REGION Network 20: #T1_ET01. ESTADO REPOSO VACIO.
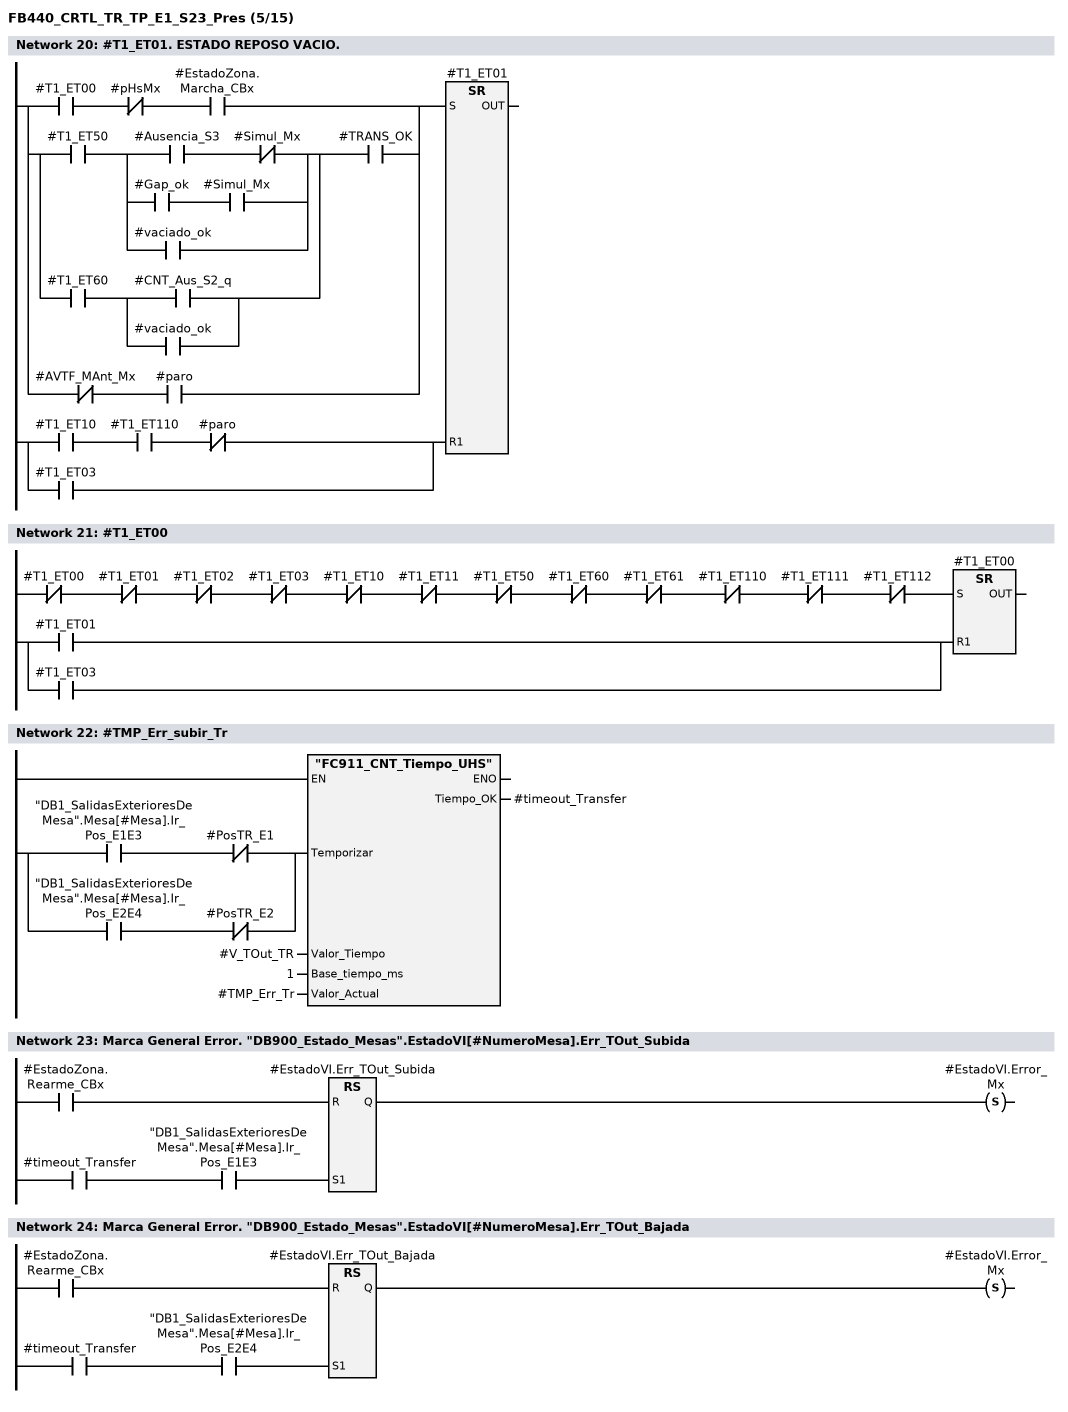
   RUNG wire#powerrail
      Contact( #T1_ET00 )
      I_Contact( #pHsMx )
      Contact( #EstadoZona.Marcha_CBx )
      wire#w1
      S_SR(operand := #T1_ET01, r1 := wire#w5)
   END_RUNG
   RUNG wire#powerrail
      Contact( #T1_ET50 )
      wire#w2
      Contact( #Ausencia_S3 )
      I_Contact( #Simul_Mx )
      wire#w3
      Contact( #TRANS_OK )
   END_RUNG wire#w1
   RUNG wire#w2
      Contact( #Gap_ok )
      Contact( #Simul_Mx )
   END_RUNG wire#w3
   RUNG wire#w2
      Contact( #vaciado_ok )
   END_RUNG wire#w3
   RUNG wire#powerrail
      Contact( #T1_ET60 )
      wire#w4
      Contact( #CNT_Aus_S2_q )
   END_RUNG wire#w3
   RUNG wire#w4
      Contact( #vaciado_ok )
   END_RUNG wire#w3
   RUNG wire#powerrail
      I_Contact( #AVTF_MAnt_Mx )
      Contact( #paro )
   END_RUNG wire#w1
   RUNG wire#powerrail
      Contact( #T1_ET10 )
      Contact( #T1_ET110 )
      I_Contact( #paro )
   END_RUNG wire#w5
   RUNG wire#powerrail
      Contact( #T1_ET03 )
   END_RUNG wire#w5
   // the same network as SCL:
   IF (#T1_ET00 AND NOT #pHsMx AND #EstadoZona.Marcha_CBx) OR (((#T1_ET50 AND ((#Ausencia_S3 AND NOT #Simul_Mx) OR (#Gap_ok AND #Simul_Mx) OR #vaciado_ok)) OR (#T1_ET60 AND (#CNT_Aus_S2_q OR #vaciado_ok))) AND #TRANS_OK) OR (NOT #AVTF_MAnt_Mx AND #paro) THEN
       #T1_ET01 := TRUE;   // SR flip-flop
   END_IF;
   IF (#T1_ET10 AND #T1_ET110 AND NOT #paro) OR #T1_ET03 THEN #T1_ET01 := FALSE; END_IF;
END_REGION

REGION Network 21: #T1_ET00
   RUNG wire#powerrail
      I_Contact( #T1_ET00 )
      I_Contact( #T1_ET01 )
      I_Contact( #T1_ET02 )
      I_Contact( #T1_ET03 )
      I_Contact( #T1_ET10 )
      I_Contact( #T1_ET11 )
      I_Contact( #T1_ET50 )
      I_Contact( #T1_ET60 )
      I_Contact( #T1_ET61 )
      I_Contact( #T1_ET110 )
      I_Contact( #T1_ET111 )
      I_Contact( #T1_ET112 )
      S_SR(operand := #T1_ET00, r1 := wire#w1)
   END_RUNG
   RUNG wire#powerrail
      Contact( #T1_ET01 )
   END_RUNG wire#w1
   RUNG wire#powerrail
      Contact( #T1_ET03 )
   END_RUNG wire#w1
   // the same network as SCL:
   IF NOT #T1_ET00 AND NOT #T1_ET01 AND NOT #T1_ET02 AND NOT #T1_ET03 AND NOT #T1_ET10 AND NOT #T1_ET11 AND NOT #T1_ET50 AND NOT #T1_ET60 AND NOT #T1_ET61 AND NOT #T1_ET110 AND NOT #T1_ET111 AND NOT #T1_ET112 THEN
       #T1_ET00 := TRUE;   // SR flip-flop
   END_IF;
   IF #T1_ET01 OR #T1_ET03 THEN #T1_ET00 := FALSE; END_IF;
END_REGION

REGION Network 22: #TMP_Err_subir_Tr
   RUNG wire#powerrail
      "FC911_CNT_Tiempo_UHS"(Temporizar := wire#w1, Valor_Tiempo := #V_TOut_TR, Base_tiempo_ms := 1, Valor_Actual := #TMP_Err_Tr, Tiempo_OK => #timeout_Transfer)
   END_RUNG
   RUNG wire#powerrail
      Contact( "DB1_SalidasExterioresDeMesa".Mesa[#Mesa].Ir_Pos_E1E3 )
      I_Contact( #PosTR_E1 )
   END_RUNG wire#w1
   RUNG wire#powerrail
      Contact( "DB1_SalidasExterioresDeMesa".Mesa[#Mesa].Ir_Pos_E2E4 )
      I_Contact( #PosTR_E2 )
   END_RUNG wire#w1
   // the same network as SCL:
   "FC911_CNT_Tiempo_UHS"(Temporizar := ("DB1_SalidasExterioresDeMesa".Mesa[#Mesa].Ir_Pos_E1E3 AND NOT #PosTR_E1) OR ("DB1_SalidasExterioresDeMesa".Mesa[#Mesa].Ir_Pos_E2E4 AND NOT #PosTR_E2),
                          Valor_Tiempo := #V_TOut_TR,
                          Base_tiempo_ms := 1,
                          Valor_Actual := #TMP_Err_Tr,
                          Tiempo_OK => #timeout_Transfer);
END_REGION

REGION Network 23: Marca General Error. "DB900_Estado_Mesas".EstadoVI[#NumeroMesa].Err_TOut_Subida
   RUNG wire#powerrail
      Contact( #EstadoZona.Rearme_CBx )
      S_RS(operand := #EstadoVI.Err_TOut_Subida, s1 := wire#w1)
      S_Coil( #EstadoVI.Error_Mx )
   END_RUNG
   RUNG wire#powerrail
      Contact( #timeout_Transfer )
      Contact( "DB1_SalidasExterioresDeMesa".Mesa[#Mesa].Ir_Pos_E1E3 )
   END_RUNG wire#w1
   // the same network as SCL:
   IF #EstadoZona.Rearme_CBx THEN
       #EstadoVI.Err_TOut_Subida := FALSE;   // RS flip-flop
   END_IF;
   IF #timeout_Transfer AND "DB1_SalidasExterioresDeMesa".Mesa[#Mesa].Ir_Pos_E1E3 THEN
       #EstadoVI.Err_TOut_Subida := TRUE;
   END_IF;
   IF #EstadoVI.Err_TOut_Subida THEN #EstadoVI.Error_Mx := TRUE; END_IF;
END_REGION

REGION Network 24: Marca General Error. "DB900_Estado_Mesas".EstadoVI[#NumeroMesa].Err_TOut_Bajada
   RUNG wire#powerrail
      Contact( #EstadoZona.Rearme_CBx )
      S_RS(operand := #EstadoVI.Err_TOut_Bajada, s1 := wire#w1)
      S_Coil( #EstadoVI.Error_Mx )
   END_RUNG
   RUNG wire#powerrail
      Contact( #timeout_Transfer )
      Contact( "DB1_SalidasExterioresDeMesa".Mesa[#Mesa].Ir_Pos_E2E4 )
   END_RUNG wire#w1
   // the same network as SCL:
   IF #EstadoZona.Rearme_CBx THEN
       #EstadoVI.Err_TOut_Bajada := FALSE;   // RS flip-flop
   END_IF;
   IF #timeout_Transfer AND "DB1_SalidasExterioresDeMesa".Mesa[#Mesa].Ir_Pos_E2E4 THEN
       #EstadoVI.Err_TOut_Bajada := TRUE;
   END_IF;
   IF #EstadoVI.Err_TOut_Bajada THEN #EstadoVI.Error_Mx := TRUE; END_IF;
END_REGION

REGION Network 25: Marca General Error. "DB900_Estado_Mesas".EstadoVI[#NumeroMesa].Err_Termico_E1_E3
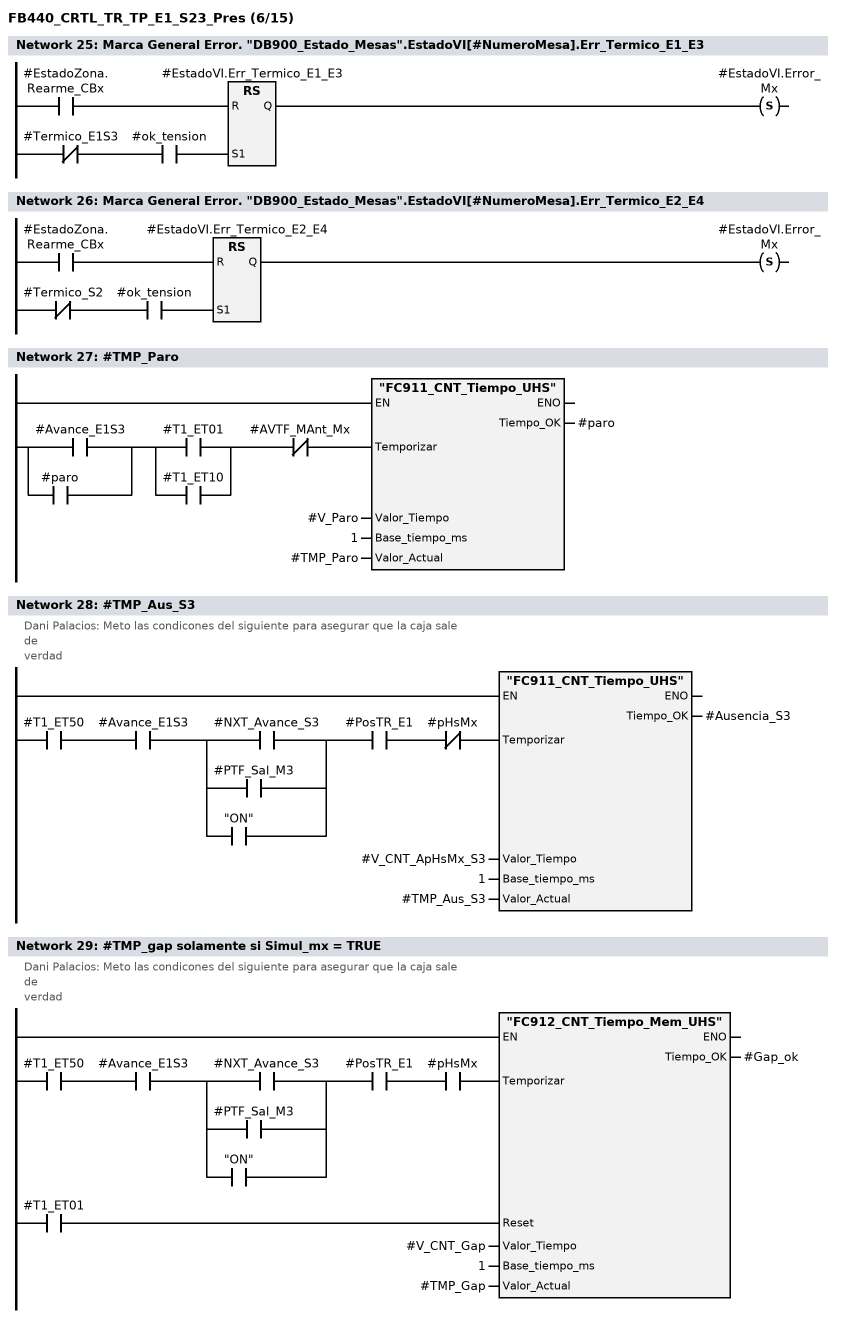
   RUNG wire#powerrail
      Contact( #EstadoZona.Rearme_CBx )
      S_RS(operand := #EstadoVI.Err_Termico_E1_E3, s1 := wire#w1)
      S_Coil( #EstadoVI.Error_Mx )
   END_RUNG
   RUNG wire#powerrail
      I_Contact( #Termico_E1S3 )
      Contact( #ok_tension )
   END_RUNG wire#w1
   // the same network as SCL:
   IF #EstadoZona.Rearme_CBx THEN
       #EstadoVI.Err_Termico_E1_E3 := FALSE;   // RS flip-flop
   END_IF;
   IF NOT #Termico_E1S3 AND #ok_tension THEN #EstadoVI.Err_Termico_E1_E3 := TRUE; END_IF;
   IF #EstadoVI.Err_Termico_E1_E3 THEN #EstadoVI.Error_Mx := TRUE; END_IF;
END_REGION

REGION Network 26: Marca General Error. "DB900_Estado_Mesas".EstadoVI[#NumeroMesa].Err_Termico_E2_E4
   RUNG wire#powerrail
      Contact( #EstadoZona.Rearme_CBx )
      S_RS(operand := #EstadoVI.Err_Termico_E2_E4, s1 := wire#w1)
      S_Coil( #EstadoVI.Error_Mx )
   END_RUNG
   RUNG wire#powerrail
      I_Contact( #Termico_S2 )
      Contact( #ok_tension )
   END_RUNG wire#w1
   // the same network as SCL:
   IF #EstadoZona.Rearme_CBx THEN
       #EstadoVI.Err_Termico_E2_E4 := FALSE;   // RS flip-flop
   END_IF;
   IF NOT #Termico_S2 AND #ok_tension THEN #EstadoVI.Err_Termico_E2_E4 := TRUE; END_IF;
   IF #EstadoVI.Err_Termico_E2_E4 THEN #EstadoVI.Error_Mx := TRUE; END_IF;
END_REGION

REGION Network 27: #TMP_Paro
   RUNG wire#powerrail
      "FC911_CNT_Tiempo_UHS"(Temporizar := wire#w3, Valor_Tiempo := #V_Paro, Base_tiempo_ms := 1, Valor_Actual := #TMP_Paro, Tiempo_OK => #paro)
   END_RUNG
   RUNG wire#powerrail
      Contact( #Avance_E1S3 )
      wire#w1
      Contact( #T1_ET01 )
      wire#w2
      I_Contact( #AVTF_MAnt_Mx )
   END_RUNG wire#w3
   RUNG wire#powerrail
      Contact( #paro )
   END_RUNG wire#w1
   RUNG wire#w1
      Contact( #T1_ET10 )
   END_RUNG wire#w2
   // the same network as SCL:
   "FC911_CNT_Tiempo_UHS"(Temporizar := (#Avance_E1S3 OR #paro) AND (#T1_ET01 OR #T1_ET10) AND NOT #AVTF_MAnt_Mx,
                          Valor_Tiempo := #V_Paro,
                          Base_tiempo_ms := 1,
                          Valor_Actual := #TMP_Paro,
                          Tiempo_OK => #paro);
END_REGION

REGION Network 28: #TMP_Aus_S3
   // Dani Palacios: Meto las condicones del siguiente para asegurar que la caja sale 
   // de 
   // verdad
   RUNG wire#powerrail
      "FC911_CNT_Tiempo_UHS"(Temporizar := wire#w3, Valor_Tiempo := #V_CNT_ApHsMx_S3, Base_tiempo_ms := 1, Valor_Actual := #TMP_Aus_S3, Tiempo_OK => #Ausencia_S3)
   END_RUNG
   RUNG wire#powerrail
      Contact( #T1_ET50 )
      Contact( #Avance_E1S3 )
      wire#w1
      Contact( #NXT_Avance_S3 )
      wire#w2
      Contact( #PosTR_E1 )
      I_Contact( #pHsMx )
   END_RUNG wire#w3
   RUNG wire#w1
      Contact( #PTF_Sal_M3 )
   END_RUNG wire#w2
   RUNG wire#w1
      Contact( "ON" )
   END_RUNG wire#w2
   // the same network as SCL:
   "FC911_CNT_Tiempo_UHS"(Temporizar := #T1_ET50 AND #Avance_E1S3 AND (#NXT_Avance_S3 OR #PTF_Sal_M3 OR "ON") AND #PosTR_E1 AND NOT #pHsMx,
                          Valor_Tiempo := #V_CNT_ApHsMx_S3,
                          Base_tiempo_ms := 1,
                          Valor_Actual := #TMP_Aus_S3,
                          Tiempo_OK => #Ausencia_S3);
END_REGION

REGION Network 29: #TMP_gap solamente si Simul_mx = TRUE
   // Dani Palacios: Meto las condicones del siguiente para asegurar que la caja sale 
   // de 
   // verdad
   RUNG wire#powerrail
      "FC912_CNT_Tiempo_Mem_UHS"(Temporizar := wire#w3, Reset := wire#w4, Valor_Tiempo := #V_CNT_Gap, Base_tiempo_ms := 1, Valor_Actual := #TMP_Gap, Tiempo_OK => #Gap_ok)
   END_RUNG
   RUNG wire#powerrail
      Contact( #T1_ET50 )
      Contact( #Avance_E1S3 )
      wire#w1
      Contact( #NXT_Avance_S3 )
      wire#w2
      Contact( #PosTR_E1 )
      Contact( #pHsMx )
   END_RUNG wire#w3
   RUNG wire#w1
      Contact( #PTF_Sal_M3 )
   END_RUNG wire#w2
   RUNG wire#w1
      Contact( "ON" )
   END_RUNG wire#w2
   RUNG wire#powerrail
      Contact( #T1_ET01 )
   END_RUNG wire#w4
   // the same network as SCL:
   "FC912_CNT_Tiempo_Mem_UHS"(Temporizar := #T1_ET50 AND #Avance_E1S3 AND (#NXT_Avance_S3 OR #PTF_Sal_M3 OR "ON") AND #PosTR_E1 AND #pHsMx,
                           Reset := #T1_ET01,
                           Valor_Tiempo := #V_CNT_Gap,
                           Base_tiempo_ms := 1,
                           Valor_Actual := #TMP_Gap,
                           Tiempo_OK => #Gap_ok);
END_REGION

REGION Network 30: tout avance
   // Nieves 16/12/17. incluyo porque no existe el error
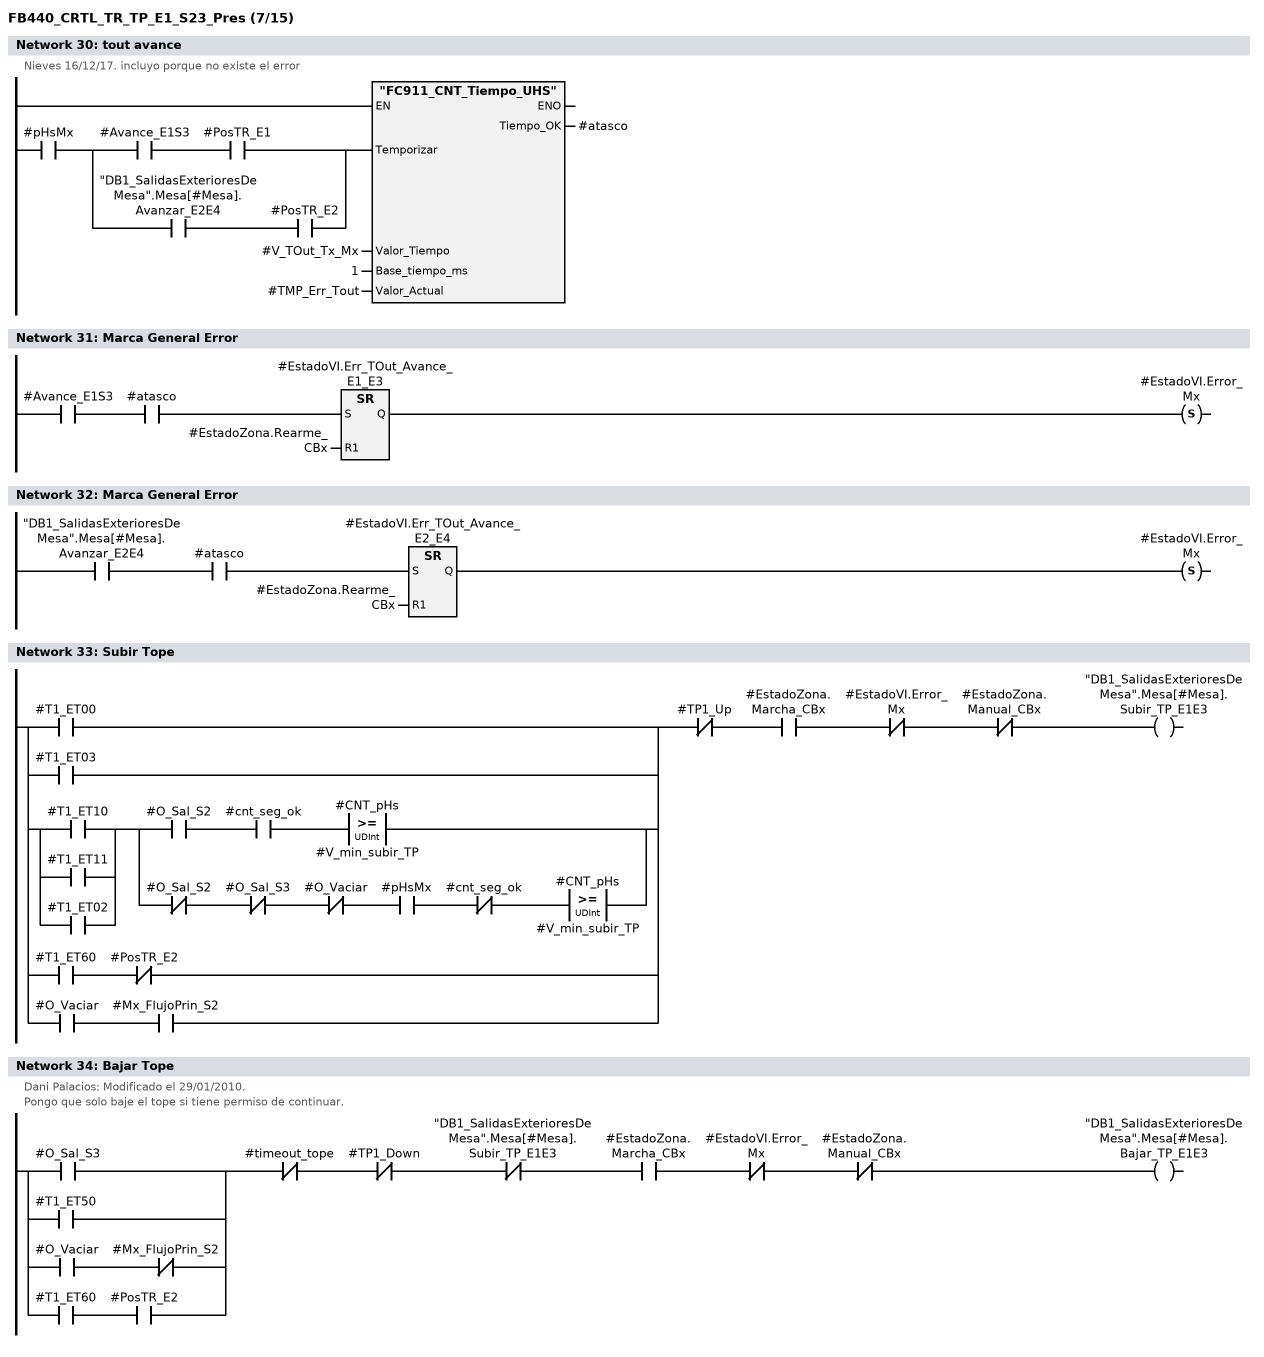
   RUNG wire#powerrail
      "FC911_CNT_Tiempo_UHS"(Temporizar := wire#w2, Valor_Tiempo := #V_TOut_Tx_Mx, Base_tiempo_ms := 1, Valor_Actual := #TMP_Err_Tout, Tiempo_OK => #atasco)
   END_RUNG
   RUNG wire#powerrail
      Contact( #pHsMx )
      wire#w1
      Contact( #Avance_E1S3 )
      Contact( #PosTR_E1 )
   END_RUNG wire#w2
   RUNG wire#w1
      Contact( "DB1_SalidasExterioresDeMesa".Mesa[#Mesa].Avanzar_E2E4 )
      Contact( #PosTR_E2 )
   END_RUNG wire#w2
   // the same network as SCL:
   "FC911_CNT_Tiempo_UHS"(Temporizar := #pHsMx AND ((#Avance_E1S3 AND #PosTR_E1) OR ("DB1_SalidasExterioresDeMesa".Mesa[#Mesa].Avanzar_E2E4 AND #PosTR_E2)),
                          Valor_Tiempo := #V_TOut_Tx_Mx,
                          Base_tiempo_ms := 1,
                          Valor_Actual := #TMP_Err_Tout,
                          Tiempo_OK => #atasco);
END_REGION

REGION Network 31: Marca General Error
   RUNG wire#powerrail
      Contact( #Avance_E1S3 )
      Contact( #atasco )
      S_SR(operand := #EstadoVI.Err_TOut_Avance_E1_E3, r1 := #EstadoZona.Rearme_CBx)
      S_Coil( #EstadoVI.Error_Mx )
   END_RUNG
   // the same network as SCL:
   IF #Avance_E1S3 AND #atasco THEN
       #EstadoVI.Err_TOut_Avance_E1_E3 := TRUE;   // SR flip-flop
   END_IF;
   IF #EstadoZona.Rearme_CBx THEN #EstadoVI.Err_TOut_Avance_E1_E3 := FALSE; END_IF;
   IF #EstadoVI.Err_TOut_Avance_E1_E3 THEN #EstadoVI.Error_Mx := TRUE; END_IF;
END_REGION

REGION Network 32: Marca General Error
   RUNG wire#powerrail
      Contact( "DB1_SalidasExterioresDeMesa".Mesa[#Mesa].Avanzar_E2E4 )
      Contact( #atasco )
      S_SR(operand := #EstadoVI.Err_TOut_Avance_E2_E4, r1 := #EstadoZona.Rearme_CBx)
      S_Coil( #EstadoVI.Error_Mx )
   END_RUNG
   // the same network as SCL:
   IF "DB1_SalidasExterioresDeMesa".Mesa[#Mesa].Avanzar_E2E4 AND #atasco THEN
       #EstadoVI.Err_TOut_Avance_E2_E4 := TRUE;   // SR flip-flop
   END_IF;
   IF #EstadoZona.Rearme_CBx THEN #EstadoVI.Err_TOut_Avance_E2_E4 := FALSE; END_IF;
   IF #EstadoVI.Err_TOut_Avance_E2_E4 THEN #EstadoVI.Error_Mx := TRUE; END_IF;
END_REGION

REGION Network 33: Subir Tope
   RUNG wire#powerrail
      Contact( #T1_ET00 )
      wire#w1
      I_Contact( #TP1_Up )
      Contact( #EstadoZona.Marcha_CBx )
      I_Contact( #EstadoVI.Error_Mx )
      I_Contact( #EstadoZona.Manual_CBx )
      Coil( "DB1_SalidasExterioresDeMesa".Mesa[#Mesa].Subir_TP_E1E3 )
   END_RUNG
   RUNG wire#powerrail
      Contact( #T1_ET03 )
   END_RUNG wire#w1
   RUNG wire#powerrail
      Contact( #T1_ET10 )
      wire#w2
      Contact( #O_Sal_S2 )
      Contact( #cnt_seg_ok )
      { S7_Templates := "SrcType := UDInt" } GE_Contact(in1 := #CNT_pHs, in2 := #V_min_subir_TP)
   END_RUNG wire#w1
   RUNG wire#powerrail
      Contact( #T1_ET11 )
   END_RUNG wire#w2
   RUNG wire#powerrail
      Contact( #T1_ET02 )
   END_RUNG wire#w2
   RUNG wire#w2
      I_Contact( #O_Sal_S2 )
      I_Contact( #O_Sal_S3 )
      I_Contact( #O_Vaciar )
      Contact( #pHsMx )
      I_Contact( #cnt_seg_ok )
      { S7_Templates := "SrcType := UDInt" } GE_Contact(in1 := #CNT_pHs, in2 := #V_min_subir_TP)
   END_RUNG wire#w1
   RUNG wire#powerrail
      Contact( #T1_ET60 )
      I_Contact( #PosTR_E2 )
   END_RUNG wire#w1
   RUNG wire#powerrail
      Contact( #O_Vaciar )
      Contact( #Mx_FlujoPrin_S2 )
   END_RUNG wire#w1
   // the same network as SCL:
   "DB1_SalidasExterioresDeMesa".Mesa[#Mesa].Subir_TP_E1E3 := (#T1_ET00 OR #T1_ET03 OR ((#T1_ET10 OR #T1_ET11 OR #T1_ET02) AND ((#O_Sal_S2 AND #cnt_seg_ok AND (#CNT_pHs >= #V_min_subir_TP)) OR (NOT #O_Sal_S2 AND NOT #O_Sal_S3 AND NOT #O_Vaciar AND #pHsMx AND NOT #cnt_seg_ok AND (#CNT_pHs >= #V_min_subir_TP)))) OR (#T1_ET60 AND NOT #PosTR_E2) OR (#O_Vaciar AND #Mx_FlujoPrin_S2)) AND NOT #TP1_Up AND #EstadoZona.Marcha_CBx AND NOT #EstadoVI.Error_Mx AND NOT #EstadoZona.Manual_CBx;
END_REGION

REGION Network 34: Bajar Tope
   // Dani Palacios: Modificado el 29/01/2010.
   // Pongo que solo baje el tope si tiene permiso de continuar.
   RUNG wire#powerrail
      Contact( #O_Sal_S3 )
      wire#w1
      I_Contact( #timeout_tope )
      I_Contact( #TP1_Down )
      I_Contact( "DB1_SalidasExterioresDeMesa".Mesa[#Mesa].Subir_TP_E1E3 )
      Contact( #EstadoZona.Marcha_CBx )
      I_Contact( #EstadoVI.Error_Mx )
      I_Contact( #EstadoZona.Manual_CBx )
      Coil( "DB1_SalidasExterioresDeMesa".Mesa[#Mesa].Bajar_TP_E1E3 )
   END_RUNG
   RUNG wire#powerrail
      Contact( #T1_ET50 )
   END_RUNG wire#w1
   RUNG wire#powerrail
      Contact( #O_Vaciar )
      I_Contact( #Mx_FlujoPrin_S2 )
   END_RUNG wire#w1
   RUNG wire#powerrail
      Contact( #T1_ET60 )
      Contact( #PosTR_E2 )
   END_RUNG wire#w1
   // the same network as SCL:
   "DB1_SalidasExterioresDeMesa".Mesa[#Mesa].Bajar_TP_E1E3 := (#O_Sal_S3 OR #T1_ET50 OR (#O_Vaciar AND NOT #Mx_FlujoPrin_S2) OR (#T1_ET60 AND #PosTR_E2)) AND NOT #timeout_tope AND NOT #TP1_Down AND NOT "DB1_SalidasExterioresDeMesa".Mesa[#Mesa].Subir_TP_E1E3 AND #EstadoZona.Marcha_CBx AND NOT #EstadoVI.Error_Mx AND NOT #EstadoZona.Manual_CBx;
END_REGION

REGION Network 35: #TIM_TP_DW
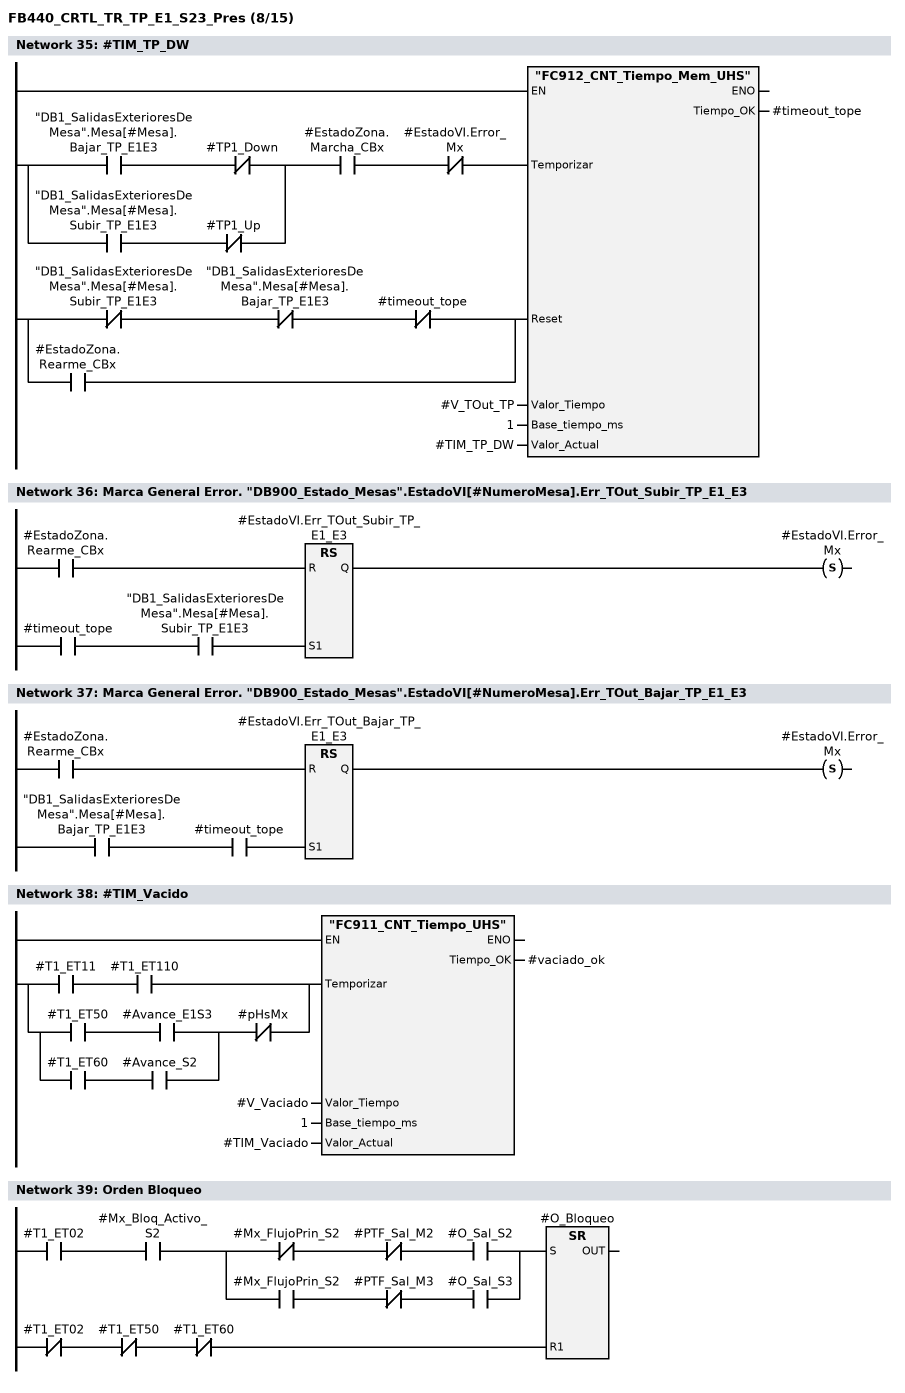
   RUNG wire#powerrail
      "FC912_CNT_Tiempo_Mem_UHS"(Temporizar := wire#w2, Reset := wire#w3, Valor_Tiempo := #V_TOut_TP, Base_tiempo_ms := 1, Valor_Actual := #TIM_TP_DW, Tiempo_OK => #timeout_tope)
   END_RUNG
   RUNG wire#powerrail
      Contact( "DB1_SalidasExterioresDeMesa".Mesa[#Mesa].Bajar_TP_E1E3 )
      I_Contact( #TP1_Down )
      wire#w1
      Contact( #EstadoZona.Marcha_CBx )
      I_Contact( #EstadoVI.Error_Mx )
   END_RUNG wire#w2
   RUNG wire#powerrail
      Contact( "DB1_SalidasExterioresDeMesa".Mesa[#Mesa].Subir_TP_E1E3 )
      I_Contact( #TP1_Up )
   END_RUNG wire#w1
   RUNG wire#powerrail
      I_Contact( "DB1_SalidasExterioresDeMesa".Mesa[#Mesa].Subir_TP_E1E3 )
      I_Contact( "DB1_SalidasExterioresDeMesa".Mesa[#Mesa].Bajar_TP_E1E3 )
      I_Contact( #timeout_tope )
   END_RUNG wire#w3
   RUNG wire#powerrail
      Contact( #EstadoZona.Rearme_CBx )
   END_RUNG wire#w3
   // the same network as SCL:
   "FC912_CNT_Tiempo_Mem_UHS"(Temporizar := (("DB1_SalidasExterioresDeMesa".Mesa[#Mesa].Bajar_TP_E1E3 AND NOT #TP1_Down) OR ("DB1_SalidasExterioresDeMesa".Mesa[#Mesa].Subir_TP_E1E3 AND NOT #TP1_Up)) AND #EstadoZona.Marcha_CBx AND NOT #EstadoVI.Error_Mx,
                           Reset := (NOT "DB1_SalidasExterioresDeMesa".Mesa[#Mesa].Subir_TP_E1E3 AND NOT "DB1_SalidasExterioresDeMesa".Mesa[#Mesa].Bajar_TP_E1E3 AND NOT #timeout_tope) OR #EstadoZona.Rearme_CBx,
                           Valor_Tiempo := #V_TOut_TP,
                           Base_tiempo_ms := 1,
                           Valor_Actual := #TIM_TP_DW,
                           Tiempo_OK => #timeout_tope);
END_REGION

REGION Network 36: Marca General Error. "DB900_Estado_Mesas".EstadoVI[#NumeroMesa].Err_TOut_Subir_TP_E1_E3
   RUNG wire#powerrail
      Contact( #EstadoZona.Rearme_CBx )
      S_RS(operand := #EstadoVI.Err_TOut_Subir_TP_E1_E3, s1 := wire#w1)
      S_Coil( #EstadoVI.Error_Mx )
   END_RUNG
   RUNG wire#powerrail
      Contact( #timeout_tope )
      Contact( "DB1_SalidasExterioresDeMesa".Mesa[#Mesa].Subir_TP_E1E3 )
   END_RUNG wire#w1
   // the same network as SCL:
   IF #EstadoZona.Rearme_CBx THEN
       #EstadoVI.Err_TOut_Subir_TP_E1_E3 := FALSE;   // RS flip-flop
   END_IF;
   IF #timeout_tope AND "DB1_SalidasExterioresDeMesa".Mesa[#Mesa].Subir_TP_E1E3 THEN
       #EstadoVI.Err_TOut_Subir_TP_E1_E3 := TRUE;
   END_IF;
   IF #EstadoVI.Err_TOut_Subir_TP_E1_E3 THEN #EstadoVI.Error_Mx := TRUE; END_IF;
END_REGION

REGION Network 37: Marca General Error. "DB900_Estado_Mesas".EstadoVI[#NumeroMesa].Err_TOut_Bajar_TP_E1_E3
   RUNG wire#powerrail
      Contact( #EstadoZona.Rearme_CBx )
      S_RS(operand := #EstadoVI.Err_TOut_Bajar_TP_E1_E3, s1 := wire#w1)
      S_Coil( #EstadoVI.Error_Mx )
   END_RUNG
   RUNG wire#powerrail
      Contact( "DB1_SalidasExterioresDeMesa".Mesa[#Mesa].Bajar_TP_E1E3 )
      Contact( #timeout_tope )
   END_RUNG wire#w1
   // the same network as SCL:
   IF #EstadoZona.Rearme_CBx THEN
       #EstadoVI.Err_TOut_Bajar_TP_E1_E3 := FALSE;   // RS flip-flop
   END_IF;
   IF "DB1_SalidasExterioresDeMesa".Mesa[#Mesa].Bajar_TP_E1E3 AND #timeout_tope THEN
       #EstadoVI.Err_TOut_Bajar_TP_E1_E3 := TRUE;
   END_IF;
   IF #EstadoVI.Err_TOut_Bajar_TP_E1_E3 THEN #EstadoVI.Error_Mx := TRUE; END_IF;
END_REGION

REGION Network 38: #TIM_Vacido
   RUNG wire#powerrail
      "FC911_CNT_Tiempo_UHS"(Temporizar := wire#w2, Valor_Tiempo := #V_Vaciado, Base_tiempo_ms := 1, Valor_Actual := #TIM_Vaciado, Tiempo_OK => #vaciado_ok)
   END_RUNG
   RUNG wire#powerrail
      Contact( #T1_ET11 )
      Contact( #T1_ET110 )
   END_RUNG wire#w2
   RUNG wire#powerrail
      Contact( #T1_ET50 )
      Contact( #Avance_E1S3 )
      wire#w1
      I_Contact( #pHsMx )
   END_RUNG wire#w2
   RUNG wire#powerrail
      Contact( #T1_ET60 )
      Contact( #Avance_S2 )
   END_RUNG wire#w1
   // the same network as SCL:
   "FC911_CNT_Tiempo_UHS"(Temporizar := (#T1_ET11 AND #T1_ET110) OR (((#T1_ET50 AND #Avance_E1S3) OR (#T1_ET60 AND #Avance_S2)) AND NOT #pHsMx),
                          Valor_Tiempo := #V_Vaciado,
                          Base_tiempo_ms := 1,
                          Valor_Actual := #TIM_Vaciado,
                          Tiempo_OK => #vaciado_ok);
END_REGION

REGION Network 39: Orden Bloqueo
   RUNG wire#powerrail
      Contact( #T1_ET02 )
      Contact( #Mx_Bloq_Activo_S2 )
      wire#w1
      I_Contact( #Mx_FlujoPrin_S2 )
      I_Contact( #PTF_Sal_M2 )
      Contact( #O_Sal_S2 )
      wire#w2
      S_SR(operand := #O_Bloqueo, r1 := wire#w3)
   END_RUNG
   RUNG wire#w1
      Contact( #Mx_FlujoPrin_S2 )
      I_Contact( #PTF_Sal_M3 )
      Contact( #O_Sal_S3 )
   END_RUNG wire#w2
   RUNG wire#powerrail
      I_Contact( #T1_ET02 )
      I_Contact( #T1_ET50 )
      I_Contact( #T1_ET60 )
   END_RUNG wire#w3
   // the same network as SCL:
   IF #T1_ET02 AND #Mx_Bloq_Activo_S2 AND ((NOT #Mx_FlujoPrin_S2 AND NOT #PTF_Sal_M2 AND #O_Sal_S2) OR (#Mx_FlujoPrin_S2 AND NOT #PTF_Sal_M3 AND #O_Sal_S3)) THEN
       #O_Bloqueo := TRUE;   // SR flip-flop
   END_IF;
   IF NOT #T1_ET02 AND NOT #T1_ET50 AND NOT #T1_ET60 THEN #O_Bloqueo := FALSE; END_IF;
END_REGION

REGION Network 40: GESTION ORDENES BORRADO
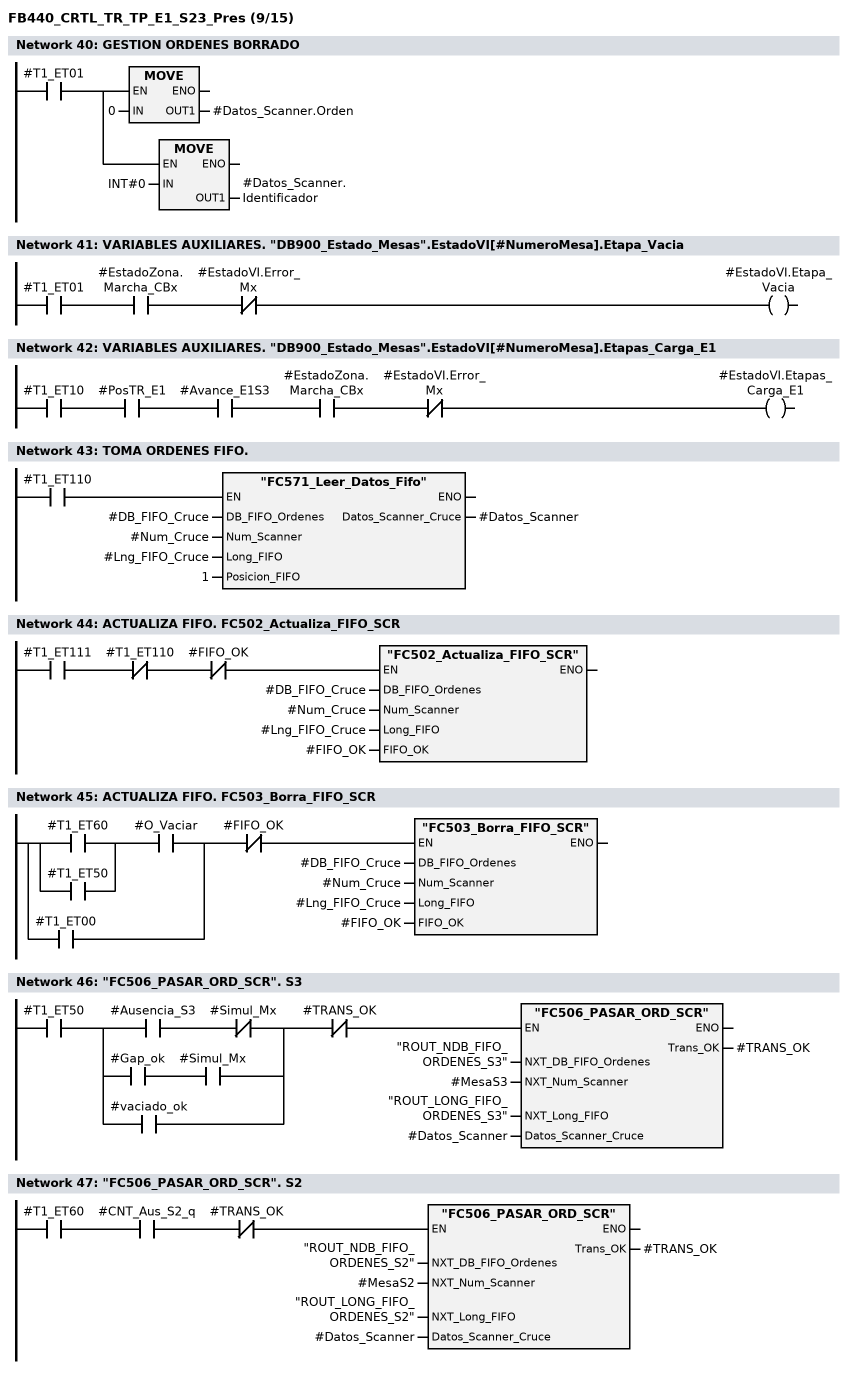
   RUNG wire#powerrail
      Contact( #T1_ET01 )
      wire#w1
      { S7_GenerateENO := "TRUE" } Move(in := 0, out1 => #Datos_Scanner.Orden)
   END_RUNG
   RUNG wire#w1
      { S7_GenerateENO := "TRUE" } Move(in := INT#0, out1 => #Datos_Scanner.Identificador)
   END_RUNG
   // the same network as SCL:
   IF #T1_ET01 THEN
       #Datos_Scanner.Orden := 0;
       #Datos_Scanner.Identificador := INT#0;
   END_IF;
END_REGION

REGION Network 41: VARIABLES AUXILIARES. "DB900_Estado_Mesas".EstadoVI[#NumeroMesa].Etapa_Vacia
   RUNG wire#powerrail
      Contact( #T1_ET01 )
      Contact( #EstadoZona.Marcha_CBx )
      I_Contact( #EstadoVI.Error_Mx )
      Coil( #EstadoVI.Etapa_Vacia )
   END_RUNG
   // the same network as SCL:
   #EstadoVI.Etapa_Vacia := #T1_ET01 AND #EstadoZona.Marcha_CBx AND NOT #EstadoVI.Error_Mx;
END_REGION

REGION Network 42: VARIABLES AUXILIARES. "DB900_Estado_Mesas".EstadoVI[#NumeroMesa].Etapas_Carga_E1
   RUNG wire#powerrail
      Contact( #T1_ET10 )
      Contact( #PosTR_E1 )
      Contact( #Avance_E1S3 )
      Contact( #EstadoZona.Marcha_CBx )
      I_Contact( #EstadoVI.Error_Mx )
      Coil( #EstadoVI.Etapas_Carga_E1 )
   END_RUNG
   // the same network as SCL:
   #EstadoVI.Etapas_Carga_E1 := #T1_ET10 AND #PosTR_E1 AND #Avance_E1S3 AND #EstadoZona.Marcha_CBx AND NOT #EstadoVI.Error_Mx;
END_REGION

REGION Network 43: TOMA ORDENES FIFO.
   RUNG wire#powerrail
      Contact( #T1_ET110 )
      "FC571_Leer_Datos_Fifo"(DB_FIFO_Ordenes := #DB_FIFO_Cruce, Num_Scanner := #Num_Cruce, Long_FIFO := #Lng_FIFO_Cruce, Posicion_FIFO := 1, Datos_Scanner_Cruce => #Datos_Scanner)
   END_RUNG
   // the same network as SCL:
   IF #T1_ET110 THEN
       "FC571_Leer_Datos_Fifo"(DB_FIFO_Ordenes := #DB_FIFO_Cruce,
                               Num_Scanner := #Num_Cruce,
                               Long_FIFO := #Lng_FIFO_Cruce,
                               Posicion_FIFO := 1,
                               Datos_Scanner_Cruce => #Datos_Scanner);
   END_IF;
END_REGION

REGION Network 44: ACTUALIZA FIFO. FC502_Actualiza_FIFO_SCR
   RUNG wire#powerrail
      Contact( #T1_ET111 )
      I_Contact( #T1_ET110 )
      I_Contact( #FIFO_OK )
      "FC502_Actualiza_FIFO_SCR"(DB_FIFO_Ordenes := #DB_FIFO_Cruce, Num_Scanner := #Num_Cruce, Long_FIFO := #Lng_FIFO_Cruce, FIFO_OK := #FIFO_OK)
   END_RUNG
   // the same network as SCL:
   IF #T1_ET111 AND NOT #T1_ET110 AND NOT #FIFO_OK THEN
       "FC502_Actualiza_FIFO_SCR"(DB_FIFO_Ordenes := #DB_FIFO_Cruce,
                               Num_Scanner := #Num_Cruce,
                               Long_FIFO := #Lng_FIFO_Cruce,
                               FIFO_OK := #FIFO_OK);
   END_IF;
END_REGION

REGION Network 45: ACTUALIZA FIFO. FC503_Borra_FIFO_SCR
   RUNG wire#powerrail
      Contact( #T1_ET60 )
      wire#w1
      Contact( #O_Vaciar )
      wire#w2
      I_Contact( #FIFO_OK )
      "FC503_Borra_FIFO_SCR"(DB_FIFO_Ordenes := #DB_FIFO_Cruce, Num_Scanner := #Num_Cruce, Long_FIFO := #Lng_FIFO_Cruce, FIFO_OK := #FIFO_OK)
   END_RUNG
   RUNG wire#powerrail
      Contact( #T1_ET50 )
   END_RUNG wire#w1
   RUNG wire#powerrail
      Contact( #T1_ET00 )
   END_RUNG wire#w2
   // the same network as SCL:
   IF (((#T1_ET60 OR #T1_ET50) AND #O_Vaciar) OR #T1_ET00) AND NOT #FIFO_OK THEN
       "FC503_Borra_FIFO_SCR"(DB_FIFO_Ordenes := #DB_FIFO_Cruce,
                              Num_Scanner := #Num_Cruce,
                              Long_FIFO := #Lng_FIFO_Cruce,
                              FIFO_OK := #FIFO_OK);
   END_IF;
END_REGION

REGION Network 46: "FC506_PASAR_ORD_SCR". S3
   RUNG wire#powerrail
      Contact( #T1_ET50 )
      wire#w1
      Contact( #Ausencia_S3 )
      I_Contact( #Simul_Mx )
      wire#w2
      I_Contact( #TRANS_OK )
      "FC506_PASAR_ORD_SCR"(NXT_DB_FIFO_Ordenes := "ROUT_NDB_FIFO_ORDENES_S3", NXT_Num_Scanner := #MesaS3, NXT_Long_FIFO := "ROUT_LONG_FIFO_ORDENES_S3", Datos_Scanner_Cruce := #Datos_Scanner, Trans_OK => #TRANS_OK)
   END_RUNG
   RUNG wire#w1
      Contact( #Gap_ok )
      Contact( #Simul_Mx )
   END_RUNG wire#w2
   RUNG wire#w1
      Contact( #vaciado_ok )
   END_RUNG wire#w2
   // the same network as SCL:
   IF #T1_ET50 AND ((#Ausencia_S3 AND NOT #Simul_Mx) OR (#Gap_ok AND #Simul_Mx) OR #vaciado_ok) AND NOT #TRANS_OK THEN
       "FC506_PASAR_ORD_SCR"(NXT_DB_FIFO_Ordenes := "ROUT_NDB_FIFO_ORDENES_S3",
                             NXT_Num_Scanner := #MesaS3,
                             NXT_Long_FIFO := "ROUT_LONG_FIFO_ORDENES_S3",
                             Datos_Scanner_Cruce := #Datos_Scanner,
                             Trans_OK => #TRANS_OK);
   END_IF;
END_REGION

REGION Network 47: "FC506_PASAR_ORD_SCR". S2
   RUNG wire#powerrail
      Contact( #T1_ET60 )
      Contact( #CNT_Aus_S2_q )
      I_Contact( #TRANS_OK )
      "FC506_PASAR_ORD_SCR"(NXT_DB_FIFO_Ordenes := "ROUT_NDB_FIFO_ORDENES_S2", NXT_Num_Scanner := #MesaS2, NXT_Long_FIFO := "ROUT_LONG_FIFO_ORDENES_S2", Datos_Scanner_Cruce := #Datos_Scanner, Trans_OK => #TRANS_OK)
   END_RUNG
   // the same network as SCL:
   IF #T1_ET60 AND #CNT_Aus_S2_q AND NOT #TRANS_OK THEN
       "FC506_PASAR_ORD_SCR"(NXT_DB_FIFO_Ordenes := "ROUT_NDB_FIFO_ORDENES_S2",
                             NXT_Num_Scanner := #MesaS2,
                             NXT_Long_FIFO := "ROUT_LONG_FIFO_ORDENES_S2",
                             Datos_Scanner_Cruce := #Datos_Scanner,
                             Trans_OK => #TRANS_OK);
   END_IF;
END_REGION

REGION Network 48: #FIFO_OK
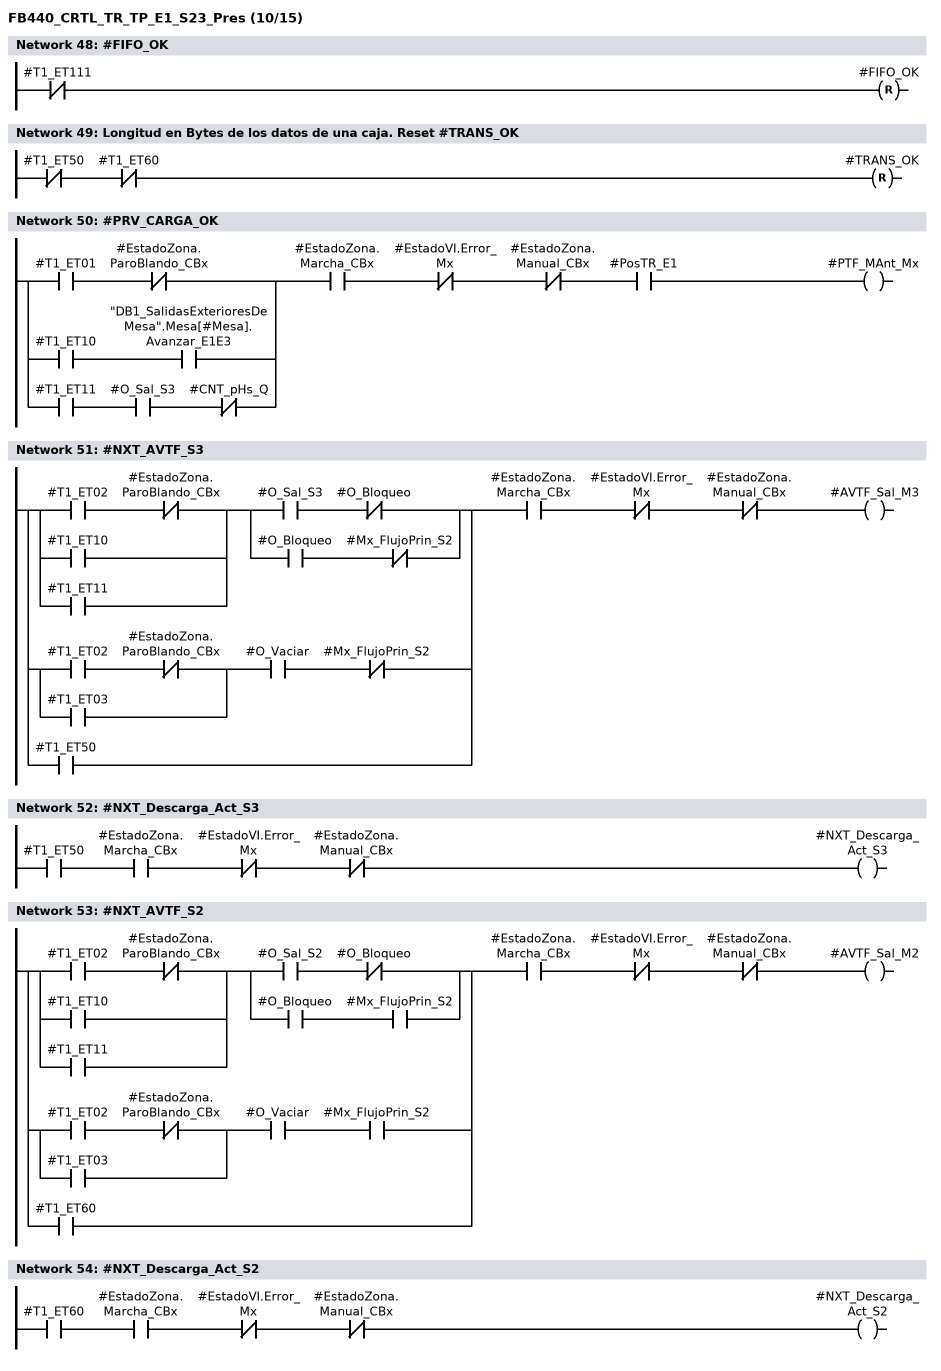
   RUNG wire#powerrail
      I_Contact( #T1_ET111 )
      R_Coil( #FIFO_OK )
   END_RUNG
   // the same network as SCL:
   IF NOT #T1_ET111 THEN #FIFO_OK := FALSE; END_IF;
END_REGION

REGION Network 49: Longitud en Bytes de los datos de una caja. Reset #TRANS_OK
   RUNG wire#powerrail
      I_Contact( #T1_ET50 )
      I_Contact( #T1_ET60 )
      R_Coil( #TRANS_OK )
   END_RUNG
   // the same network as SCL:
   IF NOT #T1_ET50 AND NOT #T1_ET60 THEN #TRANS_OK := FALSE; END_IF;
END_REGION

REGION Network 50: #PRV_CARGA_OK
   RUNG wire#powerrail
      Contact( #T1_ET01 )
      I_Contact( #EstadoZona.ParoBlando_CBx )
      wire#w1
      Contact( #EstadoZona.Marcha_CBx )
      I_Contact( #EstadoVI.Error_Mx )
      I_Contact( #EstadoZona.Manual_CBx )
      Contact( #PosTR_E1 )
      Coil( #PTF_MAnt_Mx )
   END_RUNG
   RUNG wire#powerrail
      Contact( #T1_ET10 )
      Contact( "DB1_SalidasExterioresDeMesa".Mesa[#Mesa].Avanzar_E1E3 )
   END_RUNG wire#w1
   RUNG wire#powerrail
      Contact( #T1_ET11 )
      Contact( #O_Sal_S3 )
      I_Contact( #CNT_pHs_Q )
   END_RUNG wire#w1
   // the same network as SCL:
   #PTF_MAnt_Mx := ((#T1_ET01 AND NOT #EstadoZona.ParoBlando_CBx) OR (#T1_ET10 AND "DB1_SalidasExterioresDeMesa".Mesa[#Mesa].Avanzar_E1E3) OR (#T1_ET11 AND #O_Sal_S3 AND NOT #CNT_pHs_Q)) AND #EstadoZona.Marcha_CBx AND NOT #EstadoVI.Error_Mx AND NOT #EstadoZona.Manual_CBx AND #PosTR_E1;
END_REGION

REGION Network 51: #NXT_AVTF_S3
   RUNG wire#powerrail
      Contact( #T1_ET02 )
      I_Contact( #EstadoZona.ParoBlando_CBx )
      wire#w1
      Contact( #O_Sal_S3 )
      I_Contact( #O_Bloqueo )
      wire#w2
      Contact( #EstadoZona.Marcha_CBx )
      I_Contact( #EstadoVI.Error_Mx )
      I_Contact( #EstadoZona.Manual_CBx )
      Coil( #AVTF_Sal_M3 )
   END_RUNG
   RUNG wire#powerrail
      Contact( #T1_ET10 )
   END_RUNG wire#w1
   RUNG wire#powerrail
      Contact( #T1_ET11 )
   END_RUNG wire#w1
   RUNG wire#w1
      Contact( #O_Bloqueo )
      I_Contact( #Mx_FlujoPrin_S2 )
   END_RUNG wire#w2
   RUNG wire#powerrail
      Contact( #T1_ET02 )
      I_Contact( #EstadoZona.ParoBlando_CBx )
      wire#w3
      Contact( #O_Vaciar )
      I_Contact( #Mx_FlujoPrin_S2 )
   END_RUNG wire#w2
   RUNG wire#powerrail
      Contact( #T1_ET03 )
   END_RUNG wire#w3
   RUNG wire#powerrail
      Contact( #T1_ET50 )
   END_RUNG wire#w2
   // the same network as SCL:
   #AVTF_Sal_M3 := ((((#T1_ET02 AND NOT #EstadoZona.ParoBlando_CBx) OR #T1_ET10 OR #T1_ET11) AND ((#O_Sal_S3 AND NOT #O_Bloqueo) OR (#O_Bloqueo AND NOT #Mx_FlujoPrin_S2))) OR (((#T1_ET02 AND NOT #EstadoZona.ParoBlando_CBx) OR #T1_ET03) AND #O_Vaciar AND NOT #Mx_FlujoPrin_S2) OR #T1_ET50) AND #EstadoZona.Marcha_CBx AND NOT #EstadoVI.Error_Mx AND NOT #EstadoZona.Manual_CBx;
END_REGION

REGION Network 52: #NXT_Descarga_Act_S3
   RUNG wire#powerrail
      Contact( #T1_ET50 )
      Contact( #EstadoZona.Marcha_CBx )
      I_Contact( #EstadoVI.Error_Mx )
      I_Contact( #EstadoZona.Manual_CBx )
      Coil( #NXT_Descarga_Act_S3 )
   END_RUNG
   // the same network as SCL:
   #NXT_Descarga_Act_S3 := #T1_ET50 AND #EstadoZona.Marcha_CBx AND NOT #EstadoVI.Error_Mx AND NOT #EstadoZona.Manual_CBx;
END_REGION

REGION Network 53: #NXT_AVTF_S2
   RUNG wire#powerrail
      Contact( #T1_ET02 )
      I_Contact( #EstadoZona.ParoBlando_CBx )
      wire#w1
      Contact( #O_Sal_S2 )
      I_Contact( #O_Bloqueo )
      wire#w2
      Contact( #EstadoZona.Marcha_CBx )
      I_Contact( #EstadoVI.Error_Mx )
      I_Contact( #EstadoZona.Manual_CBx )
      Coil( #AVTF_Sal_M2 )
   END_RUNG
   RUNG wire#powerrail
      Contact( #T1_ET10 )
   END_RUNG wire#w1
   RUNG wire#powerrail
      Contact( #T1_ET11 )
   END_RUNG wire#w1
   RUNG wire#w1
      Contact( #O_Bloqueo )
      Contact( #Mx_FlujoPrin_S2 )
   END_RUNG wire#w2
   RUNG wire#powerrail
      Contact( #T1_ET02 )
      I_Contact( #EstadoZona.ParoBlando_CBx )
      wire#w3
      Contact( #O_Vaciar )
      Contact( #Mx_FlujoPrin_S2 )
   END_RUNG wire#w2
   RUNG wire#powerrail
      Contact( #T1_ET03 )
   END_RUNG wire#w3
   RUNG wire#powerrail
      Contact( #T1_ET60 )
   END_RUNG wire#w2
   // the same network as SCL:
   #AVTF_Sal_M2 := ((((#T1_ET02 AND NOT #EstadoZona.ParoBlando_CBx) OR #T1_ET10 OR #T1_ET11) AND ((#O_Sal_S2 AND NOT #O_Bloqueo) OR (#O_Bloqueo AND #Mx_FlujoPrin_S2))) OR (((#T1_ET02 AND NOT #EstadoZona.ParoBlando_CBx) OR #T1_ET03) AND #O_Vaciar AND #Mx_FlujoPrin_S2) OR #T1_ET60) AND #EstadoZona.Marcha_CBx AND NOT #EstadoVI.Error_Mx AND NOT #EstadoZona.Manual_CBx;
END_REGION

REGION Network 54: #NXT_Descarga_Act_S2
   RUNG wire#powerrail
      Contact( #T1_ET60 )
      Contact( #EstadoZona.Marcha_CBx )
      I_Contact( #EstadoVI.Error_Mx )
      I_Contact( #EstadoZona.Manual_CBx )
      Coil( #NXT_Descarga_Act_S2 )
   END_RUNG
   // the same network as SCL:
   #NXT_Descarga_Act_S2 := #T1_ET60 AND #EstadoZona.Marcha_CBx AND NOT #EstadoVI.Error_Mx AND NOT #EstadoZona.Manual_CBx;
END_REGION

REGION Network 55: #MA_IR_POS_24_TR
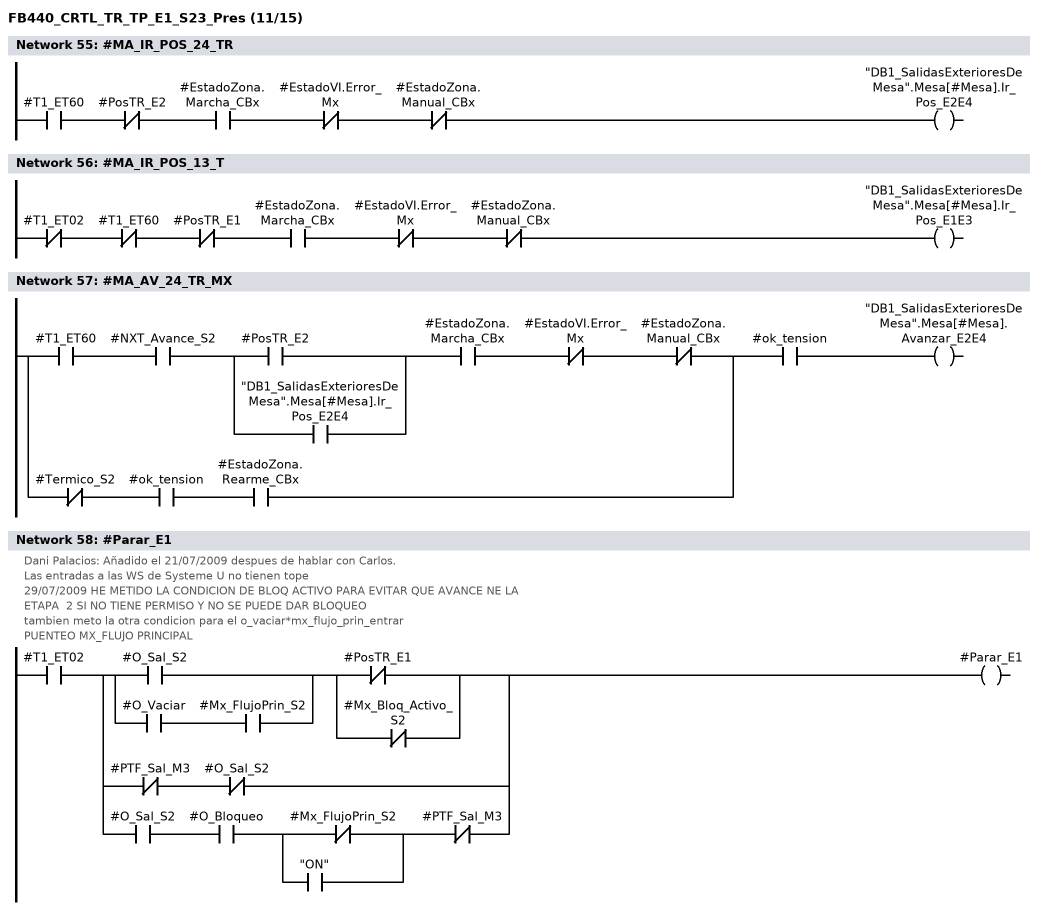
   RUNG wire#powerrail
      Contact( #T1_ET60 )
      I_Contact( #PosTR_E2 )
      Contact( #EstadoZona.Marcha_CBx )
      I_Contact( #EstadoVI.Error_Mx )
      I_Contact( #EstadoZona.Manual_CBx )
      Coil( "DB1_SalidasExterioresDeMesa".Mesa[#Mesa].Ir_Pos_E2E4 )
   END_RUNG
   // the same network as SCL:
   "DB1_SalidasExterioresDeMesa".Mesa[#Mesa].Ir_Pos_E2E4 := #T1_ET60 AND NOT #PosTR_E2 AND #EstadoZona.Marcha_CBx AND NOT #EstadoVI.Error_Mx AND NOT #EstadoZona.Manual_CBx;
END_REGION

REGION Network 56: #MA_IR_POS_13_T
   RUNG wire#powerrail
      I_Contact( #T1_ET02 )
      I_Contact( #T1_ET60 )
      I_Contact( #PosTR_E1 )
      Contact( #EstadoZona.Marcha_CBx )
      I_Contact( #EstadoVI.Error_Mx )
      I_Contact( #EstadoZona.Manual_CBx )
      Coil( "DB1_SalidasExterioresDeMesa".Mesa[#Mesa].Ir_Pos_E1E3 )
   END_RUNG
   // the same network as SCL:
   "DB1_SalidasExterioresDeMesa".Mesa[#Mesa].Ir_Pos_E1E3 := NOT #T1_ET02 AND NOT #T1_ET60 AND NOT #PosTR_E1 AND #EstadoZona.Marcha_CBx AND NOT #EstadoVI.Error_Mx AND NOT #EstadoZona.Manual_CBx;
END_REGION

REGION Network 57: #MA_AV_24_TR_MX
   RUNG wire#powerrail
      Contact( #T1_ET60 )
      Contact( #NXT_Avance_S2 )
      wire#w1
      Contact( #PosTR_E2 )
      wire#w2
      Contact( #EstadoZona.Marcha_CBx )
      I_Contact( #EstadoVI.Error_Mx )
      I_Contact( #EstadoZona.Manual_CBx )
      wire#w3
      Contact( #ok_tension )
      Coil( "DB1_SalidasExterioresDeMesa".Mesa[#Mesa].Avanzar_E2E4 )
   END_RUNG
   RUNG wire#w1
      Contact( "DB1_SalidasExterioresDeMesa".Mesa[#Mesa].Ir_Pos_E2E4 )
   END_RUNG wire#w2
   RUNG wire#powerrail
      I_Contact( #Termico_S2 )
      Contact( #ok_tension )
      Contact( #EstadoZona.Rearme_CBx )
   END_RUNG wire#w3
   // the same network as SCL:
   "DB1_SalidasExterioresDeMesa".Mesa[#Mesa].Avanzar_E2E4 := ((#T1_ET60 AND #NXT_Avance_S2 AND (#PosTR_E2 OR "DB1_SalidasExterioresDeMesa".Mesa[#Mesa].Ir_Pos_E2E4) AND #EstadoZona.Marcha_CBx AND NOT #EstadoVI.Error_Mx AND NOT #EstadoZona.Manual_CBx) OR (NOT #Termico_S2 AND #ok_tension AND #EstadoZona.Rearme_CBx)) AND #ok_tension;
END_REGION

REGION Network 58: #Parar_E1
   // Dani Palacios: Añadido el 21/07/2009 despues de hablar con Carlos.
   // Las entradas a las WS de Systeme U no tienen tope
   // 29/07/2009 HE METIDO LA CONDICION DE BLOQ ACTIVO PARA EVITAR QUE AVANCE NE LA 
   // ETAPA  2 SI NO TIENE PERMISO Y NO SE PUEDE DAR BLOQUEO
   // tambien meto la otra condicion para el o_vaciar*mx_flujo_prin_entrar
   // PUENTEO MX_FLUJO PRINCIPAL
   RUNG wire#powerrail
      Contact( #T1_ET02 )
      wire#w1
      Contact( #O_Sal_S2 )
      wire#w2
      I_Contact( #PosTR_E1 )
      wire#w3
      Coil( #Parar_E1 )
   END_RUNG
   RUNG wire#w1
      Contact( #O_Vaciar )
      Contact( #Mx_FlujoPrin_S2 )
   END_RUNG wire#w2
   RUNG wire#w2
      I_Contact( #Mx_Bloq_Activo_S2 )
   END_RUNG wire#w3
   RUNG wire#w1
      I_Contact( #PTF_Sal_M3 )
      I_Contact( #O_Sal_S2 )
   END_RUNG wire#w3
   RUNG wire#w1
      Contact( #O_Sal_S2 )
      Contact( #O_Bloqueo )
      wire#w4
      I_Contact( #Mx_FlujoPrin_S2 )
      wire#w5
      I_Contact( #PTF_Sal_M3 )
   END_RUNG wire#w3
   RUNG wire#w4
      Contact( "ON" )
   END_RUNG wire#w5
   // the same network as SCL:
   #Parar_E1 := #T1_ET02 AND (((#O_Sal_S2 OR (#O_Vaciar AND #Mx_FlujoPrin_S2)) AND (NOT #PosTR_E1 OR NOT #Mx_Bloq_Activo_S2)) OR (NOT #PTF_Sal_M3 AND NOT #O_Sal_S2) OR (#O_Sal_S2 AND #O_Bloqueo AND (NOT #Mx_FlujoPrin_S2 OR "ON") AND NOT #PTF_Sal_M3));
END_REGION

REGION Network 59: #MA_AV_13_T_MX
   // Dani Palacios: en etapa 50 se deja que avance si no fotocelula. Es para 
   // asegurar 
   // que escribe la orden en el fifo y la puede leer el siguiente
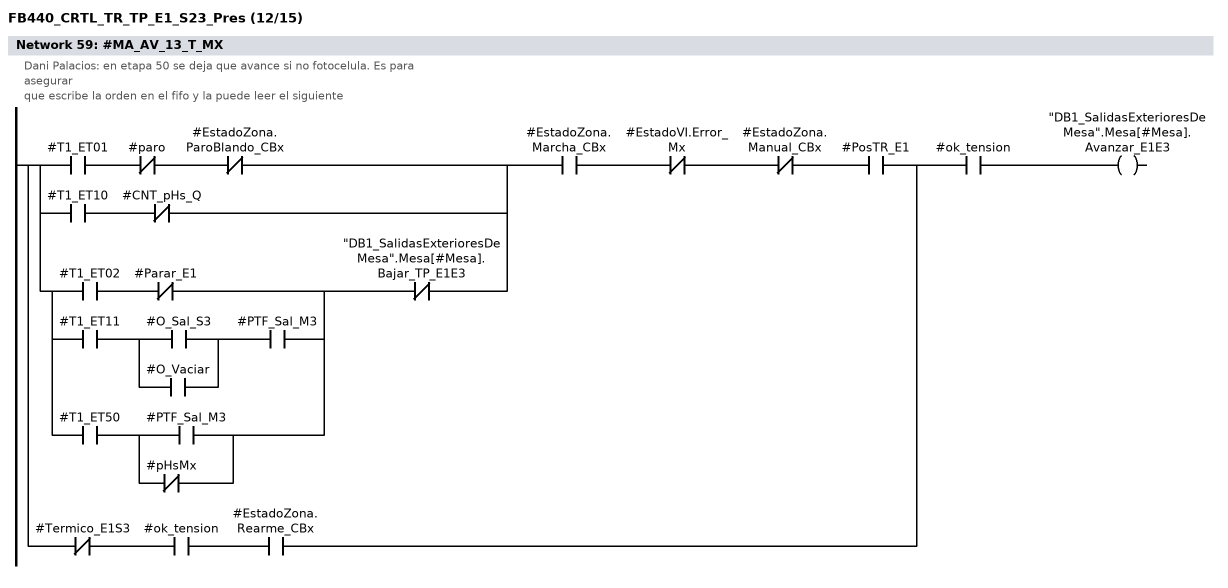
   RUNG wire#powerrail
      Contact( #T1_ET01 )
      I_Contact( #paro )
      I_Contact( #EstadoZona.ParoBlando_CBx )
      wire#w1
      Contact( #EstadoZona.Marcha_CBx )
      I_Contact( #EstadoVI.Error_Mx )
      I_Contact( #EstadoZona.Manual_CBx )
      Contact( #PosTR_E1 )
      wire#w6
      Contact( #ok_tension )
      Coil( "DB1_SalidasExterioresDeMesa".Mesa[#Mesa].Avanzar_E1E3 )
   END_RUNG
   RUNG wire#powerrail
      Contact( #T1_ET10 )
      I_Contact( #CNT_pHs_Q )
   END_RUNG wire#w1
   RUNG wire#powerrail
      Contact( #T1_ET02 )
      I_Contact( #Parar_E1 )
      wire#w2
      I_Contact( "DB1_SalidasExterioresDeMesa".Mesa[#Mesa].Bajar_TP_E1E3 )
   END_RUNG wire#w1
   RUNG wire#powerrail
      Contact( #T1_ET11 )
      wire#w3
      Contact( #O_Sal_S3 )
      wire#w4
      Contact( #PTF_Sal_M3 )
   END_RUNG wire#w2
   RUNG wire#w3
      Contact( #O_Vaciar )
   END_RUNG wire#w4
   RUNG wire#powerrail
      Contact( #T1_ET50 )
      wire#w5
      Contact( #PTF_Sal_M3 )
   END_RUNG wire#w2
   RUNG wire#w5
      I_Contact( #pHsMx )
   END_RUNG wire#w2
   RUNG wire#powerrail
      I_Contact( #Termico_E1S3 )
      Contact( #ok_tension )
      Contact( #EstadoZona.Rearme_CBx )
   END_RUNG wire#w6
   // the same network as SCL:
   "DB1_SalidasExterioresDeMesa".Mesa[#Mesa].Avanzar_E1E3 := ((((#T1_ET01 AND NOT #paro AND NOT #EstadoZona.ParoBlando_CBx) OR (#T1_ET10 AND NOT #CNT_pHs_Q) OR (((#T1_ET02 AND NOT #Parar_E1) OR (#T1_ET11 AND (#O_Sal_S3 OR #O_Vaciar) AND #PTF_Sal_M3) OR (#T1_ET50 AND (#PTF_Sal_M3 OR NOT #pHsMx))) AND NOT "DB1_SalidasExterioresDeMesa".Mesa[#Mesa].Bajar_TP_E1E3)) AND #EstadoZona.Marcha_CBx AND NOT #EstadoVI.Error_Mx AND NOT #EstadoZona.Manual_CBx AND #PosTR_E1) OR (NOT #Termico_E1S3 AND #ok_tension AND #EstadoZona.Rearme_CBx)) AND #ok_tension;
END_REGION

REGION Network 60: PASAR ETIQUETA JDT
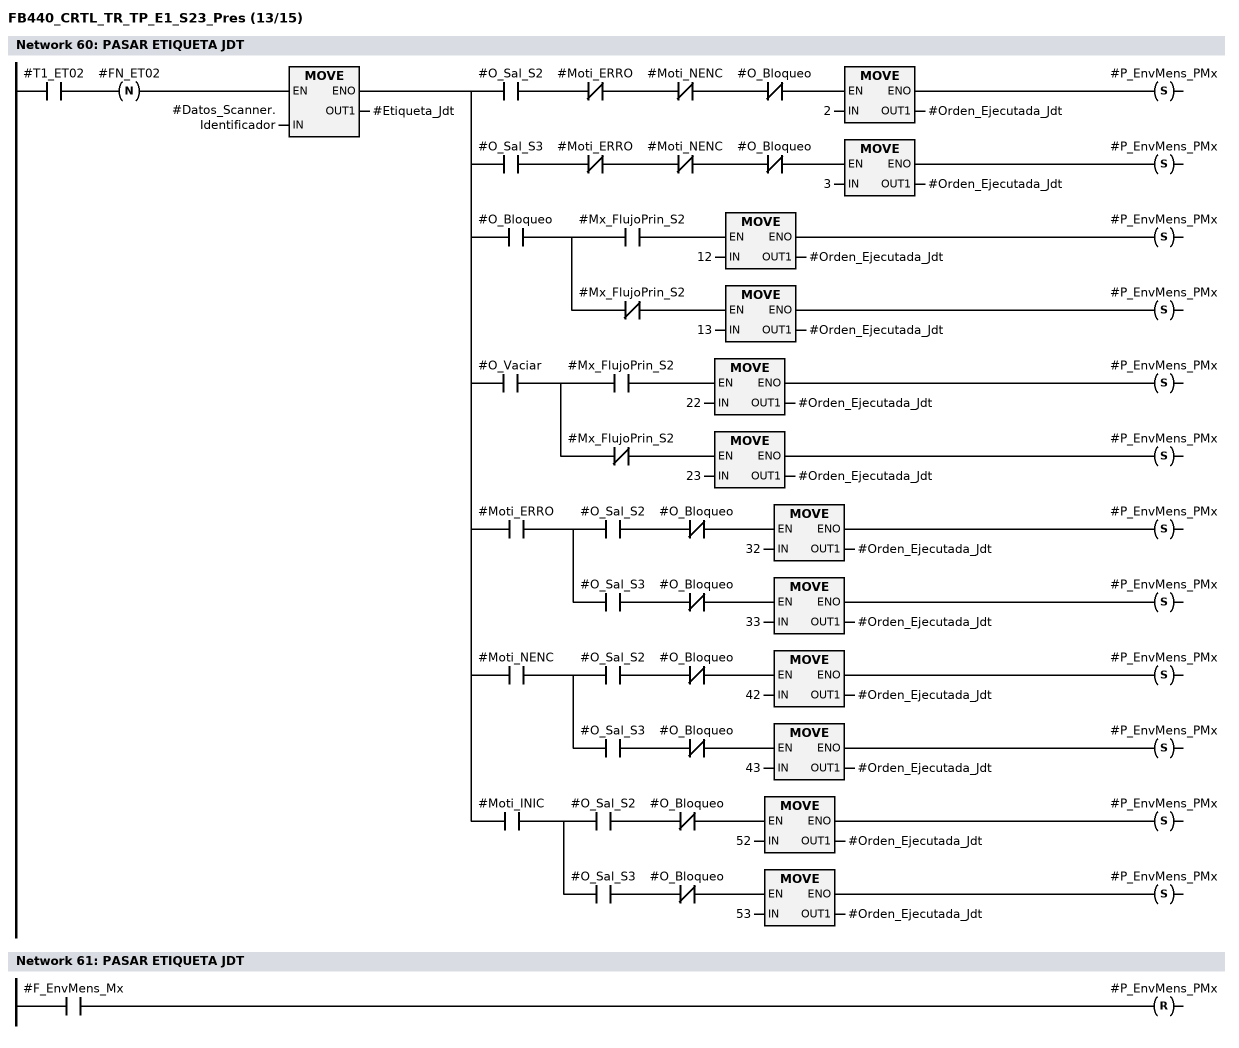
   RUNG wire#powerrail
      Contact( #T1_ET02 )
      N_Trig( #FN_ET02 )
      { S7_GenerateENO := "TRUE" } Move(in := #Datos_Scanner.Identificador, out1 => #Etiqueta_Jdt)
      wire#w1
      Contact( #O_Sal_S2 )
      I_Contact( #Moti_ERRO )
      I_Contact( #Moti_NENC )
      I_Contact( #O_Bloqueo )
      { S7_GenerateENO := "TRUE" } Move(in := 2, out1 => #Orden_Ejecutada_Jdt)
      S_Coil( #P_EnvMens_PMx )
   END_RUNG
   RUNG wire#w1
      Contact( #O_Sal_S3 )
      I_Contact( #Moti_ERRO )
      I_Contact( #Moti_NENC )
      I_Contact( #O_Bloqueo )
      { S7_GenerateENO := "TRUE" } Move(in := 3, out1 => #Orden_Ejecutada_Jdt)
      S_Coil( #P_EnvMens_PMx )
   END_RUNG
   RUNG wire#w1
      Contact( #O_Bloqueo )
      wire#w2
      Contact( #Mx_FlujoPrin_S2 )
      { S7_GenerateENO := "TRUE" } Move(in := 12, out1 => #Orden_Ejecutada_Jdt)
      S_Coil( #P_EnvMens_PMx )
   END_RUNG
   RUNG wire#w2
      I_Contact( #Mx_FlujoPrin_S2 )
      { S7_GenerateENO := "TRUE" } Move(in := 13, out1 => #Orden_Ejecutada_Jdt)
      S_Coil( #P_EnvMens_PMx )
   END_RUNG
   RUNG wire#w1
      Contact( #O_Vaciar )
      wire#w3
      Contact( #Mx_FlujoPrin_S2 )
      { S7_GenerateENO := "TRUE" } Move(in := 22, out1 => #Orden_Ejecutada_Jdt)
      S_Coil( #P_EnvMens_PMx )
   END_RUNG
   RUNG wire#w3
      I_Contact( #Mx_FlujoPrin_S2 )
      { S7_GenerateENO := "TRUE" } Move(in := 23, out1 => #Orden_Ejecutada_Jdt)
      S_Coil( #P_EnvMens_PMx )
   END_RUNG
   RUNG wire#w1
      Contact( #Moti_ERRO )
      wire#w4
      Contact( #O_Sal_S2 )
      I_Contact( #O_Bloqueo )
      { S7_GenerateENO := "TRUE" } Move(in := 32, out1 => #Orden_Ejecutada_Jdt)
      S_Coil( #P_EnvMens_PMx )
   END_RUNG
   RUNG wire#w4
      Contact( #O_Sal_S3 )
      I_Contact( #O_Bloqueo )
      { S7_GenerateENO := "TRUE" } Move(in := 33, out1 => #Orden_Ejecutada_Jdt)
      S_Coil( #P_EnvMens_PMx )
   END_RUNG
   RUNG wire#w1
      Contact( #Moti_NENC )
      wire#w5
      Contact( #O_Sal_S2 )
      I_Contact( #O_Bloqueo )
      { S7_GenerateENO := "TRUE" } Move(in := 42, out1 => #Orden_Ejecutada_Jdt)
      S_Coil( #P_EnvMens_PMx )
   END_RUNG
   RUNG wire#w5
      Contact( #O_Sal_S3 )
      I_Contact( #O_Bloqueo )
      { S7_GenerateENO := "TRUE" } Move(in := 43, out1 => #Orden_Ejecutada_Jdt)
      S_Coil( #P_EnvMens_PMx )
   END_RUNG
   RUNG wire#w1
      Contact( #Moti_INIC )
      wire#w6
      Contact( #O_Sal_S2 )
      I_Contact( #O_Bloqueo )
      { S7_GenerateENO := "TRUE" } Move(in := 52, out1 => #Orden_Ejecutada_Jdt)
      S_Coil( #P_EnvMens_PMx )
   END_RUNG
   RUNG wire#w6
      Contact( #O_Sal_S3 )
      I_Contact( #O_Bloqueo )
      { S7_GenerateENO := "TRUE" } Move(in := 53, out1 => #Orden_Ejecutada_Jdt)
      S_Coil( #P_EnvMens_PMx )
   END_RUNG
   // the same network as SCL:
   // ENO of a box is taken as its EN; it also drops when the box reports an error
   #_w1 := NOT #T1_ET02 AND #FN_ET02;   // falling edge
   #FN_ET02 := #T1_ET02;
   IF #_w1 THEN #Etiqueta_Jdt := #Datos_Scanner.Identificador; END_IF;
   IF #_w1 AND #O_Sal_S2 AND NOT #Moti_ERRO AND NOT #Moti_NENC AND NOT #O_Bloqueo THEN
       #Orden_Ejecutada_Jdt := 2;
       #P_EnvMens_PMx := TRUE;
   END_IF;
   IF #_w1 AND #O_Sal_S3 AND NOT #Moti_ERRO AND NOT #Moti_NENC AND NOT #O_Bloqueo THEN
       #Orden_Ejecutada_Jdt := 3;
       #P_EnvMens_PMx := TRUE;
   END_IF;
   #_w2 := #_w1 AND #O_Bloqueo;
   IF #_w2 AND #Mx_FlujoPrin_S2 THEN
       #Orden_Ejecutada_Jdt := 12;
       #P_EnvMens_PMx := TRUE;
   END_IF;
   IF #_w2 AND NOT #Mx_FlujoPrin_S2 THEN
       #Orden_Ejecutada_Jdt := 13;
       #P_EnvMens_PMx := TRUE;
   END_IF;
   #_w3 := #_w1 AND #O_Vaciar;
   IF #_w3 AND #Mx_FlujoPrin_S2 THEN
       #Orden_Ejecutada_Jdt := 22;
       #P_EnvMens_PMx := TRUE;
   END_IF;
   IF #_w3 AND NOT #Mx_FlujoPrin_S2 THEN
       #Orden_Ejecutada_Jdt := 23;
       #P_EnvMens_PMx := TRUE;
   END_IF;
   #_w4 := #_w1 AND #Moti_ERRO;
   IF #_w4 AND #O_Sal_S2 AND NOT #O_Bloqueo THEN
       #Orden_Ejecutada_Jdt := 32;
       #P_EnvMens_PMx := TRUE;
   END_IF;
   IF #_w4 AND #O_Sal_S3 AND NOT #O_Bloqueo THEN
       #Orden_Ejecutada_Jdt := 33;
       #P_EnvMens_PMx := TRUE;
   END_IF;
   #_w5 := #_w1 AND #Moti_NENC;
   IF #_w5 AND #O_Sal_S2 AND NOT #O_Bloqueo THEN
       #Orden_Ejecutada_Jdt := 42;
       #P_EnvMens_PMx := TRUE;
   END_IF;
   IF #_w5 AND #O_Sal_S3 AND NOT #O_Bloqueo THEN
       #Orden_Ejecutada_Jdt := 43;
       #P_EnvMens_PMx := TRUE;
   END_IF;
   #_w6 := #_w1 AND #Moti_INIC;
   IF #_w6 AND #O_Sal_S2 AND NOT #O_Bloqueo THEN
       #Orden_Ejecutada_Jdt := 52;
       #P_EnvMens_PMx := TRUE;
   END_IF;
   IF #_w6 AND #O_Sal_S3 AND NOT #O_Bloqueo THEN
       #Orden_Ejecutada_Jdt := 53;
       #P_EnvMens_PMx := TRUE;
   END_IF;
END_REGION

REGION Network 61: PASAR ETIQUETA JDT
   RUNG wire#powerrail
      Contact( #F_EnvMens_Mx )
      R_Coil( #P_EnvMens_PMx )
   END_RUNG
   // the same network as SCL:
   IF #F_EnvMens_Mx THEN #P_EnvMens_PMx := FALSE; END_IF;
END_REGION

REGION Network 62: ESTADOS MESA
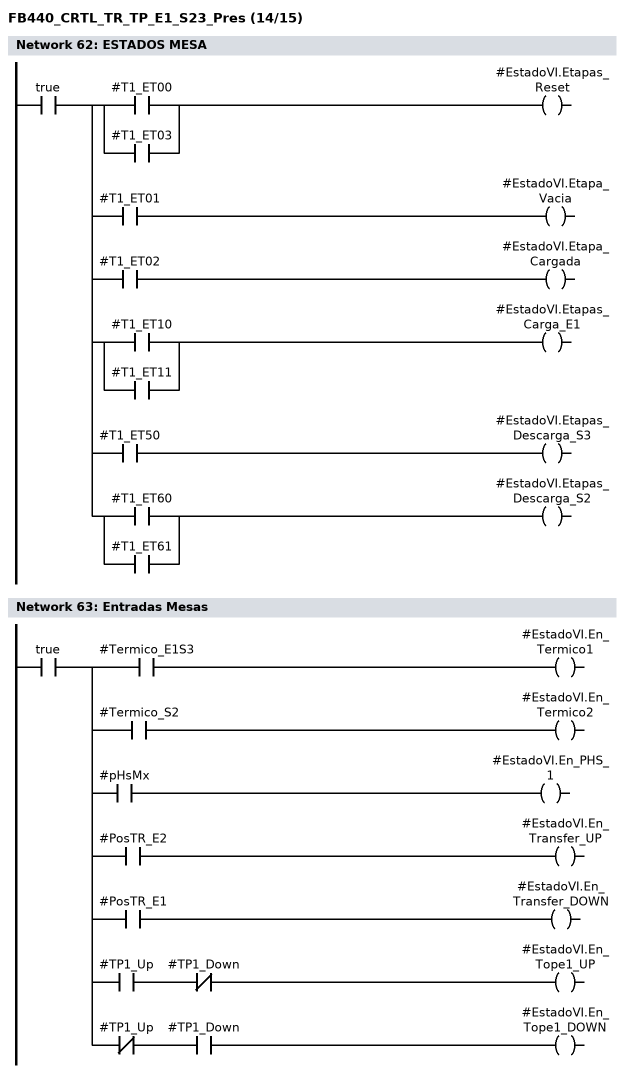
   RUNG wire#powerrail
      Contact( true )
      wire#w1
      Contact( #T1_ET00 )
      wire#w2
      Coil( #EstadoVI.Etapas_Reset )
   END_RUNG
   RUNG wire#w1
      Contact( #T1_ET03 )
   END_RUNG wire#w2
   RUNG wire#w1
      Contact( #T1_ET01 )
      Coil( #EstadoVI.Etapa_Vacia )
   END_RUNG
   RUNG wire#w1
      Contact( #T1_ET02 )
      Coil( #EstadoVI.Etapa_Cargada )
   END_RUNG
   RUNG wire#w1
      Contact( #T1_ET10 )
      wire#w3
      Coil( #EstadoVI.Etapas_Carga_E1 )
   END_RUNG
   RUNG wire#w1
      Contact( #T1_ET11 )
   END_RUNG wire#w3
   RUNG wire#w1
      Contact( #T1_ET50 )
      Coil( #EstadoVI.Etapas_Descarga_S3 )
   END_RUNG
   RUNG wire#w1
      Contact( #T1_ET60 )
      wire#w4
      Coil( #EstadoVI.Etapas_Descarga_S2 )
   END_RUNG
   RUNG wire#w1
      Contact( #T1_ET61 )
   END_RUNG wire#w4
   // the same network as SCL:
   #EstadoVI.Etapas_Reset := true AND (#T1_ET00 OR #T1_ET03);
   #EstadoVI.Etapa_Vacia := true AND #T1_ET01;
   #EstadoVI.Etapa_Cargada := true AND #T1_ET02;
   #EstadoVI.Etapas_Carga_E1 := true AND (#T1_ET10 OR #T1_ET11);
   #EstadoVI.Etapas_Descarga_S3 := true AND #T1_ET50;
   #EstadoVI.Etapas_Descarga_S2 := true AND (#T1_ET60 OR #T1_ET61);
END_REGION

REGION Network 63: Entradas Mesas
   RUNG wire#powerrail
      Contact( true )
      wire#w1
      Contact( #Termico_E1S3 )
      Coil( #EstadoVI.En_Termico1 )
   END_RUNG
   RUNG wire#w1
      Contact( #Termico_S2 )
      Coil( #EstadoVI.En_Termico2 )
   END_RUNG
   RUNG wire#w1
      Contact( #pHsMx )
      Coil( #EstadoVI.En_PHS_1 )
   END_RUNG
   RUNG wire#w1
      Contact( #PosTR_E2 )
      Coil( #EstadoVI.En_Transfer_UP )
   END_RUNG
   RUNG wire#w1
      Contact( #PosTR_E1 )
      Coil( #EstadoVI.En_Transfer_DOWN )
   END_RUNG
   RUNG wire#w1
      Contact( #TP1_Up )
      I_Contact( #TP1_Down )
      Coil( #EstadoVI.En_Tope1_UP )
   END_RUNG
   RUNG wire#w1
      I_Contact( #TP1_Up )
      Contact( #TP1_Down )
      Coil( #EstadoVI.En_Tope1_DOWN )
   END_RUNG
   // the same network as SCL:
   #EstadoVI.En_Termico1 := true AND #Termico_E1S3;
   #EstadoVI.En_Termico2 := true AND #Termico_S2;
   #EstadoVI.En_PHS_1 := true AND #pHsMx;
   #EstadoVI.En_Transfer_UP := true AND #PosTR_E2;
   #EstadoVI.En_Transfer_DOWN := true AND #PosTR_E1;
   #EstadoVI.En_Tope1_UP := true AND #TP1_Up AND NOT #TP1_Down;
   #EstadoVI.En_Tope1_DOWN := true AND NOT #TP1_Up AND #TP1_Down;
END_REGION

REGION Network 64: Salidas Mesas
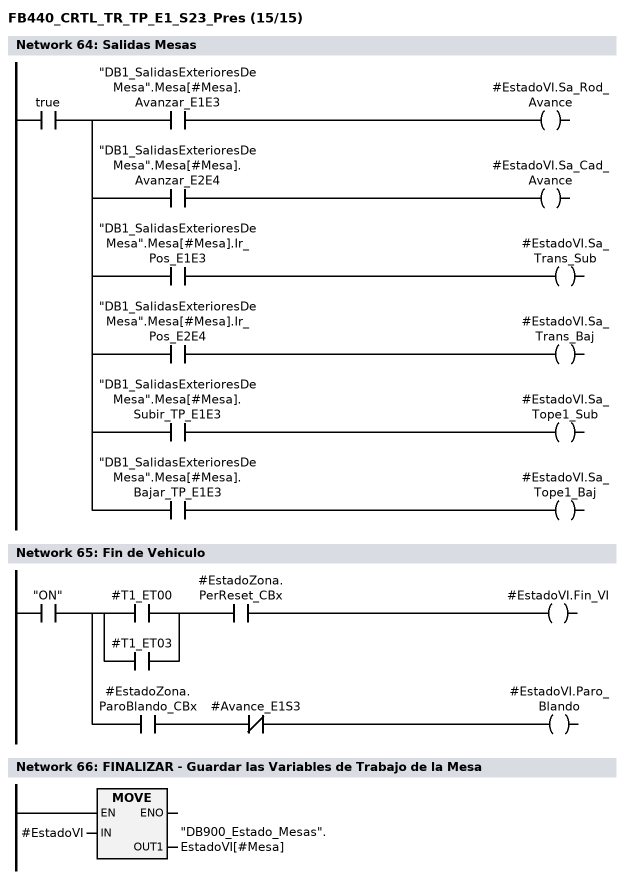
   RUNG wire#powerrail
      Contact( true )
      wire#w1
      Contact( "DB1_SalidasExterioresDeMesa".Mesa[#Mesa].Avanzar_E1E3 )
      Coil( #EstadoVI.Sa_Rod_Avance )
   END_RUNG
   RUNG wire#w1
      Contact( "DB1_SalidasExterioresDeMesa".Mesa[#Mesa].Avanzar_E2E4 )
      Coil( #EstadoVI.Sa_Cad_Avance )
   END_RUNG
   RUNG wire#w1
      Contact( "DB1_SalidasExterioresDeMesa".Mesa[#Mesa].Ir_Pos_E1E3 )
      Coil( #EstadoVI.Sa_Trans_Sub )
   END_RUNG
   RUNG wire#w1
      Contact( "DB1_SalidasExterioresDeMesa".Mesa[#Mesa].Ir_Pos_E2E4 )
      Coil( #EstadoVI.Sa_Trans_Baj )
   END_RUNG
   RUNG wire#w1
      Contact( "DB1_SalidasExterioresDeMesa".Mesa[#Mesa].Subir_TP_E1E3 )
      Coil( #EstadoVI.Sa_Tope1_Sub )
   END_RUNG
   RUNG wire#w1
      Contact( "DB1_SalidasExterioresDeMesa".Mesa[#Mesa].Bajar_TP_E1E3 )
      Coil( #EstadoVI.Sa_Tope1_Baj )
   END_RUNG
   // the same network as SCL:
   #EstadoVI.Sa_Rod_Avance := true AND "DB1_SalidasExterioresDeMesa".Mesa[#Mesa].Avanzar_E1E3;
   #EstadoVI.Sa_Cad_Avance := true AND "DB1_SalidasExterioresDeMesa".Mesa[#Mesa].Avanzar_E2E4;
   #EstadoVI.Sa_Trans_Sub := true AND "DB1_SalidasExterioresDeMesa".Mesa[#Mesa].Ir_Pos_E1E3;
   #EstadoVI.Sa_Trans_Baj := true AND "DB1_SalidasExterioresDeMesa".Mesa[#Mesa].Ir_Pos_E2E4;
   #EstadoVI.Sa_Tope1_Sub := true AND "DB1_SalidasExterioresDeMesa".Mesa[#Mesa].Subir_TP_E1E3;
   #EstadoVI.Sa_Tope1_Baj := true AND "DB1_SalidasExterioresDeMesa".Mesa[#Mesa].Bajar_TP_E1E3;
END_REGION

REGION Network 65: Fin de Vehiculo
   RUNG wire#powerrail
      Contact( "ON" )
      wire#w1
      Contact( #T1_ET00 )
      wire#w2
      Contact( #EstadoZona.PerReset_CBx )
      Coil( #EstadoVI.Fin_VI )
   END_RUNG
   RUNG wire#w1
      Contact( #T1_ET03 )
   END_RUNG wire#w2
   RUNG wire#w1
      Contact( #EstadoZona.ParoBlando_CBx )
      I_Contact( #Avance_E1S3 )
      Coil( #EstadoVI.Paro_Blando )
   END_RUNG
   // the same network as SCL:
   #EstadoVI.Fin_VI := "ON" AND (#T1_ET00 OR #T1_ET03) AND #EstadoZona.PerReset_CBx;
   #EstadoVI.Paro_Blando := "ON" AND #EstadoZona.ParoBlando_CBx AND NOT #Avance_E1S3;
END_REGION

REGION Network 66: FINALIZAR - Guardar las Variables de Trabajo de la Mesa
   RUNG wire#powerrail
      Move(in := #EstadoVI, out1 => "DB900_Estado_Mesas".EstadoVI[#Mesa])
   END_RUNG
   // the same network as SCL:
   "DB900_Estado_Mesas".EstadoVI[#Mesa] := #EstadoVI;
END_REGION
END_FUNCTION_BLOCK

FUNCTION_BLOCK "FB459_CRTL_TR_TP_E1_S2S3_Aus+ord"   // FB459, LAD
TITLE = Control del Ramal de Salidas
{ S7_Optimized_Access := 'FALSE' }
AUTHOR : TLigero
NAME : 20180827
VERSION : 3.4
// FECHA:    27/07/2011  AUTOR: C. MARCO
// INSTALACION: Eroski Laboratorio
// //////////////////////////////////
// // Registro Incidencias   ////////
// //////////////////////////////////
// FECHA:   AUTOR MODIFICACION: 
// DESCRIPCION:
// stored: AutoNumber false, SetENOAutomatically false
   VAR_INPUT
      Mesa : UInt;   // Número de mesa
      En_Tension : Bool;
      pHsMx_E1 : Bool;   // pHs DE AUSENCIA de la Mesa en E1
      pHsMx_S2 : Bool;   // pHs DE AUSENCIA de la Mesa en S2
      pHsMx_S3 : Bool;   // pHs DE AUSENCIA de la Mesa en S3
      TP1_Up : Bool;   // TP1 Arriba. E1 >> S3. si no hay tope poner ON
      TP1_Down : Bool;   // TP1 Abajo. E1 >> S3. si no hay tope poner ON
      PosTR_E1 : Bool;   // Posicion del TR en E1E3
      PosTR_E2 : Bool;   // Posicion del TR en E2E4
      Termico_E1S3 : Bool;   // Proteccion del Tx en E1E3
      Termico_S2 : Bool;   // Proteccion del Tx en E2E4
      Avance_E1S3 : Bool;   // Avance del Tx en E1E3
      Avance_S2 : Bool;   // Avance del Tx en E2E4
      PTF_Sal_M2 : Bool;   // S2 >> Mesa Siguiente PTF
      NXT_Avance_S2 : Bool;   // S2 >> Mesa Siguiente avanzando
      PTF_Sal_M3 : Bool;   // S3 >> Mesa Siguiente PTF
      NXT_Avance_S3 : Bool;   // S3 >> Mesa Siguiente avanzando
      F_EnvMens_Mx : Bool;   // Fin de Envio de Mensaje
      Mx_BloqActivo_S2 : Bool;   // Bloqueo Activo de la Mesa
      Mx_FlujoPrin_S2 : Bool;   // El flujo principal es Saliendo por S2
      AVTF_MAnt_Mx : Bool;   // E1 >> Mesa Anterior AVTF
      Habilitar_orden_JDT : Bool;   // El JDT tendrá el control del cruce con orden
      ValorOrden_S2 : Word := 16#81;   // Valor de la orden para salir por S2
      Num_Cruce : UInt;   // Número de cruce.
      DB_FIFO_Cruce : UInt := 213;   // DB de la FIFO de ordenes del cruce
      Long_FIFO_Cruce : UInt := 1;   // Longitut de la FIFO de ordenes del cruce
      MesaS2 : UInt;   // Número de mesa por S2
      MesaS3 : UInt;   // Número de mesa por S3
      V_CNT_ApHsMx_E1 : UDInt;   // Valor de Ausencia por E1 en ms
      V_CNT_ApHsMx_S2 : UDInt;   // Valor de Ausencia por S2 en ms
      V_CNT_ApHsMx_S3 : UDInt;   // Valor de Ausencia por S3 en ms
      V_Vaciado : UDInt := 10000;   // Valor de vaciado en ms
      V_Estabilizacion_carga : UDInt := 10;   // Temporizador para estabilizar la carga en ms
      V_TOut_Tx_Mx : UDInt := 5000;   // TimeOut de Atasco en ms
      V_TOut_TP : UDInt := 2000;   // TimeOut de Tope en ms
      V_TOut_TR : UDInt := 5000;   // TimeOut de Transfer en ms
   END_VAR
   VAR_OUTPUT
      P_EnvMens_PMx : Bool;   // Permiso de Enviar Mensaje de Presencia
      Etiqueta_Jdt : UDInt;   // Etiqueta que ha sido leida
      Orden_Ejecutada_Jdt : UInt;   // Orden que se ha ejecutado
      PTF_MAnt_Mx : Bool;   // E1 >> Mesa Anterior PTF
      AVTF_Sal_M2 : Bool;   // S2 >> Mesa Siguiente AVTF
      AVTF_Sal_M3 : Bool;   // S3 >> Mesa Siguiente descarga activa
   END_VAR
   VAR
      T1_ET00 : Bool;
      T1_ET01 : Bool;
      T1_ET02 : Bool;
      T1_ET2_JDT : Bool;
      T1_ET03 : Bool;
      T1_ET10 : Bool;
      T1_ET11 : Bool;
      T1_ET12 : Bool;
      T1_ET50 : Bool;
      T1_ET60 : Bool;
      T1_ET70 : Bool;
      T1_ET110 : Bool;
      T1_ET111 : Bool;
      T1_ET112 : Bool;
      Simul_Mx : Bool;
      FIFO_OK : Bool;
      TRANS_OK : Bool;
      O_Bloqueo : Bool;
      Err_Detec_PHS : Bool;
      FN_ET02 : Bool;
      MemFN_pHsE1 : Bool;
      MemFN_pHsS3 : Bool;
      MemFN_pHsS2 : Bool;
      MemAuxFN_pHsE1 : Bool;
      MemAuxFN_pHsS3 : Bool;
      MemAuxFN_pHsS2 : Bool;
      OK_TmpAusE1 : Bool;
      OK_TmpAusS3 : Bool;
      OK_TmpAusS2 : Bool;
      FP_ET2_JDT : Bool;
      FN_ET2_JDT : Bool;
      maux_fp_disparo : Bool;
      timVaciado_q : Bool;
      MA_Subir_TP_E1 : Bool;
      MA_Bajar_TP_E1 : Bool;
      TmpAus_E1 : UDInt;
      TmpAus_S2 : UDInt;
      TmpAus_S3 : UDInt;
      TOUT_Movimiento_transfer : UDInt;
      TIMVaciado : UDInt;
      T_Atasco : UDInt;
      T_estabilizacion : UDInt;
      Tout_tope : UDInt;
      TMP_En_Tension : UDInt;
      Datos_Scanner { S7_SetPoint := 'True'} : "ROUT_Orden_Fifo_Scanner";
   END_VAR
   VAR_TEMP
      EstadoZona : "EstadoZona";   // Estado de Zona de la Mesa
      EstadoVI : "EstadosMesa";   // Estado del Vehiculo Inteliguente de la Mesa
      ConfigFB : "UDT_ConfigFB";   // Configuracion de la FB de la Mesa
      O_Salir_S3 : Bool;
      O_Salir_S2 : Bool;
      O_Vaciar : Bool;
      Moti_ERRO : Bool;
      Moti_NENC : Bool;
      Moti_NORM : Bool;
      Moti_INIC : Bool;
      SalS3_JDT : Bool;
      SalS2_JDT : Bool;
      T_estabilizacion_Q : Bool;
      t_atasco_q : Bool;
      Tout_movimiento_transfer_q : Bool;
      Tout_tope_Q : Bool;
      ok_tension : Bool;
      Aux_W_Moti : Word;
      INT_ORDEN : UInt;
      Aux_W_Orden : Word;
      I_Ord_Filtrada : UInt;
      I_V_Ord_Entrar : UInt;
   END_VAR
   VAR_TEMP   // added for the SCL form of the ladder/FBD networks
      _w1 : Bool;
      _w2 : Bool;
      _w3 : Bool;
      _w4 : Bool;
      _w5 : Bool;
      _w6 : Bool;
   END_VAR
BEGIN

REGION Network 1: INICIALIZAR - Recoger las Variables de Estado de la Mesa
   // Se recoge - Estado_CBx
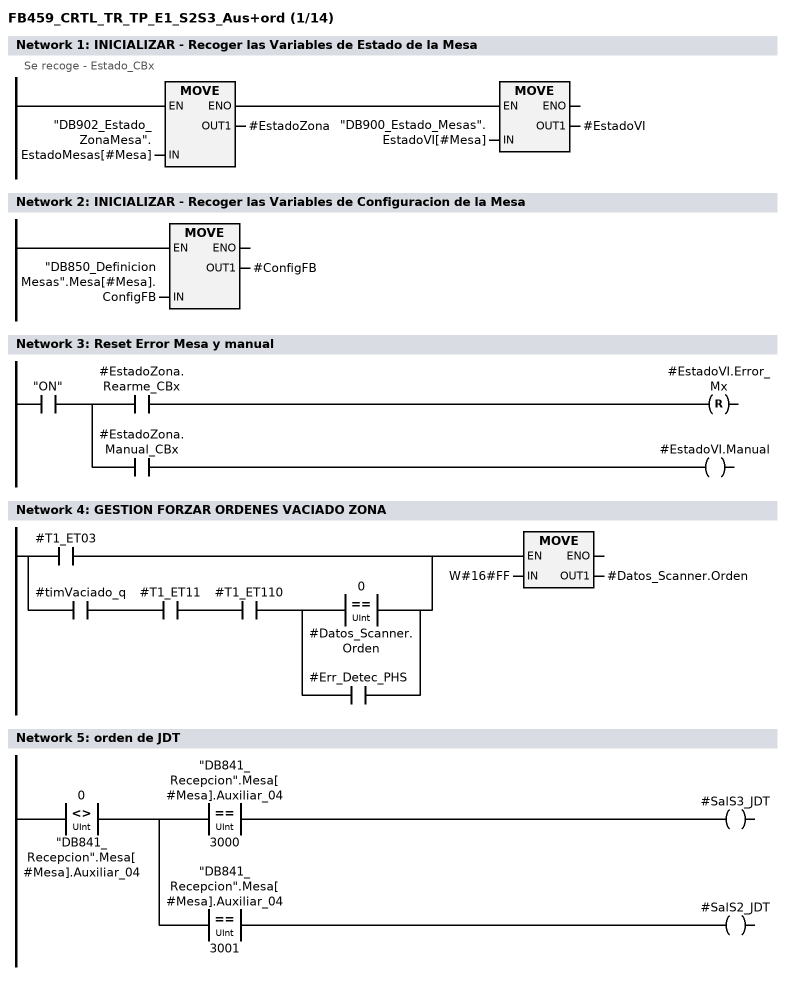
   RUNG wire#powerrail
      Move(in := "DB902_Estado_ZonaMesa".EstadoMesas[#Mesa], out1 => #EstadoZona)
      Move(in := "DB900_Estado_Mesas".EstadoVI[#Mesa], out1 => #EstadoVI)
   END_RUNG
   // the same network as SCL:
   #EstadoZona := "DB902_Estado_ZonaMesa".EstadoMesas[#Mesa];
   #EstadoVI := "DB900_Estado_Mesas".EstadoVI[#Mesa];
END_REGION

REGION Network 2: INICIALIZAR - Recoger las Variables de Configuracion de la Mesa
   RUNG wire#powerrail
      Move(in := "DB850_DefinicionMesas".Mesa[#Mesa].ConfigFB, out1 => #ConfigFB)
   END_RUNG
   // the same network as SCL:
   #ConfigFB := "DB850_DefinicionMesas".Mesa[#Mesa].ConfigFB;
END_REGION

REGION Network 3: Reset Error Mesa y manual
   RUNG wire#powerrail
      Contact( "ON" )
      wire#w1
      Contact( #EstadoZona.Rearme_CBx )
      R_Coil( #EstadoVI.Error_Mx )
   END_RUNG
   RUNG wire#w1
      Contact( #EstadoZona.Manual_CBx )
      Coil( #EstadoVI.Manual )
   END_RUNG
   // the same network as SCL:
   IF "ON" AND #EstadoZona.Rearme_CBx THEN #EstadoVI.Error_Mx := FALSE; END_IF;
   #EstadoVI.Manual := "ON" AND #EstadoZona.Manual_CBx;
END_REGION

REGION Network 4: GESTION FORZAR ORDENES VACIADO ZONA
   RUNG wire#powerrail
      Contact( #T1_ET03 )
      wire#w1
      { S7_GenerateENO := "TRUE" } Move(in := W#16#FF, out1 => #Datos_Scanner.Orden)
   END_RUNG
   RUNG wire#powerrail
      Contact( #timVaciado_q )
      Contact( #T1_ET11 )
      Contact( #T1_ET110 )
      wire#w2
      { S7_Templates := "SrcType := UInt" } EQ_Contact(in1 := 0, in2 := #Datos_Scanner.Orden)
   END_RUNG wire#w1
   RUNG wire#w2
      Contact( #Err_Detec_PHS )
   END_RUNG wire#w1
   // the same network as SCL:
   IF #T1_ET03 OR (#timVaciado_q AND #T1_ET11 AND #T1_ET110 AND ((0 = #Datos_Scanner.Orden) OR #Err_Detec_PHS)) THEN
       #Datos_Scanner.Orden := W#16#FF;
   END_IF;
END_REGION

REGION Network 5: orden de JDT
   RUNG wire#powerrail
      { S7_Templates := "SrcType := UInt" } NE_Contact(in1 := 0, in2 := "DB841_Recepcion".Mesa[#Mesa].Auxiliar_04)
      wire#w1
      { S7_Templates := "SrcType := UInt" } EQ_Contact(in1 := "DB841_Recepcion".Mesa[#Mesa].Auxiliar_04, in2 := 3000)
      Coil( #SalS3_JDT )
   END_RUNG
   RUNG wire#w1
      { S7_Templates := "SrcType := UInt" } EQ_Contact(in1 := "DB841_Recepcion".Mesa[#Mesa].Auxiliar_04, in2 := 3001)
      Coil( #SalS2_JDT )
   END_RUNG
   // the same network as SCL:
   #_w1 := 0 <> "DB841_Recepcion".Mesa[#Mesa].Auxiliar_04;
   #SalS3_JDT := #_w1 AND ("DB841_Recepcion".Mesa[#Mesa].Auxiliar_04 = 3000);
   #SalS2_JDT := #_w1 AND ("DB841_Recepcion".Mesa[#Mesa].Auxiliar_04 = 3001);
END_REGION

REGION Network 6: Extraer orden
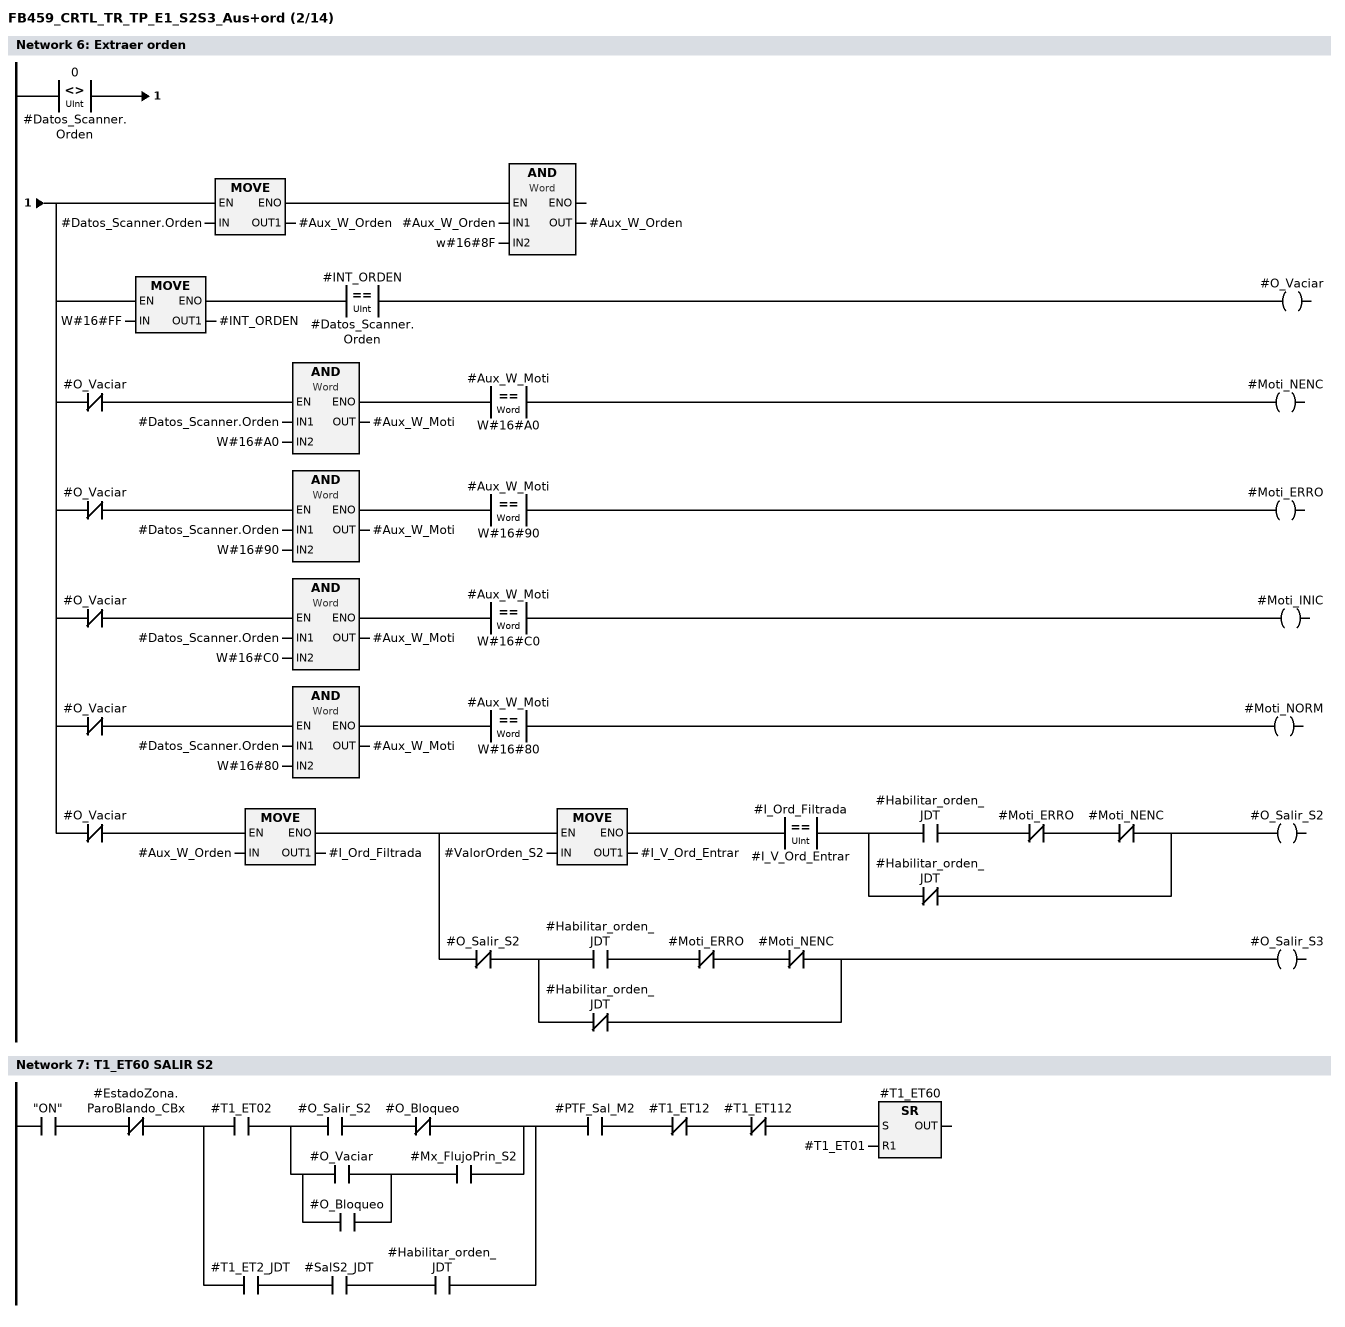
   RUNG wire#powerrail
      { S7_Templates := "SrcType := UInt" } NE_Contact(in1 := 0, in2 := #Datos_Scanner.Orden)
      wire#w1
      { S7_GenerateENO := "TRUE" } Move(in := #Datos_Scanner.Orden, out1 => #Aux_W_Orden)
      { S7_Templates := "SrcType := Word"; S7_GenerateENO := "TRUE" } And(in1 := #Aux_W_Orden, in2 := w#16#8F, out => #Aux_W_Orden)
   END_RUNG
   RUNG wire#w1
      { S7_GenerateENO := "TRUE" } Move(in := W#16#FF, out1 => #INT_ORDEN)
      { S7_Templates := "SrcType := UInt" } EQ_Contact(in1 := #INT_ORDEN, in2 := #Datos_Scanner.Orden)
      Coil( #O_Vaciar )
   END_RUNG
   RUNG wire#w1
      I_Contact( #O_Vaciar )
      { S7_Templates := "SrcType := Word"; S7_GenerateENO := "TRUE" } And(in1 := #Datos_Scanner.Orden, in2 := W#16#A0, out => #Aux_W_Moti)
      { S7_Templates := "SrcType := Word" } EQ_Contact(in1 := #Aux_W_Moti, in2 := W#16#A0)
      Coil( #Moti_NENC )
   END_RUNG
   RUNG wire#w1
      I_Contact( #O_Vaciar )
      { S7_Templates := "SrcType := Word"; S7_GenerateENO := "TRUE" } And(in1 := #Datos_Scanner.Orden, in2 := W#16#90, out => #Aux_W_Moti)
      { S7_Templates := "SrcType := Word" } EQ_Contact(in1 := #Aux_W_Moti, in2 := W#16#90)
      Coil( #Moti_ERRO )
   END_RUNG
   RUNG wire#w1
      I_Contact( #O_Vaciar )
      { S7_Templates := "SrcType := Word"; S7_GenerateENO := "TRUE" } And(in1 := #Datos_Scanner.Orden, in2 := W#16#C0, out => #Aux_W_Moti)
      { S7_Templates := "SrcType := Word" } EQ_Contact(in1 := #Aux_W_Moti, in2 := W#16#C0)
      Coil( #Moti_INIC )
   END_RUNG
   RUNG wire#w1
      I_Contact( #O_Vaciar )
      { S7_Templates := "SrcType := Word"; S7_GenerateENO := "TRUE" } And(in1 := #Datos_Scanner.Orden, in2 := W#16#80, out => #Aux_W_Moti)
      { S7_Templates := "SrcType := Word" } EQ_Contact(in1 := #Aux_W_Moti, in2 := W#16#80)
      Coil( #Moti_NORM )
   END_RUNG
   RUNG wire#w1
      I_Contact( #O_Vaciar )
      { S7_GenerateENO := "TRUE" } Move(in := #Aux_W_Orden, out1 => #I_Ord_Filtrada)
      wire#w2
      { S7_GenerateENO := "TRUE" } Move(in := #ValorOrden_S2, out1 => #I_V_Ord_Entrar)
      { S7_Templates := "SrcType := UInt" } EQ_Contact(in1 := #I_Ord_Filtrada, in2 := #I_V_Ord_Entrar)
      wire#w3
      Contact( #Habilitar_orden_JDT )
      I_Contact( #Moti_ERRO )
      I_Contact( #Moti_NENC )
      wire#w4
      Coil( #O_Salir_S2 )
   END_RUNG
   RUNG wire#w3
      I_Contact( #Habilitar_orden_JDT )
   END_RUNG wire#w4
   RUNG wire#w2
      I_Contact( #O_Salir_S2 )
      wire#w5
      Contact( #Habilitar_orden_JDT )
      I_Contact( #Moti_ERRO )
      I_Contact( #Moti_NENC )
      wire#w6
      Coil( #O_Salir_S3 )
   END_RUNG
   RUNG wire#w5
      I_Contact( #Habilitar_orden_JDT )
   END_RUNG wire#w6
   // the same network as SCL:
   // ENO of a box is taken as its EN; it also drops when the box reports an error
   #_w1 := 0 <> #Datos_Scanner.Orden;
   IF #_w1 THEN
       #Aux_W_Orden := #Datos_Scanner.Orden;
       #Aux_W_Orden := #Aux_W_Orden AND w#16#8F;
       #INT_ORDEN := W#16#FF;
   END_IF;
   #O_Vaciar := #_w1 AND (#INT_ORDEN = #Datos_Scanner.Orden);
   #_w2 := #_w1 AND NOT #O_Vaciar;
   IF #_w2 THEN #Aux_W_Moti := #Datos_Scanner.Orden AND W#16#A0; END_IF;
   #Moti_NENC := #_w2 AND (#Aux_W_Moti = W#16#A0);
   #_w3 := #_w1 AND NOT #O_Vaciar;
   IF #_w3 THEN #Aux_W_Moti := #Datos_Scanner.Orden AND W#16#90; END_IF;
   #Moti_ERRO := #_w3 AND (#Aux_W_Moti = W#16#90);
   #_w4 := #_w1 AND NOT #O_Vaciar;
   IF #_w4 THEN #Aux_W_Moti := #Datos_Scanner.Orden AND W#16#C0; END_IF;
   #Moti_INIC := #_w4 AND (#Aux_W_Moti = W#16#C0);
   #_w5 := #_w1 AND NOT #O_Vaciar;
   IF #_w5 THEN #Aux_W_Moti := #Datos_Scanner.Orden AND W#16#80; END_IF;
   #Moti_NORM := #_w5 AND (#Aux_W_Moti = W#16#80);
   #_w6 := #_w1 AND NOT #O_Vaciar;
   IF #_w6 THEN
       #I_Ord_Filtrada := #Aux_W_Orden;
       #I_V_Ord_Entrar := #ValorOrden_S2;
   END_IF;
   #O_Salir_S2 := #_w6 AND (#I_Ord_Filtrada = #I_V_Ord_Entrar) AND ((#Habilitar_orden_JDT AND NOT #Moti_ERRO AND NOT #Moti_NENC) OR NOT #Habilitar_orden_JDT);
   #O_Salir_S3 := #_w6 AND NOT #O_Salir_S2 AND ((#Habilitar_orden_JDT AND NOT #Moti_ERRO AND NOT #Moti_NENC) OR NOT #Habilitar_orden_JDT);
END_REGION

REGION Network 7: T1_ET60 SALIR S2
   RUNG wire#powerrail
      Contact( "ON" )
      I_Contact( #EstadoZona.ParoBlando_CBx )
      wire#w1
      Contact( #T1_ET02 )
      wire#w2
      Contact( #O_Salir_S2 )
      I_Contact( #O_Bloqueo )
      wire#w3
      Contact( #PTF_Sal_M2 )
      I_Contact( #T1_ET12 )
      I_Contact( #T1_ET112 )
      S_SR(operand := #T1_ET60, r1 := #T1_ET01)
   END_RUNG
   RUNG wire#w2
      Contact( #O_Vaciar )
      wire#w4
      Contact( #Mx_FlujoPrin_S2 )
   END_RUNG wire#w3
   RUNG wire#w2
      Contact( #O_Bloqueo )
   END_RUNG wire#w4
   RUNG wire#w1
      Contact( #T1_ET2_JDT )
      Contact( #SalS2_JDT )
      Contact( #Habilitar_orden_JDT )
   END_RUNG wire#w3
   // the same network as SCL:
   IF "ON" AND NOT #EstadoZona.ParoBlando_CBx AND ((#T1_ET02 AND ((#O_Salir_S2 AND NOT #O_Bloqueo) OR ((#O_Vaciar OR #O_Bloqueo) AND #Mx_FlujoPrin_S2))) OR (#T1_ET2_JDT AND #SalS2_JDT AND #Habilitar_orden_JDT)) AND #PTF_Sal_M2 AND NOT #T1_ET12 AND NOT #T1_ET112 THEN
       #T1_ET60 := TRUE;   // SR flip-flop
   END_IF;
   IF #T1_ET01 THEN #T1_ET60 := FALSE; END_IF;
END_REGION

REGION Network 8: T1_ET50 SALIR S3
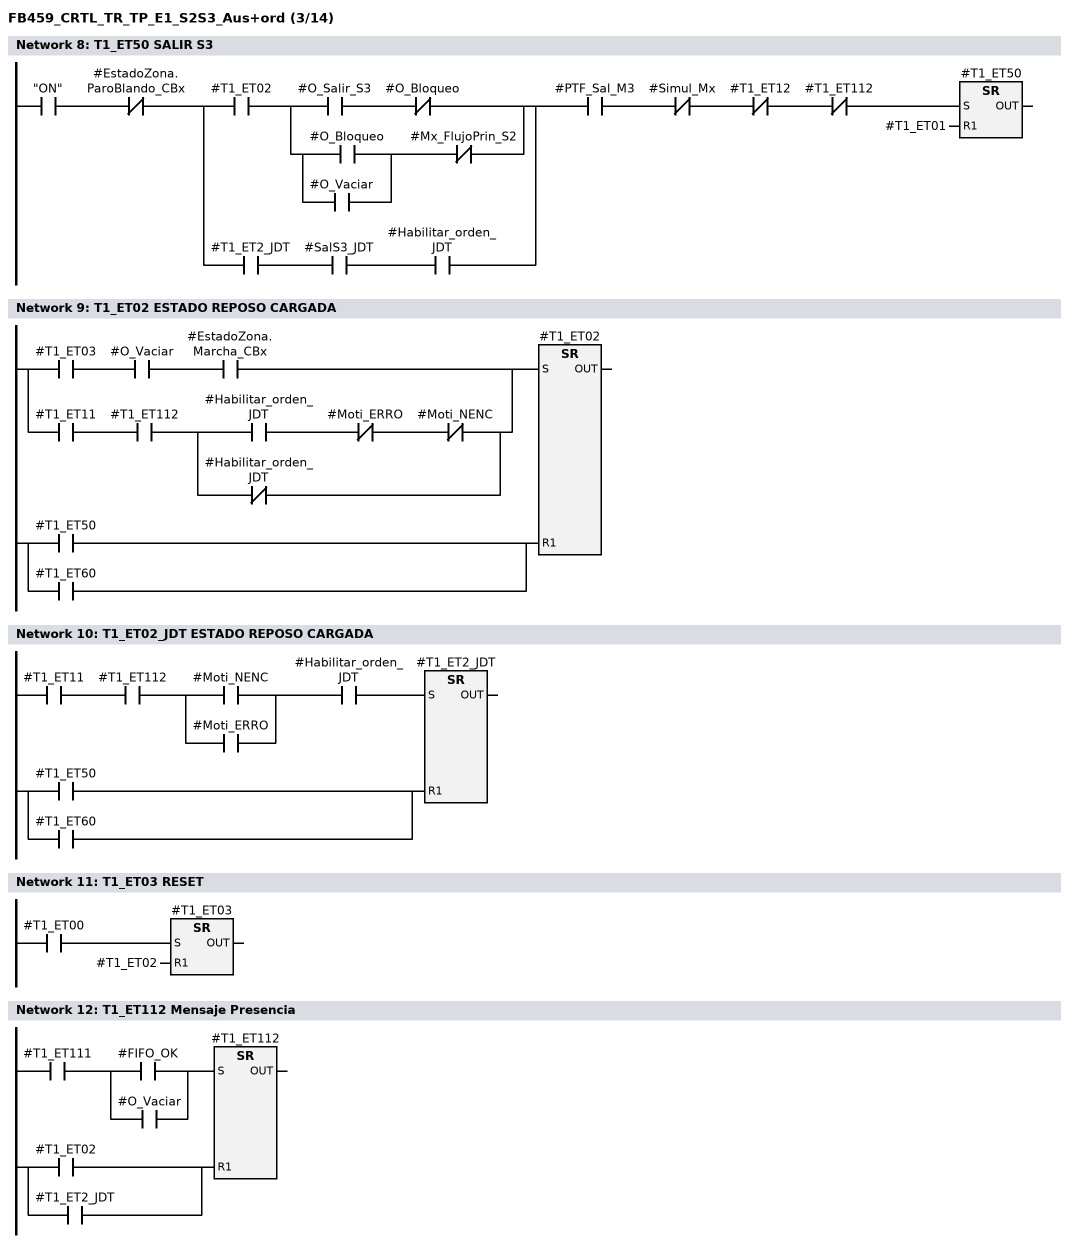
   RUNG wire#powerrail
      Contact( "ON" )
      I_Contact( #EstadoZona.ParoBlando_CBx )
      wire#w1
      Contact( #T1_ET02 )
      wire#w2
      Contact( #O_Salir_S3 )
      I_Contact( #O_Bloqueo )
      wire#w3
      Contact( #PTF_Sal_M3 )
      I_Contact( #Simul_Mx )
      I_Contact( #T1_ET12 )
      I_Contact( #T1_ET112 )
      S_SR(operand := #T1_ET50, r1 := #T1_ET01)
   END_RUNG
   RUNG wire#w2
      Contact( #O_Bloqueo )
      wire#w4
      I_Contact( #Mx_FlujoPrin_S2 )
   END_RUNG wire#w3
   RUNG wire#w2
      Contact( #O_Vaciar )
   END_RUNG wire#w4
   RUNG wire#w1
      Contact( #T1_ET2_JDT )
      Contact( #SalS3_JDT )
      Contact( #Habilitar_orden_JDT )
   END_RUNG wire#w3
   // the same network as SCL:
   IF "ON" AND NOT #EstadoZona.ParoBlando_CBx AND ((#T1_ET02 AND ((#O_Salir_S3 AND NOT #O_Bloqueo) OR ((#O_Bloqueo OR #O_Vaciar) AND NOT #Mx_FlujoPrin_S2))) OR (#T1_ET2_JDT AND #SalS3_JDT AND #Habilitar_orden_JDT)) AND #PTF_Sal_M3 AND NOT #Simul_Mx AND NOT #T1_ET12 AND NOT #T1_ET112 THEN
       #T1_ET50 := TRUE;   // SR flip-flop
   END_IF;
   IF #T1_ET01 THEN #T1_ET50 := FALSE; END_IF;
END_REGION

REGION Network 9: T1_ET02 ESTADO REPOSO CARGADA
   RUNG wire#powerrail
      Contact( #T1_ET03 )
      Contact( #O_Vaciar )
      Contact( #EstadoZona.Marcha_CBx )
      wire#w1
      S_SR(operand := #T1_ET02, r1 := wire#w3)
   END_RUNG
   RUNG wire#powerrail
      Contact( #T1_ET11 )
      Contact( #T1_ET112 )
      wire#w2
      Contact( #Habilitar_orden_JDT )
      I_Contact( #Moti_ERRO )
      I_Contact( #Moti_NENC )
   END_RUNG wire#w1
   RUNG wire#w2
      I_Contact( #Habilitar_orden_JDT )
   END_RUNG wire#w1
   RUNG wire#powerrail
      Contact( #T1_ET50 )
   END_RUNG wire#w3
   RUNG wire#powerrail
      Contact( #T1_ET60 )
   END_RUNG wire#w3
   // the same network as SCL:
   IF (#T1_ET03 AND #O_Vaciar AND #EstadoZona.Marcha_CBx) OR (#T1_ET11 AND #T1_ET112 AND ((#Habilitar_orden_JDT AND NOT #Moti_ERRO AND NOT #Moti_NENC) OR NOT #Habilitar_orden_JDT)) THEN
       #T1_ET02 := TRUE;   // SR flip-flop
   END_IF;
   IF #T1_ET50 OR #T1_ET60 THEN #T1_ET02 := FALSE; END_IF;
END_REGION

REGION Network 10: T1_ET02_JDT ESTADO REPOSO CARGADA
   RUNG wire#powerrail
      Contact( #T1_ET11 )
      Contact( #T1_ET112 )
      wire#w1
      Contact( #Moti_NENC )
      wire#w2
      Contact( #Habilitar_orden_JDT )
      S_SR(operand := #T1_ET2_JDT, r1 := wire#w3)
   END_RUNG
   RUNG wire#w1
      Contact( #Moti_ERRO )
   END_RUNG wire#w2
   RUNG wire#powerrail
      Contact( #T1_ET50 )
   END_RUNG wire#w3
   RUNG wire#powerrail
      Contact( #T1_ET60 )
   END_RUNG wire#w3
   // the same network as SCL:
   IF #T1_ET11 AND #T1_ET112 AND (#Moti_NENC OR #Moti_ERRO) AND #Habilitar_orden_JDT THEN
       #T1_ET2_JDT := TRUE;   // SR flip-flop
   END_IF;
   IF #T1_ET50 OR #T1_ET60 THEN #T1_ET2_JDT := FALSE; END_IF;
END_REGION

REGION Network 11: T1_ET03 RESET
   RUNG wire#powerrail
      Contact( #T1_ET00 )
      S_SR(operand := #T1_ET03, r1 := #T1_ET02)
   END_RUNG
   // the same network as SCL:
   IF #T1_ET00 THEN
       #T1_ET03 := TRUE;   // SR flip-flop
   END_IF;
   IF #T1_ET02 THEN #T1_ET03 := FALSE; END_IF;
END_REGION

REGION Network 12: T1_ET112 Mensaje Presencia
   RUNG wire#powerrail
      Contact( #T1_ET111 )
      wire#w1
      Contact( #FIFO_OK )
      wire#w2
      S_SR(operand := #T1_ET112, r1 := wire#w3)
   END_RUNG
   RUNG wire#w1
      Contact( #O_Vaciar )
   END_RUNG wire#w2
   RUNG wire#powerrail
      Contact( #T1_ET02 )
   END_RUNG wire#w3
   RUNG wire#powerrail
      Contact( #T1_ET2_JDT )
   END_RUNG wire#w3
   // the same network as SCL:
   IF #T1_ET111 AND (#FIFO_OK OR #O_Vaciar) THEN
       #T1_ET112 := TRUE;   // SR flip-flop
   END_IF;
   IF #T1_ET02 OR #T1_ET2_JDT THEN #T1_ET112 := FALSE; END_IF;
END_REGION

REGION Network 13: T1_ET111 Mensaje Presencia
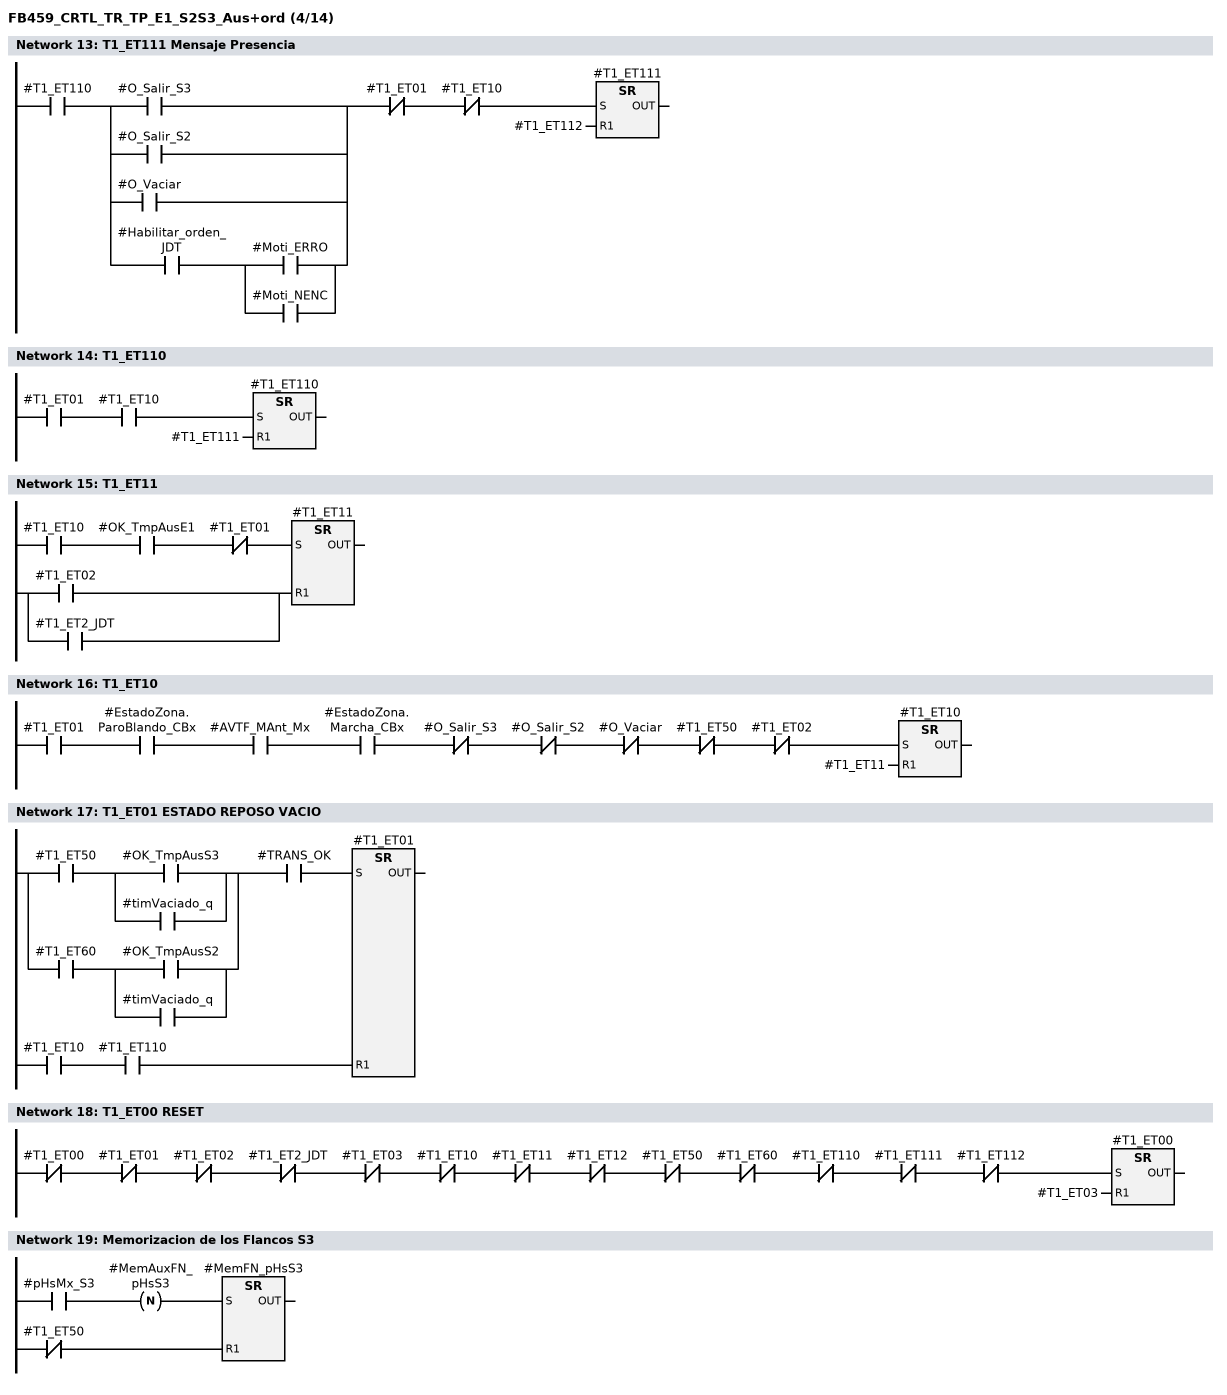
   RUNG wire#powerrail
      Contact( #T1_ET110 )
      wire#w1
      Contact( #O_Salir_S3 )
      wire#w2
      I_Contact( #T1_ET01 )
      I_Contact( #T1_ET10 )
      S_SR(operand := #T1_ET111, r1 := #T1_ET112)
   END_RUNG
   RUNG wire#w1
      Contact( #O_Salir_S2 )
   END_RUNG wire#w2
   RUNG wire#w1
      Contact( #O_Vaciar )
   END_RUNG wire#w2
   RUNG wire#w1
      Contact( #Habilitar_orden_JDT )
      wire#w3
      Contact( #Moti_ERRO )
   END_RUNG wire#w2
   RUNG wire#w3
      Contact( #Moti_NENC )
   END_RUNG wire#w2
   // the same network as SCL:
   IF #T1_ET110 AND (#O_Salir_S3 OR #O_Salir_S2 OR #O_Vaciar OR (#Habilitar_orden_JDT AND (#Moti_ERRO OR #Moti_NENC))) AND NOT #T1_ET01 AND NOT #T1_ET10 THEN
       #T1_ET111 := TRUE;   // SR flip-flop
   END_IF;
   IF #T1_ET112 THEN #T1_ET111 := FALSE; END_IF;
END_REGION

REGION Network 14: T1_ET110
   RUNG wire#powerrail
      Contact( #T1_ET01 )
      Contact( #T1_ET10 )
      S_SR(operand := #T1_ET110, r1 := #T1_ET111)
   END_RUNG
   // the same network as SCL:
   IF #T1_ET01 AND #T1_ET10 THEN
       #T1_ET110 := TRUE;   // SR flip-flop
   END_IF;
   IF #T1_ET111 THEN #T1_ET110 := FALSE; END_IF;
END_REGION

REGION Network 15: T1_ET11
   RUNG wire#powerrail
      Contact( #T1_ET10 )
      Contact( #OK_TmpAusE1 )
      I_Contact( #T1_ET01 )
      S_SR(operand := #T1_ET11, r1 := wire#w1)
   END_RUNG
   RUNG wire#powerrail
      Contact( #T1_ET02 )
   END_RUNG wire#w1
   RUNG wire#powerrail
      Contact( #T1_ET2_JDT )
   END_RUNG wire#w1
   // the same network as SCL:
   IF #T1_ET10 AND #OK_TmpAusE1 AND NOT #T1_ET01 THEN
       #T1_ET11 := TRUE;   // SR flip-flop
   END_IF;
   IF #T1_ET02 OR #T1_ET2_JDT THEN #T1_ET11 := FALSE; END_IF;
END_REGION

REGION Network 16: T1_ET10
   RUNG wire#powerrail
      Contact( #T1_ET01 )
      Contact( #EstadoZona.ParoBlando_CBx )
      Contact( #AVTF_MAnt_Mx )
      Contact( #EstadoZona.Marcha_CBx )
      I_Contact( #O_Salir_S3 )
      I_Contact( #O_Salir_S2 )
      I_Contact( #O_Vaciar )
      I_Contact( #T1_ET50 )
      I_Contact( #T1_ET02 )
      S_SR(operand := #T1_ET10, r1 := #T1_ET11)
   END_RUNG
   // the same network as SCL:
   IF #T1_ET01 AND #EstadoZona.ParoBlando_CBx AND #AVTF_MAnt_Mx AND #EstadoZona.Marcha_CBx AND NOT #O_Salir_S3 AND NOT #O_Salir_S2 AND NOT #O_Vaciar AND NOT #T1_ET50 AND NOT #T1_ET02 THEN
       #T1_ET10 := TRUE;   // SR flip-flop
   END_IF;
   IF #T1_ET11 THEN #T1_ET10 := FALSE; END_IF;
END_REGION

REGION Network 17: T1_ET01 ESTADO REPOSO VACIO
   RUNG wire#powerrail
      Contact( #T1_ET50 )
      wire#w1
      Contact( #OK_TmpAusS3 )
      wire#w2
      Contact( #TRANS_OK )
      S_SR(operand := #T1_ET01, r1 := wire#w4)
   END_RUNG
   RUNG wire#w1
      Contact( #timVaciado_q )
   END_RUNG wire#w2
   RUNG wire#powerrail
      Contact( #T1_ET60 )
      wire#w3
      Contact( #OK_TmpAusS2 )
   END_RUNG wire#w2
   RUNG wire#w3
      Contact( #timVaciado_q )
   END_RUNG wire#w2
   RUNG wire#powerrail
      Contact( #T1_ET10 )
      Contact( #T1_ET110 )
   END_RUNG wire#w4
   // the same network as SCL:
   IF ((#T1_ET50 AND (#OK_TmpAusS3 OR #timVaciado_q)) OR (#T1_ET60 AND (#OK_TmpAusS2 OR #timVaciado_q))) AND #TRANS_OK THEN
       #T1_ET01 := TRUE;   // SR flip-flop
   END_IF;
   IF #T1_ET10 AND #T1_ET110 THEN #T1_ET01 := FALSE; END_IF;
END_REGION

REGION Network 18: T1_ET00 RESET
   RUNG wire#powerrail
      I_Contact( #T1_ET00 )
      I_Contact( #T1_ET01 )
      I_Contact( #T1_ET02 )
      I_Contact( #T1_ET2_JDT )
      I_Contact( #T1_ET03 )
      I_Contact( #T1_ET10 )
      I_Contact( #T1_ET11 )
      I_Contact( #T1_ET12 )
      I_Contact( #T1_ET50 )
      I_Contact( #T1_ET60 )
      I_Contact( #T1_ET110 )
      I_Contact( #T1_ET111 )
      I_Contact( #T1_ET112 )
      S_SR(operand := #T1_ET00, r1 := #T1_ET03)
   END_RUNG
   // the same network as SCL:
   IF NOT #T1_ET00 AND NOT #T1_ET01 AND NOT #T1_ET02 AND NOT #T1_ET2_JDT AND NOT #T1_ET03 AND NOT #T1_ET10 AND NOT #T1_ET11 AND NOT #T1_ET12 AND NOT #T1_ET50 AND NOT #T1_ET60 AND NOT #T1_ET110 AND NOT #T1_ET111 AND NOT #T1_ET112 THEN
       #T1_ET00 := TRUE;   // SR flip-flop
   END_IF;
   IF #T1_ET03 THEN #T1_ET00 := FALSE; END_IF;
END_REGION

REGION Network 19: Memorizacion de los Flancos S3
   RUNG wire#powerrail
      Contact( #pHsMx_S3 )
      N_Trig( #MemAuxFN_pHsS3 )
      S_SR(operand := #MemFN_pHsS3, r1 := wire#w1)
   END_RUNG
   RUNG wire#powerrail
      I_Contact( #T1_ET50 )
   END_RUNG wire#w1
   // the same network as SCL:
   #_w1 := NOT #pHsMx_S3 AND #MemAuxFN_pHsS3;   // falling edge
   #MemAuxFN_pHsS3 := #pHsMx_S3;
   IF #_w1 THEN
       #MemFN_pHsS3 := TRUE;   // SR flip-flop
   END_IF;
   IF NOT #T1_ET50 THEN #MemFN_pHsS3 := FALSE; END_IF;
END_REGION

REGION Network 20: Memorizacion de los Flancos S2
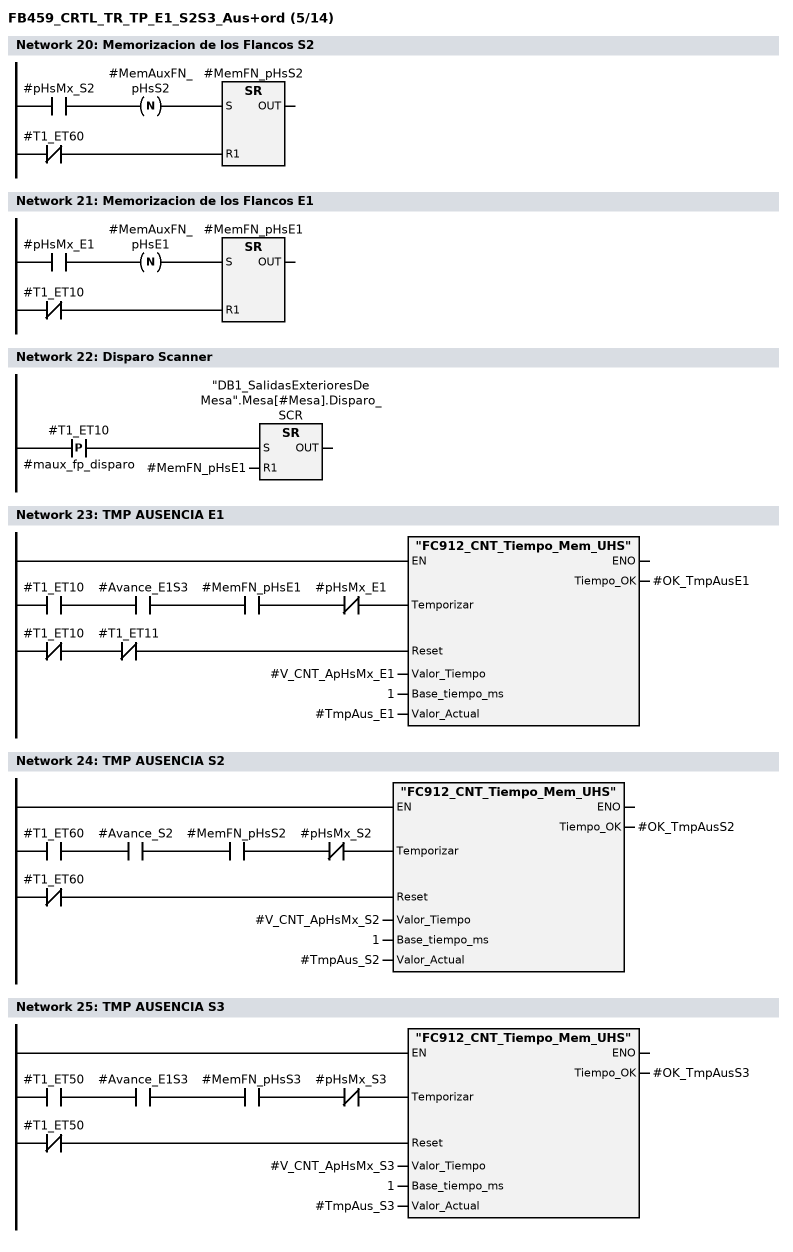
   RUNG wire#powerrail
      Contact( #pHsMx_S2 )
      N_Trig( #MemAuxFN_pHsS2 )
      S_SR(operand := #MemFN_pHsS2, r1 := wire#w1)
   END_RUNG
   RUNG wire#powerrail
      I_Contact( #T1_ET60 )
   END_RUNG wire#w1
   // the same network as SCL:
   #_w1 := NOT #pHsMx_S2 AND #MemAuxFN_pHsS2;   // falling edge
   #MemAuxFN_pHsS2 := #pHsMx_S2;
   IF #_w1 THEN
       #MemFN_pHsS2 := TRUE;   // SR flip-flop
   END_IF;
   IF NOT #T1_ET60 THEN #MemFN_pHsS2 := FALSE; END_IF;
END_REGION

REGION Network 21: Memorizacion de los Flancos E1
   RUNG wire#powerrail
      Contact( #pHsMx_E1 )
      N_Trig( #MemAuxFN_pHsE1 )
      S_SR(operand := #MemFN_pHsE1, r1 := wire#w1)
   END_RUNG
   RUNG wire#powerrail
      I_Contact( #T1_ET10 )
   END_RUNG wire#w1
   // the same network as SCL:
   #_w1 := NOT #pHsMx_E1 AND #MemAuxFN_pHsE1;   // falling edge
   #MemAuxFN_pHsE1 := #pHsMx_E1;
   IF #_w1 THEN
       #MemFN_pHsE1 := TRUE;   // SR flip-flop
   END_IF;
   IF NOT #T1_ET10 THEN #MemFN_pHsE1 := FALSE; END_IF;
END_REGION

REGION Network 22: Disparo Scanner
   RUNG wire#powerrail
      P_Contact(operand := #T1_ET10, bit := #maux_fp_disparo)
      S_SR(operand := "DB1_SalidasExterioresDeMesa".Mesa[#Mesa].Disparo_SCR, r1 := #MemFN_pHsE1)
   END_RUNG
   // the same network as SCL:
   #_w1 := #T1_ET10 AND NOT #maux_fp_disparo;   // rising edge of #T1_ET10
   #maux_fp_disparo := #T1_ET10;
   IF #_w1 THEN
       "DB1_SalidasExterioresDeMesa".Mesa[#Mesa].Disparo_SCR := TRUE;   // SR flip-flop
   END_IF;
   IF #MemFN_pHsE1 THEN "DB1_SalidasExterioresDeMesa".Mesa[#Mesa].Disparo_SCR := FALSE; END_IF;
END_REGION

REGION Network 23: TMP AUSENCIA E1
   RUNG wire#powerrail
      "FC912_CNT_Tiempo_Mem_UHS"(Temporizar := wire#w1, Reset := wire#w2, Valor_Tiempo := #V_CNT_ApHsMx_E1, Base_tiempo_ms := 1, Valor_Actual := #TmpAus_E1, Tiempo_OK => #OK_TmpAusE1)
   END_RUNG
   RUNG wire#powerrail
      Contact( #T1_ET10 )
      Contact( #Avance_E1S3 )
      Contact( #MemFN_pHsE1 )
      I_Contact( #pHsMx_E1 )
   END_RUNG wire#w1
   RUNG wire#powerrail
      I_Contact( #T1_ET10 )
      I_Contact( #T1_ET11 )
   END_RUNG wire#w2
   // the same network as SCL:
   "FC912_CNT_Tiempo_Mem_UHS"(Temporizar := #T1_ET10 AND #Avance_E1S3 AND #MemFN_pHsE1 AND NOT #pHsMx_E1,
                           Reset := NOT #T1_ET10 AND NOT #T1_ET11,
                           Valor_Tiempo := #V_CNT_ApHsMx_E1,
                           Base_tiempo_ms := 1,
                           Valor_Actual := #TmpAus_E1,
                           Tiempo_OK => #OK_TmpAusE1);
END_REGION

REGION Network 24: TMP AUSENCIA S2
   RUNG wire#powerrail
      "FC912_CNT_Tiempo_Mem_UHS"(Temporizar := wire#w1, Reset := wire#w2, Valor_Tiempo := #V_CNT_ApHsMx_S2, Base_tiempo_ms := 1, Valor_Actual := #TmpAus_S2, Tiempo_OK => #OK_TmpAusS2)
   END_RUNG
   RUNG wire#powerrail
      Contact( #T1_ET60 )
      Contact( #Avance_S2 )
      Contact( #MemFN_pHsS2 )
      I_Contact( #pHsMx_S2 )
   END_RUNG wire#w1
   RUNG wire#powerrail
      I_Contact( #T1_ET60 )
   END_RUNG wire#w2
   // the same network as SCL:
   "FC912_CNT_Tiempo_Mem_UHS"(Temporizar := #T1_ET60 AND #Avance_S2 AND #MemFN_pHsS2 AND NOT #pHsMx_S2,
                           Reset := NOT #T1_ET60,
                           Valor_Tiempo := #V_CNT_ApHsMx_S2,
                           Base_tiempo_ms := 1,
                           Valor_Actual := #TmpAus_S2,
                           Tiempo_OK => #OK_TmpAusS2);
END_REGION

REGION Network 25: TMP AUSENCIA S3
   RUNG wire#powerrail
      "FC912_CNT_Tiempo_Mem_UHS"(Temporizar := wire#w1, Reset := wire#w2, Valor_Tiempo := #V_CNT_ApHsMx_S3, Base_tiempo_ms := 1, Valor_Actual := #TmpAus_S3, Tiempo_OK => #OK_TmpAusS3)
   END_RUNG
   RUNG wire#powerrail
      Contact( #T1_ET50 )
      Contact( #Avance_E1S3 )
      Contact( #MemFN_pHsS3 )
      I_Contact( #pHsMx_S3 )
   END_RUNG wire#w1
   RUNG wire#powerrail
      I_Contact( #T1_ET50 )
   END_RUNG wire#w2
   // the same network as SCL:
   "FC912_CNT_Tiempo_Mem_UHS"(Temporizar := #T1_ET50 AND #Avance_E1S3 AND #MemFN_pHsS3 AND NOT #pHsMx_S3,
                           Reset := NOT #T1_ET50,
                           Valor_Tiempo := #V_CNT_ApHsMx_S3,
                           Base_tiempo_ms := 1,
                           Valor_Actual := #TmpAus_S3,
                           Tiempo_OK => #OK_TmpAusS3);
END_REGION

REGION Network 26: TMP VACIADO
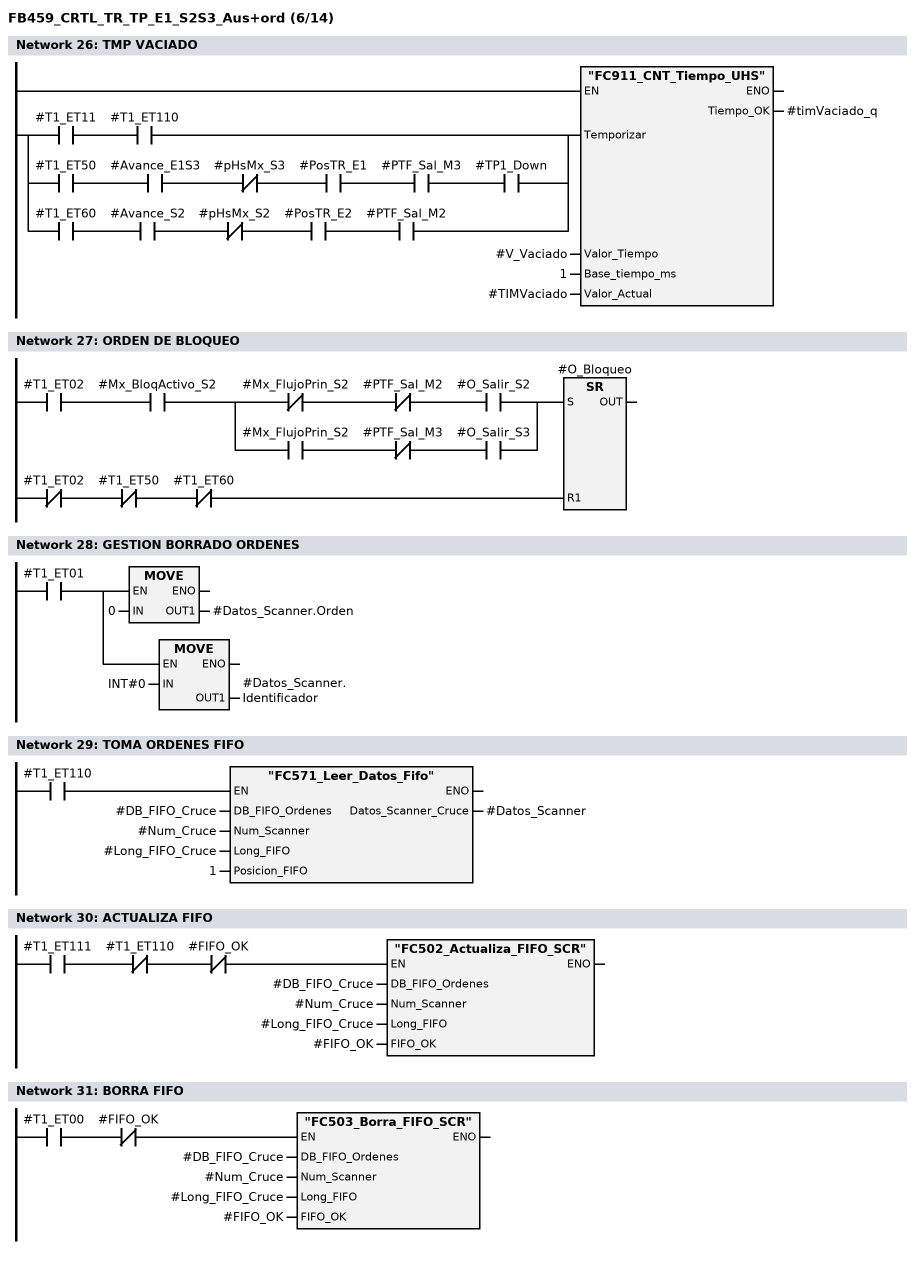
   RUNG wire#powerrail
      "FC911_CNT_Tiempo_UHS"(Temporizar := wire#w1, Valor_Tiempo := #V_Vaciado, Base_tiempo_ms := 1, Valor_Actual := #TIMVaciado, Tiempo_OK => #timVaciado_q)
   END_RUNG
   RUNG wire#powerrail
      Contact( #T1_ET11 )
      Contact( #T1_ET110 )
   END_RUNG wire#w1
   RUNG wire#powerrail
      Contact( #T1_ET50 )
      Contact( #Avance_E1S3 )
      I_Contact( #pHsMx_S3 )
      Contact( #PosTR_E1 )
      Contact( #PTF_Sal_M3 )
      Contact( #TP1_Down )
   END_RUNG wire#w1
   RUNG wire#powerrail
      Contact( #T1_ET60 )
      Contact( #Avance_S2 )
      I_Contact( #pHsMx_S2 )
      Contact( #PosTR_E2 )
      Contact( #PTF_Sal_M2 )
   END_RUNG wire#w1
   // the same network as SCL:
   "FC911_CNT_Tiempo_UHS"(Temporizar := (#T1_ET11 AND #T1_ET110) OR (#T1_ET50 AND #Avance_E1S3 AND NOT #pHsMx_S3 AND #PosTR_E1 AND #PTF_Sal_M3 AND #TP1_Down) OR (#T1_ET60 AND #Avance_S2 AND NOT #pHsMx_S2 AND #PosTR_E2 AND #PTF_Sal_M2),
                          Valor_Tiempo := #V_Vaciado,
                          Base_tiempo_ms := 1,
                          Valor_Actual := #TIMVaciado,
                          Tiempo_OK => #timVaciado_q);
END_REGION

REGION Network 27: ORDEN DE BLOQUEO
   RUNG wire#powerrail
      Contact( #T1_ET02 )
      Contact( #Mx_BloqActivo_S2 )
      wire#w1
      I_Contact( #Mx_FlujoPrin_S2 )
      I_Contact( #PTF_Sal_M2 )
      Contact( #O_Salir_S2 )
      wire#w2
      S_SR(operand := #O_Bloqueo, r1 := wire#w3)
   END_RUNG
   RUNG wire#w1
      Contact( #Mx_FlujoPrin_S2 )
      I_Contact( #PTF_Sal_M3 )
      Contact( #O_Salir_S3 )
   END_RUNG wire#w2
   RUNG wire#powerrail
      I_Contact( #T1_ET02 )
      I_Contact( #T1_ET50 )
      I_Contact( #T1_ET60 )
   END_RUNG wire#w3
   // the same network as SCL:
   IF #T1_ET02 AND #Mx_BloqActivo_S2 AND ((NOT #Mx_FlujoPrin_S2 AND NOT #PTF_Sal_M2 AND #O_Salir_S2) OR (#Mx_FlujoPrin_S2 AND NOT #PTF_Sal_M3 AND #O_Salir_S3)) THEN
       #O_Bloqueo := TRUE;   // SR flip-flop
   END_IF;
   IF NOT #T1_ET02 AND NOT #T1_ET50 AND NOT #T1_ET60 THEN #O_Bloqueo := FALSE; END_IF;
END_REGION

REGION Network 28: GESTION BORRADO ORDENES
   RUNG wire#powerrail
      Contact( #T1_ET01 )
      wire#w1
      { S7_GenerateENO := "TRUE" } Move(in := 0, out1 => #Datos_Scanner.Orden)
   END_RUNG
   RUNG wire#w1
      { S7_GenerateENO := "TRUE" } Move(in := INT#0, out1 => #Datos_Scanner.Identificador)
   END_RUNG
   // the same network as SCL:
   IF #T1_ET01 THEN
       #Datos_Scanner.Orden := 0;
       #Datos_Scanner.Identificador := INT#0;
   END_IF;
END_REGION

REGION Network 29: TOMA ORDENES FIFO
   RUNG wire#powerrail
      Contact( #T1_ET110 )
      "FC571_Leer_Datos_Fifo"(DB_FIFO_Ordenes := #DB_FIFO_Cruce, Num_Scanner := #Num_Cruce, Long_FIFO := #Long_FIFO_Cruce, Posicion_FIFO := 1, Datos_Scanner_Cruce => #Datos_Scanner)
   END_RUNG
   // the same network as SCL:
   IF #T1_ET110 THEN
       "FC571_Leer_Datos_Fifo"(DB_FIFO_Ordenes := #DB_FIFO_Cruce,
                               Num_Scanner := #Num_Cruce,
                               Long_FIFO := #Long_FIFO_Cruce,
                               Posicion_FIFO := 1,
                               Datos_Scanner_Cruce => #Datos_Scanner);
   END_IF;
END_REGION

REGION Network 30: ACTUALIZA FIFO
   RUNG wire#powerrail
      Contact( #T1_ET111 )
      I_Contact( #T1_ET110 )
      I_Contact( #FIFO_OK )
      "FC502_Actualiza_FIFO_SCR"(DB_FIFO_Ordenes := #DB_FIFO_Cruce, Num_Scanner := #Num_Cruce, Long_FIFO := #Long_FIFO_Cruce, FIFO_OK := #FIFO_OK)
   END_RUNG
   // the same network as SCL:
   IF #T1_ET111 AND NOT #T1_ET110 AND NOT #FIFO_OK THEN
       "FC502_Actualiza_FIFO_SCR"(DB_FIFO_Ordenes := #DB_FIFO_Cruce,
                               Num_Scanner := #Num_Cruce,
                               Long_FIFO := #Long_FIFO_Cruce,
                               FIFO_OK := #FIFO_OK);
   END_IF;
END_REGION

REGION Network 31: BORRA FIFO
   RUNG wire#powerrail
      Contact( #T1_ET00 )
      I_Contact( #FIFO_OK )
      "FC503_Borra_FIFO_SCR"(DB_FIFO_Ordenes := #DB_FIFO_Cruce, Num_Scanner := #Num_Cruce, Long_FIFO := #Long_FIFO_Cruce, FIFO_OK := #FIFO_OK)
   END_RUNG
   // the same network as SCL:
   IF #T1_ET00 AND NOT #FIFO_OK THEN
       "FC503_Borra_FIFO_SCR"(DB_FIFO_Ordenes := #DB_FIFO_Cruce,
                              Num_Scanner := #Num_Cruce,
                              Long_FIFO := #Long_FIFO_Cruce,
                              FIFO_OK := #FIFO_OK);
   END_IF;
END_REGION

REGION Network 32: PASAR ORDEN SALIDA S3
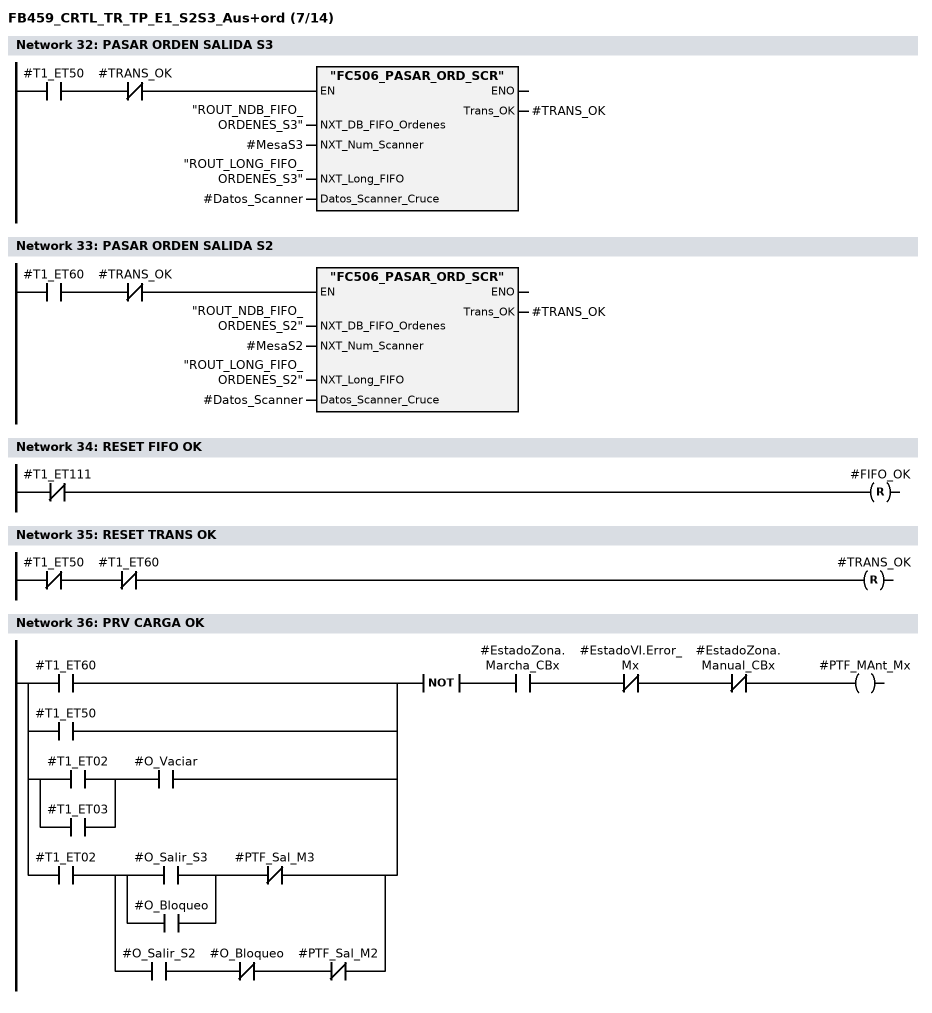
   RUNG wire#powerrail
      Contact( #T1_ET50 )
      I_Contact( #TRANS_OK )
      "FC506_PASAR_ORD_SCR"(NXT_DB_FIFO_Ordenes := "ROUT_NDB_FIFO_ORDENES_S3", NXT_Num_Scanner := #MesaS3, NXT_Long_FIFO := "ROUT_LONG_FIFO_ORDENES_S3", Datos_Scanner_Cruce := #Datos_Scanner, Trans_OK => #TRANS_OK)
   END_RUNG
   // the same network as SCL:
   IF #T1_ET50 AND NOT #TRANS_OK THEN
       "FC506_PASAR_ORD_SCR"(NXT_DB_FIFO_Ordenes := "ROUT_NDB_FIFO_ORDENES_S3",
                             NXT_Num_Scanner := #MesaS3,
                             NXT_Long_FIFO := "ROUT_LONG_FIFO_ORDENES_S3",
                             Datos_Scanner_Cruce := #Datos_Scanner,
                             Trans_OK => #TRANS_OK);
   END_IF;
END_REGION

REGION Network 33: PASAR ORDEN SALIDA S2
   RUNG wire#powerrail
      Contact( #T1_ET60 )
      I_Contact( #TRANS_OK )
      "FC506_PASAR_ORD_SCR"(NXT_DB_FIFO_Ordenes := "ROUT_NDB_FIFO_ORDENES_S2", NXT_Num_Scanner := #MesaS2, NXT_Long_FIFO := "ROUT_LONG_FIFO_ORDENES_S2", Datos_Scanner_Cruce := #Datos_Scanner, Trans_OK => #TRANS_OK)
   END_RUNG
   // the same network as SCL:
   IF #T1_ET60 AND NOT #TRANS_OK THEN
       "FC506_PASAR_ORD_SCR"(NXT_DB_FIFO_Ordenes := "ROUT_NDB_FIFO_ORDENES_S2",
                             NXT_Num_Scanner := #MesaS2,
                             NXT_Long_FIFO := "ROUT_LONG_FIFO_ORDENES_S2",
                             Datos_Scanner_Cruce := #Datos_Scanner,
                             Trans_OK => #TRANS_OK);
   END_IF;
END_REGION

REGION Network 34: RESET FIFO OK
   RUNG wire#powerrail
      I_Contact( #T1_ET111 )
      R_Coil( #FIFO_OK )
   END_RUNG
   // the same network as SCL:
   IF NOT #T1_ET111 THEN #FIFO_OK := FALSE; END_IF;
END_REGION

REGION Network 35: RESET TRANS OK
   RUNG wire#powerrail
      I_Contact( #T1_ET50 )
      I_Contact( #T1_ET60 )
      R_Coil( #TRANS_OK )
   END_RUNG
   // the same network as SCL:
   IF NOT #T1_ET50 AND NOT #T1_ET60 THEN #TRANS_OK := FALSE; END_IF;
END_REGION

REGION Network 36: PRV CARGA OK
   RUNG wire#powerrail
      Contact( #T1_ET60 )
      wire#w1
      Not()
      Contact( #EstadoZona.Marcha_CBx )
      I_Contact( #EstadoVI.Error_Mx )
      I_Contact( #EstadoZona.Manual_CBx )
      Coil( #PTF_MAnt_Mx )
   END_RUNG
   RUNG wire#powerrail
      Contact( #T1_ET50 )
   END_RUNG wire#w1
   RUNG wire#powerrail
      Contact( #T1_ET02 )
      wire#w2
      Contact( #O_Vaciar )
   END_RUNG wire#w1
   RUNG wire#powerrail
      Contact( #T1_ET03 )
   END_RUNG wire#w2
   RUNG wire#powerrail
      Contact( #T1_ET02 )
      wire#w3
      Contact( #O_Salir_S3 )
      wire#w4
      I_Contact( #PTF_Sal_M3 )
   END_RUNG wire#w1
   RUNG wire#w3
      Contact( #O_Bloqueo )
   END_RUNG wire#w4
   RUNG wire#w3
      Contact( #O_Salir_S2 )
      I_Contact( #O_Bloqueo )
      I_Contact( #PTF_Sal_M2 )
   END_RUNG wire#w1
   // the same network as SCL:
   #PTF_MAnt_Mx := NOT (#T1_ET60 OR #T1_ET50 OR ((#T1_ET02 OR #T1_ET03) AND #O_Vaciar) OR (#T1_ET02 AND (((#O_Salir_S3 OR #O_Bloqueo) AND NOT #PTF_Sal_M3) OR (#O_Salir_S2 AND NOT #O_Bloqueo AND NOT #PTF_Sal_M2)))) AND #EstadoZona.Marcha_CBx AND NOT #EstadoVI.Error_Mx AND NOT #EstadoZona.Manual_CBx;
END_REGION

REGION Network 37: NXT AVISO TRANSFERENCIA S3
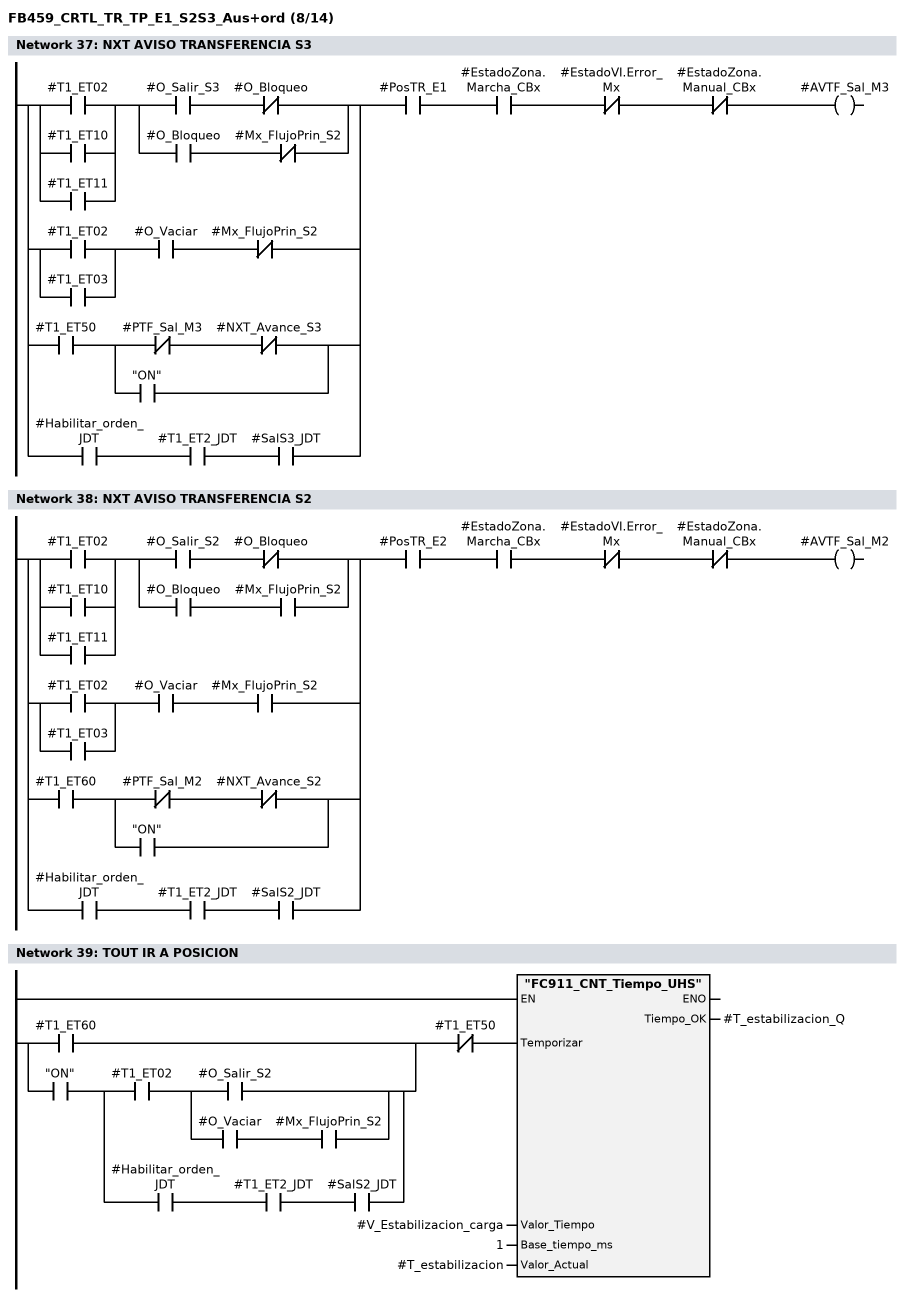
   RUNG wire#powerrail
      Contact( #T1_ET02 )
      wire#w1
      Contact( #O_Salir_S3 )
      I_Contact( #O_Bloqueo )
      wire#w2
      Contact( #PosTR_E1 )
      Contact( #EstadoZona.Marcha_CBx )
      I_Contact( #EstadoVI.Error_Mx )
      I_Contact( #EstadoZona.Manual_CBx )
      Coil( #AVTF_Sal_M3 )
   END_RUNG
   RUNG wire#powerrail
      Contact( #T1_ET10 )
   END_RUNG wire#w1
   RUNG wire#powerrail
      Contact( #T1_ET11 )
   END_RUNG wire#w1
   RUNG wire#w1
      Contact( #O_Bloqueo )
      I_Contact( #Mx_FlujoPrin_S2 )
   END_RUNG wire#w2
   RUNG wire#powerrail
      Contact( #T1_ET02 )
      wire#w3
      Contact( #O_Vaciar )
      I_Contact( #Mx_FlujoPrin_S2 )
   END_RUNG wire#w2
   RUNG wire#powerrail
      Contact( #T1_ET03 )
   END_RUNG wire#w3
   RUNG wire#powerrail
      Contact( #T1_ET50 )
      wire#w4
      I_Contact( #PTF_Sal_M3 )
      I_Contact( #NXT_Avance_S3 )
   END_RUNG wire#w2
   RUNG wire#w4
      Contact( "ON" )
   END_RUNG wire#w2
   RUNG wire#powerrail
      Contact( #Habilitar_orden_JDT )
      Contact( #T1_ET2_JDT )
      Contact( #SalS3_JDT )
   END_RUNG wire#w2
   // the same network as SCL:
   #AVTF_Sal_M3 := (((#T1_ET02 OR #T1_ET10 OR #T1_ET11) AND ((#O_Salir_S3 AND NOT #O_Bloqueo) OR (#O_Bloqueo AND NOT #Mx_FlujoPrin_S2))) OR ((#T1_ET02 OR #T1_ET03) AND #O_Vaciar AND NOT #Mx_FlujoPrin_S2) OR (#T1_ET50 AND ((NOT #PTF_Sal_M3 AND NOT #NXT_Avance_S3) OR "ON")) OR (#Habilitar_orden_JDT AND #T1_ET2_JDT AND #SalS3_JDT)) AND #PosTR_E1 AND #EstadoZona.Marcha_CBx AND NOT #EstadoVI.Error_Mx AND NOT #EstadoZona.Manual_CBx;
END_REGION

REGION Network 38: NXT AVISO TRANSFERENCIA S2
   RUNG wire#powerrail
      Contact( #T1_ET02 )
      wire#w1
      Contact( #O_Salir_S2 )
      I_Contact( #O_Bloqueo )
      wire#w2
      Contact( #PosTR_E2 )
      Contact( #EstadoZona.Marcha_CBx )
      I_Contact( #EstadoVI.Error_Mx )
      I_Contact( #EstadoZona.Manual_CBx )
      Coil( #AVTF_Sal_M2 )
   END_RUNG
   RUNG wire#powerrail
      Contact( #T1_ET10 )
   END_RUNG wire#w1
   RUNG wire#powerrail
      Contact( #T1_ET11 )
   END_RUNG wire#w1
   RUNG wire#w1
      Contact( #O_Bloqueo )
      Contact( #Mx_FlujoPrin_S2 )
   END_RUNG wire#w2
   RUNG wire#powerrail
      Contact( #T1_ET02 )
      wire#w3
      Contact( #O_Vaciar )
      Contact( #Mx_FlujoPrin_S2 )
   END_RUNG wire#w2
   RUNG wire#powerrail
      Contact( #T1_ET03 )
   END_RUNG wire#w3
   RUNG wire#powerrail
      Contact( #T1_ET60 )
      wire#w4
      I_Contact( #PTF_Sal_M2 )
      I_Contact( #NXT_Avance_S2 )
   END_RUNG wire#w2
   RUNG wire#w4
      Contact( "ON" )
   END_RUNG wire#w2
   RUNG wire#powerrail
      Contact( #Habilitar_orden_JDT )
      Contact( #T1_ET2_JDT )
      Contact( #SalS2_JDT )
   END_RUNG wire#w2
   // the same network as SCL:
   #AVTF_Sal_M2 := (((#T1_ET02 OR #T1_ET10 OR #T1_ET11) AND ((#O_Salir_S2 AND NOT #O_Bloqueo) OR (#O_Bloqueo AND #Mx_FlujoPrin_S2))) OR ((#T1_ET02 OR #T1_ET03) AND #O_Vaciar AND #Mx_FlujoPrin_S2) OR (#T1_ET60 AND ((NOT #PTF_Sal_M2 AND NOT #NXT_Avance_S2) OR "ON")) OR (#Habilitar_orden_JDT AND #T1_ET2_JDT AND #SalS2_JDT)) AND #PosTR_E2 AND #EstadoZona.Marcha_CBx AND NOT #EstadoVI.Error_Mx AND NOT #EstadoZona.Manual_CBx;
END_REGION

REGION Network 39: TOUT IR A POSICION
   RUNG wire#powerrail
      "FC911_CNT_Tiempo_UHS"(Temporizar := wire#w4, Valor_Tiempo := #V_Estabilizacion_carga, Base_tiempo_ms := 1, Valor_Actual := #T_estabilizacion, Tiempo_OK => #T_estabilizacion_Q)
   END_RUNG
   RUNG wire#powerrail
      Contact( #T1_ET60 )
      wire#w1
      I_Contact( #T1_ET50 )
   END_RUNG wire#w4
   RUNG wire#powerrail
      Contact( "ON" )
      wire#w2
      Contact( #T1_ET02 )
      wire#w3
      Contact( #O_Salir_S2 )
   END_RUNG wire#w1
   RUNG wire#w3
      Contact( #O_Vaciar )
      Contact( #Mx_FlujoPrin_S2 )
   END_RUNG wire#w1
   RUNG wire#w2
      Contact( #Habilitar_orden_JDT )
      Contact( #T1_ET2_JDT )
      Contact( #SalS2_JDT )
   END_RUNG wire#w1
   // the same network as SCL:
   "FC911_CNT_Tiempo_UHS"(Temporizar := (#T1_ET60 OR ("ON" AND ((#T1_ET02 AND (#O_Salir_S2 OR (#O_Vaciar AND #Mx_FlujoPrin_S2))) OR (#Habilitar_orden_JDT AND #T1_ET2_JDT AND #SalS2_JDT)))) AND NOT #T1_ET50,
                          Valor_Tiempo := #V_Estabilizacion_carga,
                          Base_tiempo_ms := 1,
                          Valor_Actual := #T_estabilizacion,
                          Tiempo_OK => #T_estabilizacion_Q);
END_REGION

REGION Network 40: MA IR POS 24
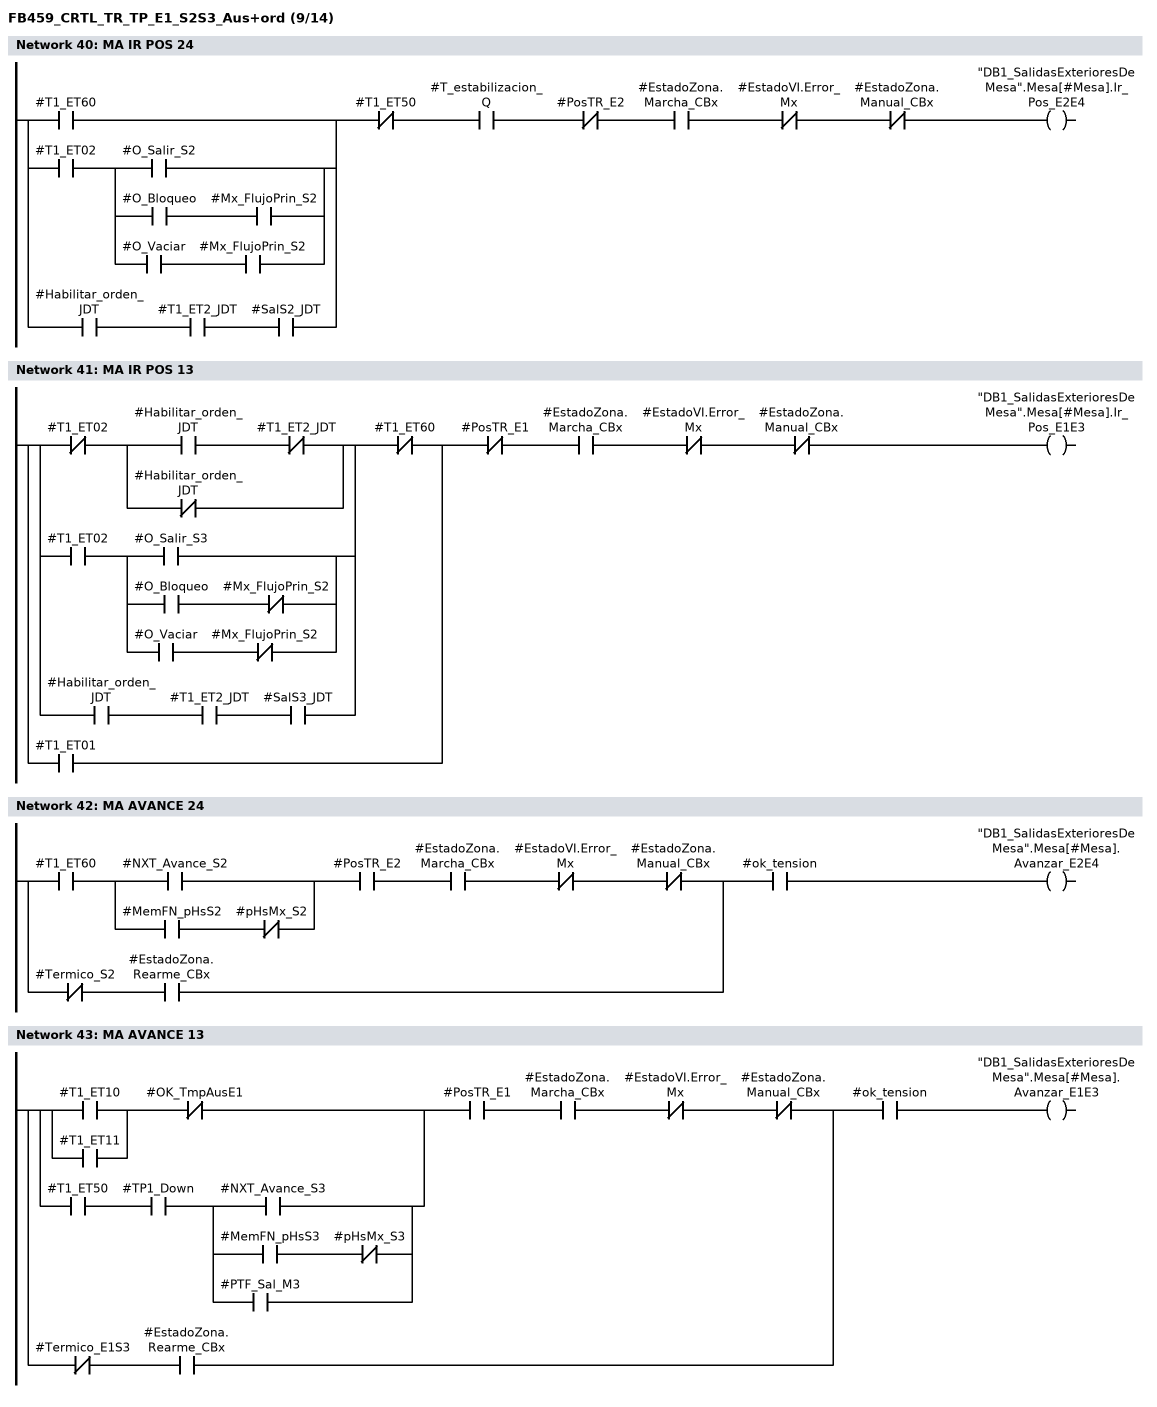
   RUNG wire#powerrail
      Contact( #T1_ET60 )
      wire#w1
      I_Contact( #T1_ET50 )
      Contact( #T_estabilizacion_Q )
      I_Contact( #PosTR_E2 )
      Contact( #EstadoZona.Marcha_CBx )
      I_Contact( #EstadoVI.Error_Mx )
      I_Contact( #EstadoZona.Manual_CBx )
      Coil( "DB1_SalidasExterioresDeMesa".Mesa[#Mesa].Ir_Pos_E2E4 )
   END_RUNG
   RUNG wire#powerrail
      Contact( #T1_ET02 )
      wire#w2
      Contact( #O_Salir_S2 )
   END_RUNG wire#w1
   RUNG wire#w2
      Contact( #O_Bloqueo )
      Contact( #Mx_FlujoPrin_S2 )
   END_RUNG wire#w1
   RUNG wire#w2
      Contact( #O_Vaciar )
      Contact( #Mx_FlujoPrin_S2 )
   END_RUNG wire#w1
   RUNG wire#powerrail
      Contact( #Habilitar_orden_JDT )
      Contact( #T1_ET2_JDT )
      Contact( #SalS2_JDT )
   END_RUNG wire#w1
   // the same network as SCL:
   "DB1_SalidasExterioresDeMesa".Mesa[#Mesa].Ir_Pos_E2E4 := (#T1_ET60 OR (#T1_ET02 AND (#O_Salir_S2 OR (#O_Bloqueo AND #Mx_FlujoPrin_S2) OR (#O_Vaciar AND #Mx_FlujoPrin_S2))) OR (#Habilitar_orden_JDT AND #T1_ET2_JDT AND #SalS2_JDT)) AND NOT #T1_ET50 AND #T_estabilizacion_Q AND NOT #PosTR_E2 AND #EstadoZona.Marcha_CBx AND NOT #EstadoVI.Error_Mx AND NOT #EstadoZona.Manual_CBx;
END_REGION

REGION Network 41: MA IR POS 13
   RUNG wire#powerrail
      I_Contact( #T1_ET02 )
      wire#w1
      Contact( #Habilitar_orden_JDT )
      I_Contact( #T1_ET2_JDT )
      wire#w2
      I_Contact( #T1_ET60 )
      wire#w4
      I_Contact( #PosTR_E1 )
      Contact( #EstadoZona.Marcha_CBx )
      I_Contact( #EstadoVI.Error_Mx )
      I_Contact( #EstadoZona.Manual_CBx )
      Coil( "DB1_SalidasExterioresDeMesa".Mesa[#Mesa].Ir_Pos_E1E3 )
   END_RUNG
   RUNG wire#w1
      I_Contact( #Habilitar_orden_JDT )
   END_RUNG wire#w2
   RUNG wire#powerrail
      Contact( #T1_ET02 )
      wire#w3
      Contact( #O_Salir_S3 )
   END_RUNG wire#w2
   RUNG wire#w3
      Contact( #O_Bloqueo )
      I_Contact( #Mx_FlujoPrin_S2 )
   END_RUNG wire#w2
   RUNG wire#w3
      Contact( #O_Vaciar )
      I_Contact( #Mx_FlujoPrin_S2 )
   END_RUNG wire#w2
   RUNG wire#powerrail
      Contact( #Habilitar_orden_JDT )
      Contact( #T1_ET2_JDT )
      Contact( #SalS3_JDT )
   END_RUNG wire#w2
   RUNG wire#powerrail
      Contact( #T1_ET01 )
   END_RUNG wire#w4
   // the same network as SCL:
   "DB1_SalidasExterioresDeMesa".Mesa[#Mesa].Ir_Pos_E1E3 := ((((NOT #T1_ET02 AND ((#Habilitar_orden_JDT AND NOT #T1_ET2_JDT) OR NOT #Habilitar_orden_JDT)) OR (#T1_ET02 AND (#O_Salir_S3 OR (#O_Bloqueo AND NOT #Mx_FlujoPrin_S2) OR (#O_Vaciar AND NOT #Mx_FlujoPrin_S2))) OR (#Habilitar_orden_JDT AND #T1_ET2_JDT AND #SalS3_JDT)) AND NOT #T1_ET60) OR #T1_ET01) AND NOT #PosTR_E1 AND #EstadoZona.Marcha_CBx AND NOT #EstadoVI.Error_Mx AND NOT #EstadoZona.Manual_CBx;
END_REGION

REGION Network 42: MA AVANCE 24
   RUNG wire#powerrail
      Contact( #T1_ET60 )
      wire#w1
      Contact( #NXT_Avance_S2 )
      wire#w2
      Contact( #PosTR_E2 )
      Contact( #EstadoZona.Marcha_CBx )
      I_Contact( #EstadoVI.Error_Mx )
      I_Contact( #EstadoZona.Manual_CBx )
      wire#w3
      Contact( #ok_tension )
      Coil( "DB1_SalidasExterioresDeMesa".Mesa[#Mesa].Avanzar_E2E4 )
   END_RUNG
   RUNG wire#w1
      Contact( #MemFN_pHsS2 )
      I_Contact( #pHsMx_S2 )
   END_RUNG wire#w2
   RUNG wire#powerrail
      I_Contact( #Termico_S2 )
      Contact( #EstadoZona.Rearme_CBx )
   END_RUNG wire#w3
   // the same network as SCL:
   "DB1_SalidasExterioresDeMesa".Mesa[#Mesa].Avanzar_E2E4 := ((#T1_ET60 AND (#NXT_Avance_S2 OR (#MemFN_pHsS2 AND NOT #pHsMx_S2)) AND #PosTR_E2 AND #EstadoZona.Marcha_CBx AND NOT #EstadoVI.Error_Mx AND NOT #EstadoZona.Manual_CBx) OR (NOT #Termico_S2 AND #EstadoZona.Rearme_CBx)) AND #ok_tension;
END_REGION

REGION Network 43: MA AVANCE 13
   RUNG wire#powerrail
      Contact( #T1_ET10 )
      wire#w1
      I_Contact( #OK_TmpAusE1 )
      wire#w2
      Contact( #PosTR_E1 )
      Contact( #EstadoZona.Marcha_CBx )
      I_Contact( #EstadoVI.Error_Mx )
      I_Contact( #EstadoZona.Manual_CBx )
      wire#w4
      Contact( #ok_tension )
      Coil( "DB1_SalidasExterioresDeMesa".Mesa[#Mesa].Avanzar_E1E3 )
   END_RUNG
   RUNG wire#powerrail
      Contact( #T1_ET11 )
   END_RUNG wire#w1
   RUNG wire#powerrail
      Contact( #T1_ET50 )
      Contact( #TP1_Down )
      wire#w3
      Contact( #NXT_Avance_S3 )
   END_RUNG wire#w2
   RUNG wire#w3
      Contact( #MemFN_pHsS3 )
      I_Contact( #pHsMx_S3 )
   END_RUNG wire#w2
   RUNG wire#w3
      Contact( #PTF_Sal_M3 )
   END_RUNG wire#w2
   RUNG wire#powerrail
      I_Contact( #Termico_E1S3 )
      Contact( #EstadoZona.Rearme_CBx )
   END_RUNG wire#w4
   // the same network as SCL:
   "DB1_SalidasExterioresDeMesa".Mesa[#Mesa].Avanzar_E1E3 := (((((#T1_ET10 OR #T1_ET11) AND NOT #OK_TmpAusE1) OR (#T1_ET50 AND #TP1_Down AND (#NXT_Avance_S3 OR (#MemFN_pHsS3 AND NOT #pHsMx_S3) OR #PTF_Sal_M3))) AND #PosTR_E1 AND #EstadoZona.Marcha_CBx AND NOT #EstadoVI.Error_Mx AND NOT #EstadoZona.Manual_CBx) OR (NOT #Termico_E1S3 AND #EstadoZona.Rearme_CBx)) AND #ok_tension;
END_REGION

REGION Network 44: PASAR ETIQUETA JDT
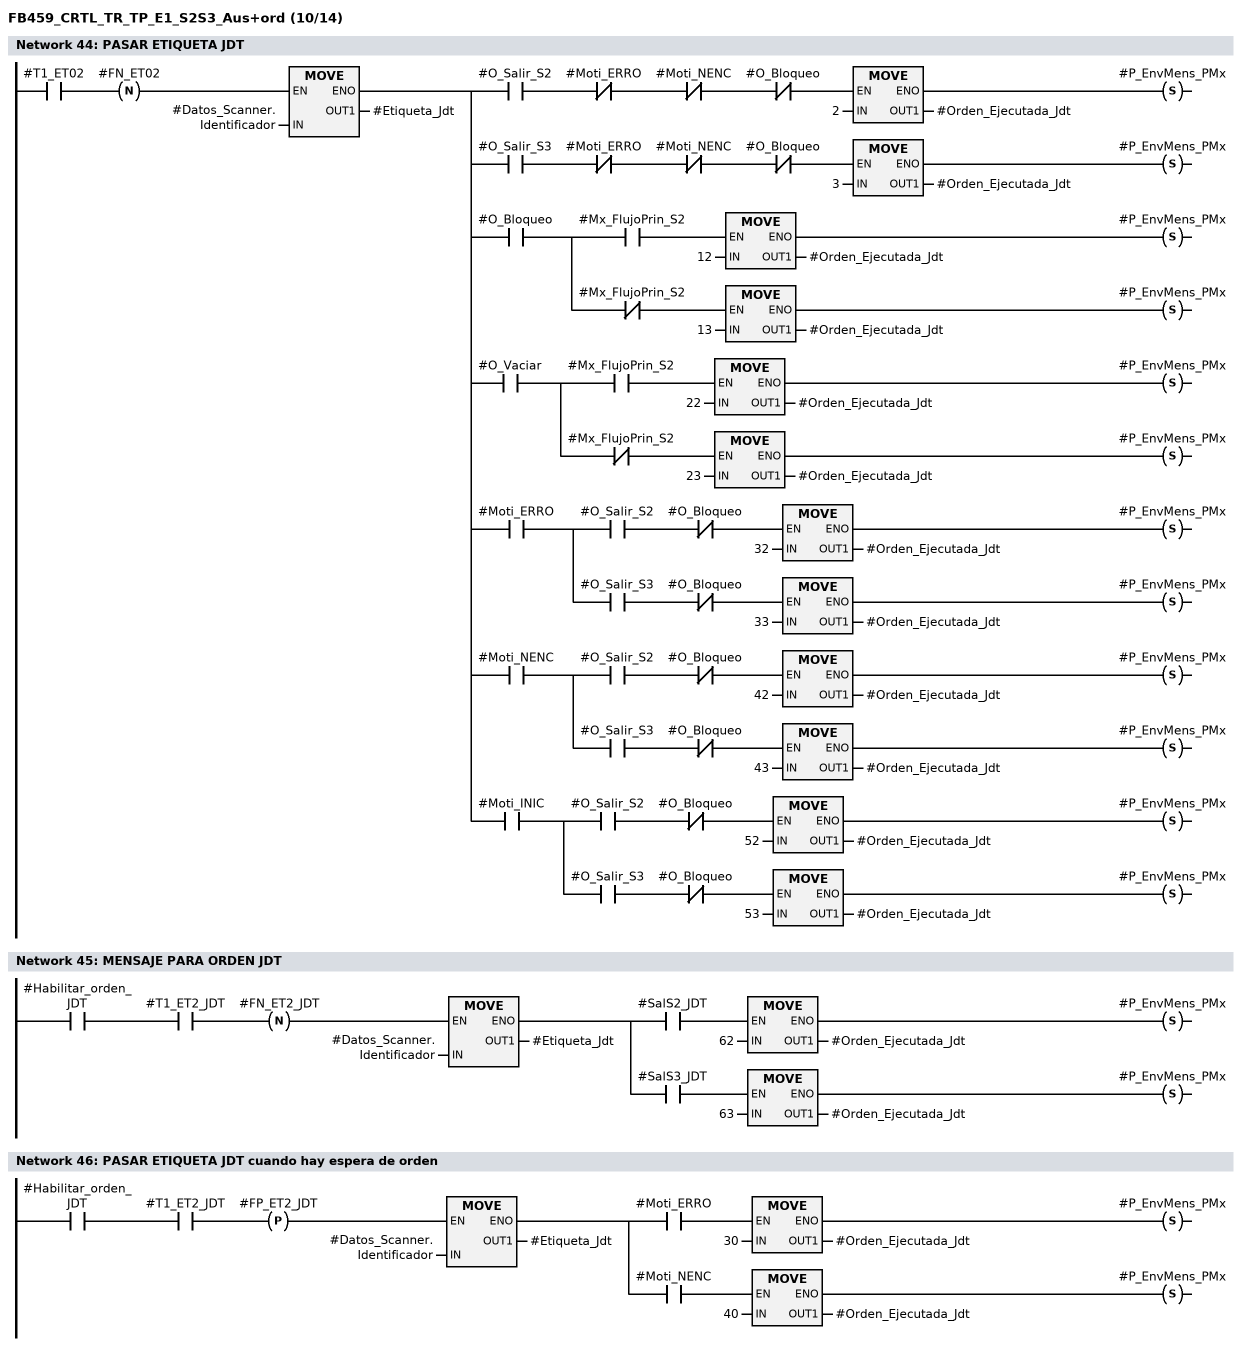
   RUNG wire#powerrail
      Contact( #T1_ET02 )
      N_Trig( #FN_ET02 )
      { S7_GenerateENO := "TRUE" } Move(in := #Datos_Scanner.Identificador, out1 => #Etiqueta_Jdt)
      wire#w1
      Contact( #O_Salir_S2 )
      I_Contact( #Moti_ERRO )
      I_Contact( #Moti_NENC )
      I_Contact( #O_Bloqueo )
      { S7_GenerateENO := "TRUE" } Move(in := 2, out1 => #Orden_Ejecutada_Jdt)
      S_Coil( #P_EnvMens_PMx )
   END_RUNG
   RUNG wire#w1
      Contact( #O_Salir_S3 )
      I_Contact( #Moti_ERRO )
      I_Contact( #Moti_NENC )
      I_Contact( #O_Bloqueo )
      { S7_GenerateENO := "TRUE" } Move(in := 3, out1 => #Orden_Ejecutada_Jdt)
      S_Coil( #P_EnvMens_PMx )
   END_RUNG
   RUNG wire#w1
      Contact( #O_Bloqueo )
      wire#w2
      Contact( #Mx_FlujoPrin_S2 )
      { S7_GenerateENO := "TRUE" } Move(in := 12, out1 => #Orden_Ejecutada_Jdt)
      S_Coil( #P_EnvMens_PMx )
   END_RUNG
   RUNG wire#w2
      I_Contact( #Mx_FlujoPrin_S2 )
      { S7_GenerateENO := "TRUE" } Move(in := 13, out1 => #Orden_Ejecutada_Jdt)
      S_Coil( #P_EnvMens_PMx )
   END_RUNG
   RUNG wire#w1
      Contact( #O_Vaciar )
      wire#w3
      Contact( #Mx_FlujoPrin_S2 )
      { S7_GenerateENO := "TRUE" } Move(in := 22, out1 => #Orden_Ejecutada_Jdt)
      S_Coil( #P_EnvMens_PMx )
   END_RUNG
   RUNG wire#w3
      I_Contact( #Mx_FlujoPrin_S2 )
      { S7_GenerateENO := "TRUE" } Move(in := 23, out1 => #Orden_Ejecutada_Jdt)
      S_Coil( #P_EnvMens_PMx )
   END_RUNG
   RUNG wire#w1
      Contact( #Moti_ERRO )
      wire#w4
      Contact( #O_Salir_S2 )
      I_Contact( #O_Bloqueo )
      { S7_GenerateENO := "TRUE" } Move(in := 32, out1 => #Orden_Ejecutada_Jdt)
      S_Coil( #P_EnvMens_PMx )
   END_RUNG
   RUNG wire#w4
      Contact( #O_Salir_S3 )
      I_Contact( #O_Bloqueo )
      { S7_GenerateENO := "TRUE" } Move(in := 33, out1 => #Orden_Ejecutada_Jdt)
      S_Coil( #P_EnvMens_PMx )
   END_RUNG
   RUNG wire#w1
      Contact( #Moti_NENC )
      wire#w5
      Contact( #O_Salir_S2 )
      I_Contact( #O_Bloqueo )
      { S7_GenerateENO := "TRUE" } Move(in := 42, out1 => #Orden_Ejecutada_Jdt)
      S_Coil( #P_EnvMens_PMx )
   END_RUNG
   RUNG wire#w5
      Contact( #O_Salir_S3 )
      I_Contact( #O_Bloqueo )
      { S7_GenerateENO := "TRUE" } Move(in := 43, out1 => #Orden_Ejecutada_Jdt)
      S_Coil( #P_EnvMens_PMx )
   END_RUNG
   RUNG wire#w1
      Contact( #Moti_INIC )
      wire#w6
      Contact( #O_Salir_S2 )
      I_Contact( #O_Bloqueo )
      { S7_GenerateENO := "TRUE" } Move(in := 52, out1 => #Orden_Ejecutada_Jdt)
      S_Coil( #P_EnvMens_PMx )
   END_RUNG
   RUNG wire#w6
      Contact( #O_Salir_S3 )
      I_Contact( #O_Bloqueo )
      { S7_GenerateENO := "TRUE" } Move(in := 53, out1 => #Orden_Ejecutada_Jdt)
      S_Coil( #P_EnvMens_PMx )
   END_RUNG
   // the same network as SCL:
   // ENO of a box is taken as its EN; it also drops when the box reports an error
   #_w1 := NOT #T1_ET02 AND #FN_ET02;   // falling edge
   #FN_ET02 := #T1_ET02;
   IF #_w1 THEN #Etiqueta_Jdt := #Datos_Scanner.Identificador; END_IF;
   IF #_w1 AND #O_Salir_S2 AND NOT #Moti_ERRO AND NOT #Moti_NENC AND NOT #O_Bloqueo THEN
       #Orden_Ejecutada_Jdt := 2;
       #P_EnvMens_PMx := TRUE;
   END_IF;
   IF #_w1 AND #O_Salir_S3 AND NOT #Moti_ERRO AND NOT #Moti_NENC AND NOT #O_Bloqueo THEN
       #Orden_Ejecutada_Jdt := 3;
       #P_EnvMens_PMx := TRUE;
   END_IF;
   #_w2 := #_w1 AND #O_Bloqueo;
   IF #_w2 AND #Mx_FlujoPrin_S2 THEN
       #Orden_Ejecutada_Jdt := 12;
       #P_EnvMens_PMx := TRUE;
   END_IF;
   IF #_w2 AND NOT #Mx_FlujoPrin_S2 THEN
       #Orden_Ejecutada_Jdt := 13;
       #P_EnvMens_PMx := TRUE;
   END_IF;
   #_w3 := #_w1 AND #O_Vaciar;
   IF #_w3 AND #Mx_FlujoPrin_S2 THEN
       #Orden_Ejecutada_Jdt := 22;
       #P_EnvMens_PMx := TRUE;
   END_IF;
   IF #_w3 AND NOT #Mx_FlujoPrin_S2 THEN
       #Orden_Ejecutada_Jdt := 23;
       #P_EnvMens_PMx := TRUE;
   END_IF;
   #_w4 := #_w1 AND #Moti_ERRO;
   IF #_w4 AND #O_Salir_S2 AND NOT #O_Bloqueo THEN
       #Orden_Ejecutada_Jdt := 32;
       #P_EnvMens_PMx := TRUE;
   END_IF;
   IF #_w4 AND #O_Salir_S3 AND NOT #O_Bloqueo THEN
       #Orden_Ejecutada_Jdt := 33;
       #P_EnvMens_PMx := TRUE;
   END_IF;
   #_w5 := #_w1 AND #Moti_NENC;
   IF #_w5 AND #O_Salir_S2 AND NOT #O_Bloqueo THEN
       #Orden_Ejecutada_Jdt := 42;
       #P_EnvMens_PMx := TRUE;
   END_IF;
   IF #_w5 AND #O_Salir_S3 AND NOT #O_Bloqueo THEN
       #Orden_Ejecutada_Jdt := 43;
       #P_EnvMens_PMx := TRUE;
   END_IF;
   #_w6 := #_w1 AND #Moti_INIC;
   IF #_w6 AND #O_Salir_S2 AND NOT #O_Bloqueo THEN
       #Orden_Ejecutada_Jdt := 52;
       #P_EnvMens_PMx := TRUE;
   END_IF;
   IF #_w6 AND #O_Salir_S3 AND NOT #O_Bloqueo THEN
       #Orden_Ejecutada_Jdt := 53;
       #P_EnvMens_PMx := TRUE;
   END_IF;
END_REGION

REGION Network 45: MENSAJE PARA ORDEN JDT
   RUNG wire#powerrail
      Contact( #Habilitar_orden_JDT )
      Contact( #T1_ET2_JDT )
      N_Trig( #FN_ET2_JDT )
      { S7_GenerateENO := "TRUE" } Move(in := #Datos_Scanner.Identificador, out1 => #Etiqueta_Jdt)
      wire#w1
      Contact( #SalS2_JDT )
      { S7_GenerateENO := "TRUE" } Move(in := 62, out1 => #Orden_Ejecutada_Jdt)
      S_Coil( #P_EnvMens_PMx )
   END_RUNG
   RUNG wire#w1
      Contact( #SalS3_JDT )
      { S7_GenerateENO := "TRUE" } Move(in := 63, out1 => #Orden_Ejecutada_Jdt)
      S_Coil( #P_EnvMens_PMx )
   END_RUNG
   // the same network as SCL:
   // ENO of a box is taken as its EN; it also drops when the box reports an error
   #_w1 := #Habilitar_orden_JDT AND #T1_ET2_JDT;
   #_w2 := NOT #_w1 AND #FN_ET2_JDT;   // falling edge
   #FN_ET2_JDT := #_w1;
   IF #_w2 THEN #Etiqueta_Jdt := #Datos_Scanner.Identificador; END_IF;
   IF #_w2 AND #SalS2_JDT THEN
       #Orden_Ejecutada_Jdt := 62;
       #P_EnvMens_PMx := TRUE;
   END_IF;
   IF #_w2 AND #SalS3_JDT THEN
       #Orden_Ejecutada_Jdt := 63;
       #P_EnvMens_PMx := TRUE;
   END_IF;
END_REGION

REGION Network 46: PASAR ETIQUETA JDT cuando hay espera de orden
   RUNG wire#powerrail
      Contact( #Habilitar_orden_JDT )
      Contact( #T1_ET2_JDT )
      P_Trig( #FP_ET2_JDT )
      { S7_GenerateENO := "TRUE" } Move(in := #Datos_Scanner.Identificador, out1 => #Etiqueta_Jdt)
      wire#w1
      Contact( #Moti_ERRO )
      { S7_GenerateENO := "TRUE" } Move(in := 30, out1 => #Orden_Ejecutada_Jdt)
      S_Coil( #P_EnvMens_PMx )
   END_RUNG
   RUNG wire#w1
      Contact( #Moti_NENC )
      { S7_GenerateENO := "TRUE" } Move(in := 40, out1 => #Orden_Ejecutada_Jdt)
      S_Coil( #P_EnvMens_PMx )
   END_RUNG
   // the same network as SCL:
   // ENO of a box is taken as its EN; it also drops when the box reports an error
   #_w1 := #Habilitar_orden_JDT AND #T1_ET2_JDT;
   #_w2 := #_w1 AND NOT #FP_ET2_JDT;   // rising edge
   #FP_ET2_JDT := #_w1;
   IF #_w2 THEN #Etiqueta_Jdt := #Datos_Scanner.Identificador; END_IF;
   IF #_w2 AND #Moti_ERRO THEN
       #Orden_Ejecutada_Jdt := 30;
       #P_EnvMens_PMx := TRUE;
   END_IF;
   IF #_w2 AND #Moti_NENC THEN
       #Orden_Ejecutada_Jdt := 40;
       #P_EnvMens_PMx := TRUE;
   END_IF;
END_REGION

REGION Network 47: RESET PRESENCIA
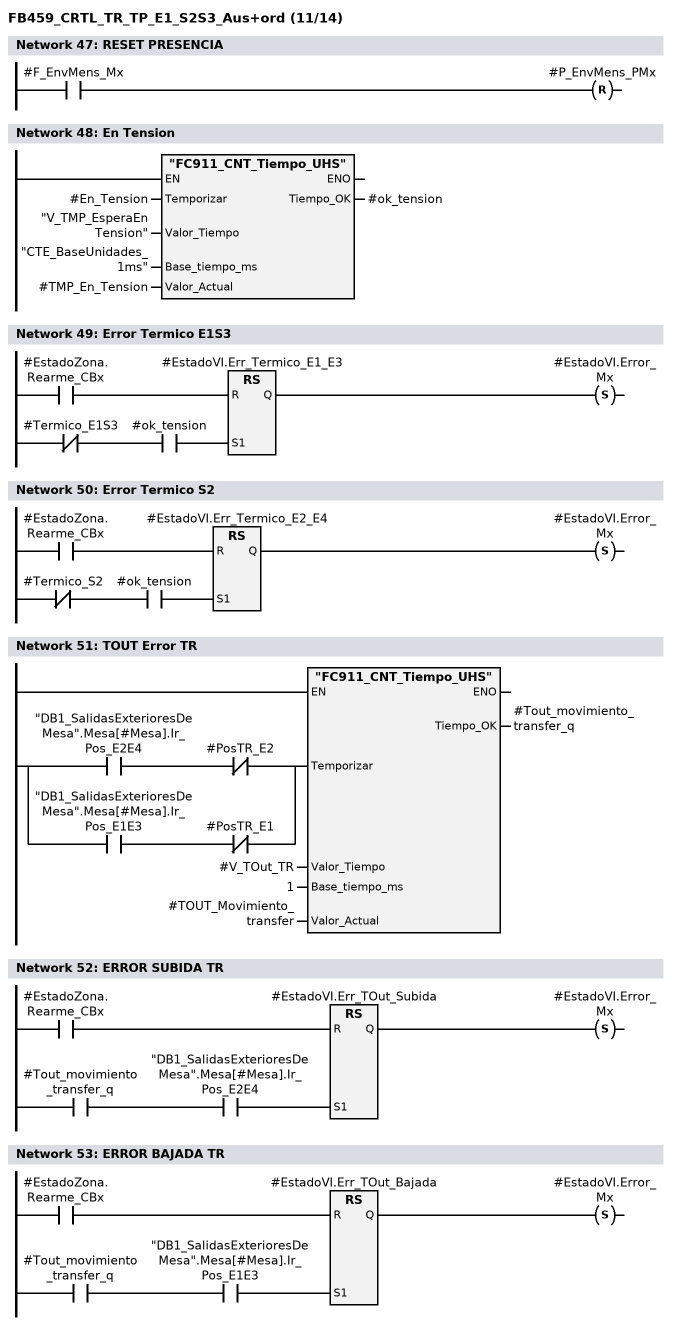
   RUNG wire#powerrail
      Contact( #F_EnvMens_Mx )
      R_Coil( #P_EnvMens_PMx )
   END_RUNG
   // the same network as SCL:
   IF #F_EnvMens_Mx THEN #P_EnvMens_PMx := FALSE; END_IF;
END_REGION

REGION Network 48: En Tension
   RUNG wire#powerrail
      "FC911_CNT_Tiempo_UHS"(Temporizar := #En_Tension, Valor_Tiempo := "V_TMP_EsperaEnTension", Base_tiempo_ms := "CTE_BaseUnidades_1ms", Valor_Actual := #TMP_En_Tension, Tiempo_OK => #ok_tension)
   END_RUNG
   // the same network as SCL:
   "FC911_CNT_Tiempo_UHS"(Temporizar := #En_Tension,
                          Valor_Tiempo := "V_TMP_EsperaEnTension",
                          Base_tiempo_ms := "CTE_BaseUnidades_1ms",
                          Valor_Actual := #TMP_En_Tension,
                          Tiempo_OK => #ok_tension);
END_REGION

REGION Network 49: Error Termico E1S3
   RUNG wire#powerrail
      Contact( #EstadoZona.Rearme_CBx )
      S_RS(operand := #EstadoVI.Err_Termico_E1_E3, s1 := wire#w1)
      S_Coil( #EstadoVI.Error_Mx )
   END_RUNG
   RUNG wire#powerrail
      I_Contact( #Termico_E1S3 )
      Contact( #ok_tension )
   END_RUNG wire#w1
   // the same network as SCL:
   IF #EstadoZona.Rearme_CBx THEN
       #EstadoVI.Err_Termico_E1_E3 := FALSE;   // RS flip-flop
   END_IF;
   IF NOT #Termico_E1S3 AND #ok_tension THEN #EstadoVI.Err_Termico_E1_E3 := TRUE; END_IF;
   IF #EstadoVI.Err_Termico_E1_E3 THEN #EstadoVI.Error_Mx := TRUE; END_IF;
END_REGION

REGION Network 50: Error Termico S2
   RUNG wire#powerrail
      Contact( #EstadoZona.Rearme_CBx )
      S_RS(operand := #EstadoVI.Err_Termico_E2_E4, s1 := wire#w1)
      S_Coil( #EstadoVI.Error_Mx )
   END_RUNG
   RUNG wire#powerrail
      I_Contact( #Termico_S2 )
      Contact( #ok_tension )
   END_RUNG wire#w1
   // the same network as SCL:
   IF #EstadoZona.Rearme_CBx THEN
       #EstadoVI.Err_Termico_E2_E4 := FALSE;   // RS flip-flop
   END_IF;
   IF NOT #Termico_S2 AND #ok_tension THEN #EstadoVI.Err_Termico_E2_E4 := TRUE; END_IF;
   IF #EstadoVI.Err_Termico_E2_E4 THEN #EstadoVI.Error_Mx := TRUE; END_IF;
END_REGION

